(* CODESYS project BoshanMassa_13.3.project
   CustomField04_name: CustomField04
   CustomField06_name: CustomField06
   CustomField07_name: CustomField07
   CustomField09_name: CustomField09
   CustomField08_name: CustomField08
   CustomField02_name: CustomField02
   CustomField10_name: CustomField10
   CustomField01_name: CustomField01
   CustomField03_name: CustomField03
   CustomField05_name: CustomField05

Project tree, tasks and I/O mapping:
  MASSA : TM238LFDC24DT, Schneider Electric, order no. TM238LFDC24DT, version 4.0.1.28
      settings: Expansion Tasks.Expansion 1 Task Name = 'MAST'; Expansion Tasks.Expansion 2 Task Name = 'MAST'
    application Application
      task MAST (cyclic, interval 20 ms, priority 15, watchdog 100 ms x 1) calls POU_M
      program POU_M [LD]
      visualisation VisualizationM
      Symbols
    TM2DDI32DK : TM2DDI32DK, Schneider Electric, order no. TM2DDI32DK, version 4.0.1.28
        input  i_TZ_KO1 : BOOL  // ID0.I0
        input  i_TZ_KO2 : BOOL  // ID0.I1
        input  i_TZ_KO3 : BOOL  // ID0.I2
        input  i_TZ_KO4 : BOOL  // ID0.I3
        input  i_TZ_KO6 : BOOL  // ID0.I4
        input  i_TZ_KO7 : BOOL  // ID0.I5
        input  i_TZ_SMK517_37 : BOOL  // ID0.I6
        input  i_TZ_SMK517_5 : BOOL  // ID0.I7
        input  i_Nominal_SMK517_ATS : BOOL  // ID0.I8
        input  i_Avar_SMK517_ATS : BOOL  // ID0.I9
        input  i_TZ_SMK516_37 : BOOL  // ID0.I10
        input  i_TZ_SMK516_45 : BOOL  // ID0.I11
        input  i_TZ_KonvSMK516 : BOOL  // ID0.I12
        input  i_TZ_RazrSMK516 : BOOL  // ID0.I13
        input  i_TZ_EP80_1 : BOOL  // ID0.I15
        input  i_TZ_EP80_2 : BOOL  // ID0.I16
        input  i_Tros_KO1 : BOOL  // ID0.I17
        input  i_Tros_KO2 : BOOL  // ID0.I18
        input  i_Tros_KO3 : BOOL  // ID0.I19
        input  i_Tros_KO4 : BOOL  // ID0.I20
        input  i_Tros_KO6 : BOOL  // ID0.I21
        input  i_Tros_KO7 : BOOL  // ID0.I22
        input  i_Othod_SMK517 : BOOL  // ID0.I23
        input  i_Kozhuh_SMK517 : BOOL  // ID0.I24
        input  i_Othod_SMK516 : BOOL  // ID0.I25
        input  i_Kozhuh_SMK516 : BOOL  // ID0.I26
        input  i_Tros_KonvSMK516 : BOOL  // ID0.I27
        input  i_KEY_Protochka : BOOL  // ID0.I28
        input  i_Avar_PL024 : BOOL  // ID0.I31
        unmapped channels: ID0
    Serial Line 1
      Modbus_Manager : Modbus Manager, Schneider Electric, version 4.0.0.2
    Embedded Functions
      HSC : HSC, Schneider Electric, version 4.0.1.28
          settings: HSC00VarName = ''
      IO : IO, Schneider Electric, version 4.0.1.28
          input  i_Avar_PL012 : BOOL  // IW0.I0
          input  i_Rabota_PL250 : BOOL  // IW0.I1
          input  i_Avar_PL250 : BOOL  // IW0.I2
          input  i_Gotov_USM40 : BOOL  // IW0.I3
          input  i_Privoda_USM40_v_rabote : BOOL  // IW0.I4
          input  i_Liniya_USM40_v_rabote : BOOL  // IW0.I5
          input  i_TrosLentaUSM40 : BOOL  // IW0.I6
          input  i_Avar_USM40 : BOOL  // IW0.I7
          input  i_TZ_KO11 : BOOL  // IW0.I8
          input  i_Tros_KO11 : BOOL  // IW0.I9
          input  i_TZ_PL1 : BOOL  // IW0.I10
          input  i_TZ_PL2 : BOOL  // IW0.I11
          input  i_Vkl_Protoch517 : BOOL  // IW0.I12
          input  i_Otkl_Protoch517 : BOOL  // IW0.I13
          unmapped channels: IW0, QW0
      PTO_PWM : PTO_PWM, Schneider Electric, version 4.0.1.28
    CAN
      CANopen_Optimized : CANopen Optimized, Schneider Electric, order no. 1806, version 3.0.1.24
          settings: ConfigVersion = 50659584
        PL250 : Altivar 312, Schneider Electric, order no. 0, version 4.5.0.0
            settings: General Options.Optional Device = TRUE; NODEIDSAVED = 3; SDO Timeout = 1000000; EXPERTSETTINGS = True; Emergency-General Parameters.Emergency COBID = 16#83; Heartbeat-Producer Time = 200; PDO 16#1400.COBID = 16#80000203; PDO 16#1405.COBID = 16#00000303; PDO 16#1800.COBID = 16#80000183; PDO 16#1805.COBID = 16#00000283; Heartbeat-Consuming1.Heartbeat-Time = 300 ms; Drivecom command reg..Subindex = 16#00; Drivecom command reg..Subindex = 16#00; Target velocity.Index = 16#6042; Target velocity.Subindex = 16#00; Target velocity.ObjectLength = 16; Drivecom status register.Subindex = 16#00; Drivecom status register.Subindex = 16#00; Output frequency.Index = 16#2002; Output frequency.Subindex = 16#03; Output frequency.ObjectLength = 16; Motor Current.Index = 16#2002; Motor Current.Subindex = 16#05; Motor Current.ObjectLength = 16; SDO List.Set Guardtime.Index = 16#100C; SDO List.Set Guardtime.Subindex = 16#00; SDO List.Set Guardtime.Value = 16#00000000; SDO List.Set Guardtime.Size = 16; SDO List.Set Guardtime.AbortIfError = FALSE; SDO List.Set Guardtime.JumpToLine = FALSE; SDO List.Set Guardtime.Line = 0; SDO List.Set Lifetime.Index = 16#100D; SDO List.Set Lifetime.Subindex = 16#00; SDO List.Set Lifetime.Value = 16#00000000; SDO List.Set Lifetime.Size = 8; SDO List.Set Lifetime.AbortIfError = FALSE; SDO List.Set Lifetime.JumpToLine = FALSE; SDO List.Set Lifetime.Line = 0; SDO List.Set Heartbeat Consumer.Index = 16#1016; SDO List.Set Heartbeat Consumer.Subindex = 16#01;
              SDO List.Set Heartbeat Consumer.Value = 16#007F012C; SDO List.Set Heartbeat Consumer.Size = 32; SDO List.Set Heartbeat Consumer.AbortIfError = FALSE; SDO List.Set Heartbeat Consumer.JumpToLine = FALSE; SDO List.Set Heartbeat Consumer.Line = 0; SDO List.Set Heartbeat Producer.Index = 16#1017; SDO List.Set Heartbeat Producer.Subindex = 16#00; SDO List.Set Heartbeat Producer.Value = 16#000000C8; SDO List.Set Heartbeat Producer.Size = 16; SDO List.Set Heartbeat Producer.AbortIfError = FALSE; SDO List.Set Heartbeat Producer.JumpToLine = FALSE; SDO List.Set Heartbeat Producer.Line = 0; SDO List.Disable PDO.Index = 16#1400; SDO List.Disable PDO.Subindex = 16#01; SDO List.Disable PDO.Value = 16#80000203; SDO List.Disable PDO.Size = 32; SDO List.Disable PDO.AbortIfError = FALSE; SDO List.Disable PDO.JumpToLine = FALSE; SDO List.Disable PDO.Line = 0; SDO List.Disable PDO.Index = 16#1405; SDO List.Disable PDO.Subindex = 16#01; SDO List.Disable PDO.Value = 16#80000303; SDO List.Disable PDO.Size = 32; SDO List.Disable PDO.AbortIfError = FALSE; SDO List.Disable PDO.JumpToLine = FALSE; SDO List.Disable PDO.Line = 0; SDO List.Set transmission type.Index = 16#1405; SDO List.Set transmission type.Subindex = 16#02; SDO List.Set transmission type.Value = 16#FF; SDO List.Set transmission type.Size = 8; SDO List.Set transmission type.AbortIfError = FALSE; SDO List.Set transmission type.JumpToLine = FALSE; SDO List.Set transmission type.Line = 0; SDO List.Clear pdo mapping.Index = 16#1605; SDO List.Clear pdo mapping.Subindex = 16#00; SDO List.Clear pdo mapping.Value = 16#0; SDO List.Clear pdo mapping.Size = 8; SDO List.Clear pdo mapping.AbortIfError = FALSE; SDO List.Clear pdo mapping.JumpToLine = FALSE; SDO List.Clear pdo mapping.Line = 0;
              SDO List.Set Mapping.Index = 16#1605; SDO List.Set Mapping.Subindex = 16#01; SDO List.Set Mapping.Value = 16#60400010; SDO List.Set Mapping.Size = 32; SDO List.Set Mapping.AbortIfError = FALSE; SDO List.Set Mapping.JumpToLine = FALSE; SDO List.Set Mapping.Line = 0; SDO List.Set Mapping.Index = 16#1605; SDO List.Set Mapping.Subindex = 16#02; SDO List.Set Mapping.Value = 16#60420010; SDO List.Set Mapping.Size = 32; SDO List.Set Mapping.AbortIfError = FALSE; SDO List.Set Mapping.JumpToLine = FALSE; SDO List.Set Mapping.Line = 0; SDO List.Set number of pdos.Index = 16#1605; SDO List.Set number of pdos.Subindex = 16#00; SDO List.Set number of pdos.Value = 16#02; SDO List.Set number of pdos.Size = 8; SDO List.Set number of pdos.AbortIfError = FALSE; SDO List.Set number of pdos.JumpToLine = FALSE; SDO List.Set number of pdos.Line = 0; SDO List.Set and enable COB-ID.Index = 16#1405; SDO List.Set and enable COB-ID.Subindex = 16#01; SDO List.Set and enable COB-ID.Value = 16#00000303; SDO List.Set and enable COB-ID.Size = 32; SDO List.Set and enable COB-ID.AbortIfError = FALSE; SDO List.Set and enable COB-ID.JumpToLine = FALSE; SDO List.Set and enable COB-ID.Line = 0; SDO List.Disable PDO.Index = 16#1800; SDO List.Disable PDO.Subindex = 16#01; SDO List.Disable PDO.Value = 16#80000183; SDO List.Disable PDO.Size = 32; SDO List.Disable PDO.AbortIfError = FALSE; SDO List.Disable PDO.JumpToLine = FALSE; SDO List.Disable PDO.Line = 0; SDO List.Disable PDO.Index = 16#1805; SDO List.Disable PDO.Subindex = 16#01; SDO List.Disable PDO.Value = 16#80000283; SDO List.Disable PDO.Size = 32; SDO List.Disable PDO.AbortIfError = FALSE;
              SDO List.Disable PDO.JumpToLine = FALSE; SDO List.Disable PDO.Line = 0; SDO List.Set transmission type.Index = 16#1805; SDO List.Set transmission type.Subindex = 16#02; SDO List.Set transmission type.Value = 16#FF; SDO List.Set transmission type.Size = 8; SDO List.Set transmission type.AbortIfError = FALSE; SDO List.Set transmission type.JumpToLine = FALSE; SDO List.Set transmission type.Line = 0; SDO List.Set inhibit time.Index = 16#1805; SDO List.Set inhibit time.Subindex = 16#03; SDO List.Set inhibit time.Value = 16#001E; SDO List.Set inhibit time.Size = 16; SDO List.Set inhibit time.AbortIfError = FALSE; SDO List.Set inhibit time.JumpToLine = FALSE; SDO List.Set inhibit time.Line = 0; SDO List.Set event time.Index = 16#1805; SDO List.Set event time.Subindex = 16#05; SDO List.Set event time.Value = 16#0064; SDO List.Set event time.Size = 16; SDO List.Set event time.AbortIfError = FALSE; SDO List.Set event time.JumpToLine = FALSE; SDO List.Set event time.Line = 0; SDO List.Clear pdo mapping.Index = 16#1A05; SDO List.Clear pdo mapping.Subindex = 16#00; SDO List.Clear pdo mapping.Value = 16#0; SDO List.Clear pdo mapping.Size = 8; SDO List.Clear pdo mapping.AbortIfError = FALSE; SDO List.Clear pdo mapping.JumpToLine = FALSE; SDO List.Clear pdo mapping.Line = 0; SDO List.Set Mapping.Index = 16#1A05; SDO List.Set Mapping.Subindex = 16#01; SDO List.Set Mapping.Value = 16#60410010; SDO List.Set Mapping.Size = 32; SDO List.Set Mapping.AbortIfError = FALSE; SDO List.Set Mapping.JumpToLine = FALSE; SDO List.Set Mapping.Line = 0; SDO List.Set Mapping.Index = 16#1A05; SDO List.Set Mapping.Subindex = 16#02; SDO List.Set Mapping.Value = 16#20020310;
              SDO List.Set Mapping.Size = 32; SDO List.Set Mapping.AbortIfError = FALSE; SDO List.Set Mapping.JumpToLine = FALSE; SDO List.Set Mapping.Line = 0; SDO List.Set Mapping.Index = 16#1A05; SDO List.Set Mapping.Subindex = 16#03; SDO List.Set Mapping.Value = 16#20020510; SDO List.Set Mapping.Size = 32; SDO List.Set Mapping.AbortIfError = FALSE; SDO List.Set Mapping.JumpToLine = FALSE; SDO List.Set Mapping.Line = 0; SDO List.Set number of pdos.Index = 16#1A05; SDO List.Set number of pdos.Subindex = 16#00; SDO List.Set number of pdos.Value = 16#03; SDO List.Set number of pdos.Size = 8; SDO List.Set number of pdos.AbortIfError = FALSE; SDO List.Set number of pdos.JumpToLine = FALSE; SDO List.Set number of pdos.Line = 0; SDO List.Set and enable COB-ID.Index = 16#1805; SDO List.Set and enable COB-ID.Subindex = 16#01; SDO List.Set and enable COB-ID.Value = 16#00000283; SDO List.Set and enable COB-ID.Size = 32; SDO List.Set and enable COB-ID.AbortIfError = FALSE; SDO List.Set and enable COB-ID.JumpToLine = FALSE; SDO List.Set and enable COB-ID.Line = 0; ConfigVersion = 50659584
            output q_ATVPL250_Controlword : UINT  // Drivecom command reg.
            output q_ATVPL250_WriteVelocity : INT  // Target velocity
            input  i_ATVPL250_Status : UINT  // Drivecom status register
            input  i_ATVPL250_OutFrec : INT  // Output frequency
            input  i_ATVPL250_OutCur : UINT  // Motor Current
        PL024 : Altivar 312, Schneider Electric, order no. 0, version 4.5.0.0
            settings: General Options.Optional Device = TRUE; NODEIDSAVED = 5; SDO Timeout = 1000000; EXPERTSETTINGS = True; Emergency-General Parameters.Emergency COBID = 16#85; Heartbeat-Producer Time = 200; PDO 16#1400.COBID = 16#80000205; PDO 16#1405.COBID = 16#00000305; PDO 16#1800.COBID = 16#80000185; PDO 16#1805.COBID = 16#00000285; Heartbeat-Consuming1.Heartbeat-Time = 300 ms; Drivecom command reg..Subindex = 16#00; Drivecom command reg..Subindex = 16#00; Target velocity.Index = 16#6042; Target velocity.Subindex = 16#00; Target velocity.ObjectLength = 16; Drivecom status register.Subindex = 16#00; Drivecom status register.Subindex = 16#00; Output frequency.Index = 16#2002; Output frequency.Subindex = 16#03; Output frequency.ObjectLength = 16; Motor Current.Index = 16#2002; Motor Current.Subindex = 16#05; Motor Current.ObjectLength = 16; SDO List.Set Guardtime.Index = 16#100C; SDO List.Set Guardtime.Subindex = 16#00; SDO List.Set Guardtime.Value = 16#00000000; SDO List.Set Guardtime.Size = 16; SDO List.Set Guardtime.AbortIfError = FALSE; SDO List.Set Guardtime.JumpToLine = FALSE; SDO List.Set Guardtime.Line = 0; SDO List.Set Lifetime.Index = 16#100D; SDO List.Set Lifetime.Subindex = 16#00; SDO List.Set Lifetime.Value = 16#00000000; SDO List.Set Lifetime.Size = 8; SDO List.Set Lifetime.AbortIfError = FALSE; SDO List.Set Lifetime.JumpToLine = FALSE; SDO List.Set Lifetime.Line = 0; SDO List.Set Heartbeat Consumer.Index = 16#1016; SDO List.Set Heartbeat Consumer.Subindex = 16#01;
              SDO List.Set Heartbeat Consumer.Value = 16#007F012C; SDO List.Set Heartbeat Consumer.Size = 32; SDO List.Set Heartbeat Consumer.AbortIfError = FALSE; SDO List.Set Heartbeat Consumer.JumpToLine = FALSE; SDO List.Set Heartbeat Consumer.Line = 0; SDO List.Set Heartbeat Producer.Index = 16#1017; SDO List.Set Heartbeat Producer.Subindex = 16#00; SDO List.Set Heartbeat Producer.Value = 16#000000C8; SDO List.Set Heartbeat Producer.Size = 16; SDO List.Set Heartbeat Producer.AbortIfError = FALSE; SDO List.Set Heartbeat Producer.JumpToLine = FALSE; SDO List.Set Heartbeat Producer.Line = 0; SDO List.Disable PDO.Index = 16#1400; SDO List.Disable PDO.Subindex = 16#01; SDO List.Disable PDO.Value = 16#80000205; SDO List.Disable PDO.Size = 32; SDO List.Disable PDO.AbortIfError = FALSE; SDO List.Disable PDO.JumpToLine = FALSE; SDO List.Disable PDO.Line = 0; SDO List.Disable PDO.Index = 16#1405; SDO List.Disable PDO.Subindex = 16#01; SDO List.Disable PDO.Value = 16#80000305; SDO List.Disable PDO.Size = 32; SDO List.Disable PDO.AbortIfError = FALSE; SDO List.Disable PDO.JumpToLine = FALSE; SDO List.Disable PDO.Line = 0; SDO List.Set transmission type.Index = 16#1405; SDO List.Set transmission type.Subindex = 16#02; SDO List.Set transmission type.Value = 16#FF; SDO List.Set transmission type.Size = 8; SDO List.Set transmission type.AbortIfError = FALSE; SDO List.Set transmission type.JumpToLine = FALSE; SDO List.Set transmission type.Line = 0; SDO List.Clear pdo mapping.Index = 16#1605; SDO List.Clear pdo mapping.Subindex = 16#00; SDO List.Clear pdo mapping.Value = 16#0; SDO List.Clear pdo mapping.Size = 8; SDO List.Clear pdo mapping.AbortIfError = FALSE; SDO List.Clear pdo mapping.JumpToLine = FALSE; SDO List.Clear pdo mapping.Line = 0;
              SDO List.Set Mapping.Index = 16#1605; SDO List.Set Mapping.Subindex = 16#01; SDO List.Set Mapping.Value = 16#60400010; SDO List.Set Mapping.Size = 32; SDO List.Set Mapping.AbortIfError = FALSE; SDO List.Set Mapping.JumpToLine = FALSE; SDO List.Set Mapping.Line = 0; SDO List.Set Mapping.Index = 16#1605; SDO List.Set Mapping.Subindex = 16#02; SDO List.Set Mapping.Value = 16#60420010; SDO List.Set Mapping.Size = 32; SDO List.Set Mapping.AbortIfError = FALSE; SDO List.Set Mapping.JumpToLine = FALSE; SDO List.Set Mapping.Line = 0; SDO List.Set number of pdos.Index = 16#1605; SDO List.Set number of pdos.Subindex = 16#00; SDO List.Set number of pdos.Value = 16#02; SDO List.Set number of pdos.Size = 8; SDO List.Set number of pdos.AbortIfError = FALSE; SDO List.Set number of pdos.JumpToLine = FALSE; SDO List.Set number of pdos.Line = 0; SDO List.Set and enable COB-ID.Index = 16#1405; SDO List.Set and enable COB-ID.Subindex = 16#01; SDO List.Set and enable COB-ID.Value = 16#00000305; SDO List.Set and enable COB-ID.Size = 32; SDO List.Set and enable COB-ID.AbortIfError = FALSE; SDO List.Set and enable COB-ID.JumpToLine = FALSE; SDO List.Set and enable COB-ID.Line = 0; SDO List.Disable PDO.Index = 16#1800; SDO List.Disable PDO.Subindex = 16#01; SDO List.Disable PDO.Value = 16#80000185; SDO List.Disable PDO.Size = 32; SDO List.Disable PDO.AbortIfError = FALSE; SDO List.Disable PDO.JumpToLine = FALSE; SDO List.Disable PDO.Line = 0; SDO List.Disable PDO.Index = 16#1805; SDO List.Disable PDO.Subindex = 16#01; SDO List.Disable PDO.Value = 16#80000285; SDO List.Disable PDO.Size = 32; SDO List.Disable PDO.AbortIfError = FALSE;
              SDO List.Disable PDO.JumpToLine = FALSE; SDO List.Disable PDO.Line = 0; SDO List.Set transmission type.Index = 16#1805; SDO List.Set transmission type.Subindex = 16#02; SDO List.Set transmission type.Value = 16#FF; SDO List.Set transmission type.Size = 8; SDO List.Set transmission type.AbortIfError = FALSE; SDO List.Set transmission type.JumpToLine = FALSE; SDO List.Set transmission type.Line = 0; SDO List.Set inhibit time.Index = 16#1805; SDO List.Set inhibit time.Subindex = 16#03; SDO List.Set inhibit time.Value = 16#001E; SDO List.Set inhibit time.Size = 16; SDO List.Set inhibit time.AbortIfError = FALSE; SDO List.Set inhibit time.JumpToLine = FALSE; SDO List.Set inhibit time.Line = 0; SDO List.Set event time.Index = 16#1805; SDO List.Set event time.Subindex = 16#05; SDO List.Set event time.Value = 16#0064; SDO List.Set event time.Size = 16; SDO List.Set event time.AbortIfError = FALSE; SDO List.Set event time.JumpToLine = FALSE; SDO List.Set event time.Line = 0; SDO List.Clear pdo mapping.Index = 16#1A05; SDO List.Clear pdo mapping.Subindex = 16#00; SDO List.Clear pdo mapping.Value = 16#0; SDO List.Clear pdo mapping.Size = 8; SDO List.Clear pdo mapping.AbortIfError = FALSE; SDO List.Clear pdo mapping.JumpToLine = FALSE; SDO List.Clear pdo mapping.Line = 0; SDO List.Set Mapping.Index = 16#1A05; SDO List.Set Mapping.Subindex = 16#01; SDO List.Set Mapping.Value = 16#60410010; SDO List.Set Mapping.Size = 32; SDO List.Set Mapping.AbortIfError = FALSE; SDO List.Set Mapping.JumpToLine = FALSE; SDO List.Set Mapping.Line = 0; SDO List.Set Mapping.Index = 16#1A05; SDO List.Set Mapping.Subindex = 16#02; SDO List.Set Mapping.Value = 16#20020310;
              SDO List.Set Mapping.Size = 32; SDO List.Set Mapping.AbortIfError = FALSE; SDO List.Set Mapping.JumpToLine = FALSE; SDO List.Set Mapping.Line = 0; SDO List.Set Mapping.Index = 16#1A05; SDO List.Set Mapping.Subindex = 16#03; SDO List.Set Mapping.Value = 16#20020510; SDO List.Set Mapping.Size = 32; SDO List.Set Mapping.AbortIfError = FALSE; SDO List.Set Mapping.JumpToLine = FALSE; SDO List.Set Mapping.Line = 0; SDO List.Set number of pdos.Index = 16#1A05; SDO List.Set number of pdos.Subindex = 16#00; SDO List.Set number of pdos.Value = 16#03; SDO List.Set number of pdos.Size = 8; SDO List.Set number of pdos.AbortIfError = FALSE; SDO List.Set number of pdos.JumpToLine = FALSE; SDO List.Set number of pdos.Line = 0; SDO List.Set and enable COB-ID.Index = 16#1805; SDO List.Set and enable COB-ID.Subindex = 16#01; SDO List.Set and enable COB-ID.Value = 16#00000285; SDO List.Set and enable COB-ID.Size = 32; SDO List.Set and enable COB-ID.AbortIfError = FALSE; SDO List.Set and enable COB-ID.JumpToLine = FALSE; SDO List.Set and enable COB-ID.Line = 0; ConfigVersion = 50659584
            output q_ATVPL024_Controlword : UINT  // Drivecom command reg.
            output q_ATVPL024_WriteVelocity : INT  // Target velocity
            input  i_ATVPL024_Status : UINT  // Drivecom status register
            input  i_ATVPL024_OutFrec : INT  // Output frequency
            input  i_ATVPL024_OutCur : UINT  // Motor Current
        RazrSMK516 : Altivar 312, Schneider Electric, order no. 0, version 4.5.0.0
            settings: General Options.Optional Device = TRUE; NODEIDSAVED = 7; SDO Timeout = 1000000; EXPERTSETTINGS = True; Emergency-General Parameters.Emergency COBID = 16#87; Heartbeat-Producer Time = 200; PDO 16#1400.COBID = 16#80000207; PDO 16#1405.COBID = 16#00000307; PDO 16#1800.COBID = 16#80000187; PDO 16#1805.COBID = 16#00000287; Heartbeat-Consuming1.Heartbeat-Time = 300 ms; Drivecom command reg..Subindex = 16#00; Drivecom command reg..Subindex = 16#00; Target velocity.Index = 16#6042; Target velocity.Subindex = 16#00; Target velocity.ObjectLength = 16; Drivecom status register.Subindex = 16#00; Drivecom status register.Subindex = 16#00; Output frequency.Index = 16#2002; Output frequency.Subindex = 16#03; Output frequency.ObjectLength = 16; Motor Current.Index = 16#2002; Motor Current.Subindex = 16#05; Motor Current.ObjectLength = 16; SDO List.Set Guardtime.Index = 16#100C; SDO List.Set Guardtime.Subindex = 16#00; SDO List.Set Guardtime.Value = 16#00000000; SDO List.Set Guardtime.Size = 16; SDO List.Set Guardtime.AbortIfError = FALSE; SDO List.Set Guardtime.JumpToLine = FALSE; SDO List.Set Guardtime.Line = 0; SDO List.Set Lifetime.Index = 16#100D; SDO List.Set Lifetime.Subindex = 16#00; SDO List.Set Lifetime.Value = 16#00000000; SDO List.Set Lifetime.Size = 8; SDO List.Set Lifetime.AbortIfError = FALSE; SDO List.Set Lifetime.JumpToLine = FALSE; SDO List.Set Lifetime.Line = 0; SDO List.Set Heartbeat Consumer.Index = 16#1016; SDO List.Set Heartbeat Consumer.Subindex = 16#01;
              SDO List.Set Heartbeat Consumer.Value = 16#007F012C; SDO List.Set Heartbeat Consumer.Size = 32; SDO List.Set Heartbeat Consumer.AbortIfError = FALSE; SDO List.Set Heartbeat Consumer.JumpToLine = FALSE; SDO List.Set Heartbeat Consumer.Line = 0; SDO List.Set Heartbeat Producer.Index = 16#1017; SDO List.Set Heartbeat Producer.Subindex = 16#00; SDO List.Set Heartbeat Producer.Value = 16#000000C8; SDO List.Set Heartbeat Producer.Size = 16; SDO List.Set Heartbeat Producer.AbortIfError = FALSE; SDO List.Set Heartbeat Producer.JumpToLine = FALSE; SDO List.Set Heartbeat Producer.Line = 0; SDO List.Disable PDO.Index = 16#1400; SDO List.Disable PDO.Subindex = 16#01; SDO List.Disable PDO.Value = 16#80000207; SDO List.Disable PDO.Size = 32; SDO List.Disable PDO.AbortIfError = FALSE; SDO List.Disable PDO.JumpToLine = FALSE; SDO List.Disable PDO.Line = 0; SDO List.Disable PDO.Index = 16#1405; SDO List.Disable PDO.Subindex = 16#01; SDO List.Disable PDO.Value = 16#80000307; SDO List.Disable PDO.Size = 32; SDO List.Disable PDO.AbortIfError = FALSE; SDO List.Disable PDO.JumpToLine = FALSE; SDO List.Disable PDO.Line = 0; SDO List.Set transmission type.Index = 16#1405; SDO List.Set transmission type.Subindex = 16#02; SDO List.Set transmission type.Value = 16#FF; SDO List.Set transmission type.Size = 8; SDO List.Set transmission type.AbortIfError = FALSE; SDO List.Set transmission type.JumpToLine = FALSE; SDO List.Set transmission type.Line = 0; SDO List.Clear pdo mapping.Index = 16#1605; SDO List.Clear pdo mapping.Subindex = 16#00; SDO List.Clear pdo mapping.Value = 16#0; SDO List.Clear pdo mapping.Size = 8; SDO List.Clear pdo mapping.AbortIfError = FALSE; SDO List.Clear pdo mapping.JumpToLine = FALSE; SDO List.Clear pdo mapping.Line = 0;
              SDO List.Set Mapping.Index = 16#1605; SDO List.Set Mapping.Subindex = 16#01; SDO List.Set Mapping.Value = 16#60400010; SDO List.Set Mapping.Size = 32; SDO List.Set Mapping.AbortIfError = FALSE; SDO List.Set Mapping.JumpToLine = FALSE; SDO List.Set Mapping.Line = 0; SDO List.Set Mapping.Index = 16#1605; SDO List.Set Mapping.Subindex = 16#02; SDO List.Set Mapping.Value = 16#60420010; SDO List.Set Mapping.Size = 32; SDO List.Set Mapping.AbortIfError = FALSE; SDO List.Set Mapping.JumpToLine = FALSE; SDO List.Set Mapping.Line = 0; SDO List.Set number of pdos.Index = 16#1605; SDO List.Set number of pdos.Subindex = 16#00; SDO List.Set number of pdos.Value = 16#02; SDO List.Set number of pdos.Size = 8; SDO List.Set number of pdos.AbortIfError = FALSE; SDO List.Set number of pdos.JumpToLine = FALSE; SDO List.Set number of pdos.Line = 0; SDO List.Set and enable COB-ID.Index = 16#1405; SDO List.Set and enable COB-ID.Subindex = 16#01; SDO List.Set and enable COB-ID.Value = 16#00000307; SDO List.Set and enable COB-ID.Size = 32; SDO List.Set and enable COB-ID.AbortIfError = FALSE; SDO List.Set and enable COB-ID.JumpToLine = FALSE; SDO List.Set and enable COB-ID.Line = 0; SDO List.Disable PDO.Index = 16#1800; SDO List.Disable PDO.Subindex = 16#01; SDO List.Disable PDO.Value = 16#80000187; SDO List.Disable PDO.Size = 32; SDO List.Disable PDO.AbortIfError = FALSE; SDO List.Disable PDO.JumpToLine = FALSE; SDO List.Disable PDO.Line = 0; SDO List.Disable PDO.Index = 16#1805; SDO List.Disable PDO.Subindex = 16#01; SDO List.Disable PDO.Value = 16#80000287; SDO List.Disable PDO.Size = 32; SDO List.Disable PDO.AbortIfError = FALSE;
              SDO List.Disable PDO.JumpToLine = FALSE; SDO List.Disable PDO.Line = 0; SDO List.Set transmission type.Index = 16#1805; SDO List.Set transmission type.Subindex = 16#02; SDO List.Set transmission type.Value = 16#FF; SDO List.Set transmission type.Size = 8; SDO List.Set transmission type.AbortIfError = FALSE; SDO List.Set transmission type.JumpToLine = FALSE; SDO List.Set transmission type.Line = 0; SDO List.Set inhibit time.Index = 16#1805; SDO List.Set inhibit time.Subindex = 16#03; SDO List.Set inhibit time.Value = 16#001E; SDO List.Set inhibit time.Size = 16; SDO List.Set inhibit time.AbortIfError = FALSE; SDO List.Set inhibit time.JumpToLine = FALSE; SDO List.Set inhibit time.Line = 0; SDO List.Set event time.Index = 16#1805; SDO List.Set event time.Subindex = 16#05; SDO List.Set event time.Value = 16#0064; SDO List.Set event time.Size = 16; SDO List.Set event time.AbortIfError = FALSE; SDO List.Set event time.JumpToLine = FALSE; SDO List.Set event time.Line = 0; SDO List.Clear pdo mapping.Index = 16#1A05; SDO List.Clear pdo mapping.Subindex = 16#00; SDO List.Clear pdo mapping.Value = 16#0; SDO List.Clear pdo mapping.Size = 8; SDO List.Clear pdo mapping.AbortIfError = FALSE; SDO List.Clear pdo mapping.JumpToLine = FALSE; SDO List.Clear pdo mapping.Line = 0; SDO List.Set Mapping.Index = 16#1A05; SDO List.Set Mapping.Subindex = 16#01; SDO List.Set Mapping.Value = 16#60410010; SDO List.Set Mapping.Size = 32; SDO List.Set Mapping.AbortIfError = FALSE; SDO List.Set Mapping.JumpToLine = FALSE; SDO List.Set Mapping.Line = 0; SDO List.Set Mapping.Index = 16#1A05; SDO List.Set Mapping.Subindex = 16#02; SDO List.Set Mapping.Value = 16#20020310;
              SDO List.Set Mapping.Size = 32; SDO List.Set Mapping.AbortIfError = FALSE; SDO List.Set Mapping.JumpToLine = FALSE; SDO List.Set Mapping.Line = 0; SDO List.Set Mapping.Index = 16#1A05; SDO List.Set Mapping.Subindex = 16#03; SDO List.Set Mapping.Value = 16#20020510; SDO List.Set Mapping.Size = 32; SDO List.Set Mapping.AbortIfError = FALSE; SDO List.Set Mapping.JumpToLine = FALSE; SDO List.Set Mapping.Line = 0; SDO List.Set number of pdos.Index = 16#1A05; SDO List.Set number of pdos.Subindex = 16#00; SDO List.Set number of pdos.Value = 16#03; SDO List.Set number of pdos.Size = 8; SDO List.Set number of pdos.AbortIfError = FALSE; SDO List.Set number of pdos.JumpToLine = FALSE; SDO List.Set number of pdos.Line = 0; SDO List.Set and enable COB-ID.Index = 16#1805; SDO List.Set and enable COB-ID.Subindex = 16#01; SDO List.Set and enable COB-ID.Value = 16#00000287; SDO List.Set and enable COB-ID.Size = 32; SDO List.Set and enable COB-ID.AbortIfError = FALSE; SDO List.Set and enable COB-ID.JumpToLine = FALSE; SDO List.Set and enable COB-ID.Line = 0; ConfigVersion = 50659584
            output q_ATVRazrSMK516_Controlword : UINT  // Drivecom command reg.
            output q_ATVRazrSMK516_WriteVelocity : INT  // Target velocity
            input  i_ATVRazrSMK516_Status : UINT  // Drivecom status register
            input  i_ATVRazrSMK516_OutFrec : INT  // Output frequency
            input  i_ATVRazrSMK516_OutCur : UINT  // Motor Current
        PL012 : Altivar 312, Schneider Electric, order no. 0, version 4.5.0.0
            settings: General Options.Optional Device = TRUE; NODEIDSAVED = 1; SDO Timeout = 1000000; EXPERTSETTINGS = True; Heartbeat-Producer Time = 200; PDO 16#1405.COBID = 16#00000301; PDO 16#1405.available PDO-Parameter.Inhibit Time available = TRUE; Generic COBID = '$NODEID+16#0300'; PDO 16#1805.COBID = 16#00000281; Heartbeat-Consuming1.Heartbeat-Time = 300 ms; Drivecom command reg..Subindex = 16#00; Drivecom command reg..Subindex = 16#00; Target velocity.Index = 16#6042; Target velocity.Subindex = 16#00; Target velocity.ObjectLength = 16; Drivecom status register.Subindex = 16#00; Drivecom status register.Subindex = 16#00; Output frequency.Index = 16#2002; Output frequency.Subindex = 16#03; Output frequency.ObjectLength = 16; Motor Current.Index = 16#2002; Motor Current.Subindex = 16#05; Motor Current.ObjectLength = 16; SDO List.Set Guardtime.Index = 16#100C; SDO List.Set Guardtime.Subindex = 16#00; SDO List.Set Guardtime.Value = 16#00000000; SDO List.Set Guardtime.Size = 16; SDO List.Set Guardtime.AbortIfError = FALSE; SDO List.Set Guardtime.JumpToLine = FALSE; SDO List.Set Guardtime.Line = 0; SDO List.Set Lifetime.Index = 16#100D; SDO List.Set Lifetime.Subindex = 16#00; SDO List.Set Lifetime.Value = 16#00000000; SDO List.Set Lifetime.Size = 8; SDO List.Set Lifetime.AbortIfError = FALSE; SDO List.Set Lifetime.JumpToLine = FALSE; SDO List.Set Lifetime.Line = 0; SDO List.Set Heartbeat Consumer.Index = 16#1016; SDO List.Set Heartbeat Consumer.Subindex = 16#01; SDO List.Set Heartbeat Consumer.Value = 16#007F012C;
              SDO List.Set Heartbeat Consumer.Size = 32; SDO List.Set Heartbeat Consumer.AbortIfError = FALSE; SDO List.Set Heartbeat Consumer.JumpToLine = FALSE; SDO List.Set Heartbeat Consumer.Line = 0; SDO List.Set Heartbeat Producer.Index = 16#1017; SDO List.Set Heartbeat Producer.Subindex = 16#00; SDO List.Set Heartbeat Producer.Value = 16#000000C8; SDO List.Set Heartbeat Producer.Size = 16; SDO List.Set Heartbeat Producer.AbortIfError = FALSE; SDO List.Set Heartbeat Producer.JumpToLine = FALSE; SDO List.Set Heartbeat Producer.Line = 0; SDO List.Disable PDO.Index = 16#1400; SDO List.Disable PDO.Subindex = 16#01; SDO List.Disable PDO.Value = 16#80000201; SDO List.Disable PDO.Size = 32; SDO List.Disable PDO.AbortIfError = FALSE; SDO List.Disable PDO.JumpToLine = FALSE; SDO List.Disable PDO.Line = 0; SDO List.Disable PDO.Index = 16#1405; SDO List.Disable PDO.Subindex = 16#01; SDO List.Disable PDO.Value = 16#80000301; SDO List.Disable PDO.Size = 32; SDO List.Disable PDO.AbortIfError = FALSE; SDO List.Disable PDO.JumpToLine = FALSE; SDO List.Disable PDO.Line = 0; SDO List.Set transmission type.Index = 16#1405; SDO List.Set transmission type.Subindex = 16#02; SDO List.Set transmission type.Value = 16#FF; SDO List.Set transmission type.Size = 8; SDO List.Set transmission type.AbortIfError = FALSE; SDO List.Set transmission type.JumpToLine = FALSE; SDO List.Set transmission type.Line = 0; SDO List.Set inhibit time.Index = 16#1405; SDO List.Set inhibit time.Subindex = 16#03; SDO List.Set inhibit time.Value = 16#0000; SDO List.Set inhibit time.Size = 16; SDO List.Set inhibit time.AbortIfError = FALSE; SDO List.Set inhibit time.JumpToLine = FALSE; SDO List.Set inhibit time.Line = 0; SDO List.Clear pdo mapping.Index = 16#1605;
              SDO List.Clear pdo mapping.Subindex = 16#00; SDO List.Clear pdo mapping.Value = 16#0; SDO List.Clear pdo mapping.Size = 8; SDO List.Clear pdo mapping.AbortIfError = FALSE; SDO List.Clear pdo mapping.JumpToLine = FALSE; SDO List.Clear pdo mapping.Line = 0; SDO List.Set Mapping.Index = 16#1605; SDO List.Set Mapping.Subindex = 16#01; SDO List.Set Mapping.Value = 16#60400010; SDO List.Set Mapping.Size = 32; SDO List.Set Mapping.AbortIfError = FALSE; SDO List.Set Mapping.JumpToLine = FALSE; SDO List.Set Mapping.Line = 0; SDO List.Set Mapping.Index = 16#1605; SDO List.Set Mapping.Subindex = 16#02; SDO List.Set Mapping.Value = 16#60420010; SDO List.Set Mapping.Size = 32; SDO List.Set Mapping.AbortIfError = FALSE; SDO List.Set Mapping.JumpToLine = FALSE; SDO List.Set Mapping.Line = 0; SDO List.Set number of pdos.Index = 16#1605; SDO List.Set number of pdos.Subindex = 16#00; SDO List.Set number of pdos.Value = 16#02; SDO List.Set number of pdos.Size = 8; SDO List.Set number of pdos.AbortIfError = FALSE; SDO List.Set number of pdos.JumpToLine = FALSE; SDO List.Set number of pdos.Line = 0; SDO List.Set and enable COB-ID.Index = 16#1405; SDO List.Set and enable COB-ID.Subindex = 16#01; SDO List.Set and enable COB-ID.Value = 16#00000301; SDO List.Set and enable COB-ID.Size = 32; SDO List.Set and enable COB-ID.AbortIfError = FALSE; SDO List.Set and enable COB-ID.JumpToLine = FALSE; SDO List.Set and enable COB-ID.Line = 0; SDO List.Disable PDO.Index = 16#1800; SDO List.Disable PDO.Subindex = 16#01; SDO List.Disable PDO.Value = 16#80000181; SDO List.Disable PDO.Size = 32; SDO List.Disable PDO.AbortIfError = FALSE; SDO List.Disable PDO.JumpToLine = FALSE;
              SDO List.Disable PDO.Line = 0; SDO List.Disable PDO.Index = 16#1805; SDO List.Disable PDO.Subindex = 16#01; SDO List.Disable PDO.Value = 16#80000281; SDO List.Disable PDO.Size = 32; SDO List.Disable PDO.AbortIfError = FALSE; SDO List.Disable PDO.JumpToLine = FALSE; SDO List.Disable PDO.Line = 0; SDO List.Set transmission type.Index = 16#1805; SDO List.Set transmission type.Subindex = 16#02; SDO List.Set transmission type.Value = 16#FF; SDO List.Set transmission type.Size = 8; SDO List.Set transmission type.AbortIfError = FALSE; SDO List.Set transmission type.JumpToLine = FALSE; SDO List.Set transmission type.Line = 0; SDO List.Set inhibit time.Index = 16#1805; SDO List.Set inhibit time.Subindex = 16#03; SDO List.Set inhibit time.Value = 16#001E; SDO List.Set inhibit time.Size = 16; SDO List.Set inhibit time.AbortIfError = FALSE; SDO List.Set inhibit time.JumpToLine = FALSE; SDO List.Set inhibit time.Line = 0; SDO List.Set event time.Index = 16#1805; SDO List.Set event time.Subindex = 16#05; SDO List.Set event time.Value = 16#0064; SDO List.Set event time.Size = 16; SDO List.Set event time.AbortIfError = FALSE; SDO List.Set event time.JumpToLine = FALSE; SDO List.Set event time.Line = 0; SDO List.Clear pdo mapping.Index = 16#1A05; SDO List.Clear pdo mapping.Subindex = 16#00; SDO List.Clear pdo mapping.Value = 16#0; SDO List.Clear pdo mapping.Size = 8; SDO List.Clear pdo mapping.AbortIfError = FALSE; SDO List.Clear pdo mapping.JumpToLine = FALSE; SDO List.Clear pdo mapping.Line = 0; SDO List.Set Mapping.Index = 16#1A05; SDO List.Set Mapping.Subindex = 16#01; SDO List.Set Mapping.Value = 16#60410010; SDO List.Set Mapping.Size = 32;
              SDO List.Set Mapping.AbortIfError = FALSE; SDO List.Set Mapping.JumpToLine = FALSE; SDO List.Set Mapping.Line = 0; SDO List.Set Mapping.Index = 16#1A05; SDO List.Set Mapping.Subindex = 16#02; SDO List.Set Mapping.Value = 16#20020310; SDO List.Set Mapping.Size = 32; SDO List.Set Mapping.AbortIfError = FALSE; SDO List.Set Mapping.JumpToLine = FALSE; SDO List.Set Mapping.Line = 0; SDO List.Set Mapping.Index = 16#1A05; SDO List.Set Mapping.Subindex = 16#03; SDO List.Set Mapping.Value = 16#20020510; SDO List.Set Mapping.Size = 32; SDO List.Set Mapping.AbortIfError = FALSE; SDO List.Set Mapping.JumpToLine = FALSE; SDO List.Set Mapping.Line = 0; SDO List.Set number of pdos.Index = 16#1A05; SDO List.Set number of pdos.Subindex = 16#00; SDO List.Set number of pdos.Value = 16#03; SDO List.Set number of pdos.Size = 8; SDO List.Set number of pdos.AbortIfError = FALSE; SDO List.Set number of pdos.JumpToLine = FALSE; SDO List.Set number of pdos.Line = 0; SDO List.Set and enable COB-ID.Index = 16#1805; SDO List.Set and enable COB-ID.Subindex = 16#01; SDO List.Set and enable COB-ID.Value = 16#00000281; SDO List.Set and enable COB-ID.Size = 32; SDO List.Set and enable COB-ID.AbortIfError = FALSE; SDO List.Set and enable COB-ID.JumpToLine = FALSE; SDO List.Set and enable COB-ID.Line = 0; ConfigVersion = 50659584
            output q_ATVPL012_Controlword : UINT  // Drivecom command reg.
            output q_ATVPL012_WriteVelocity : INT  // Target velocity
            input  i_ATVPL012_Status : UINT  // Drivecom status register
            input  i_ATVPL012_OutFrec : INT  // Output frequency
            input  i_ATVPL012_OutCur : UINT  // Motor Current
    TM2DDO32TK : TM2DDO32TK, Schneider Electric, order no. TM2DDO32TK, version 4.0.1.28
        output q_Pusk_KO1 : BOOL  // QD0.Q0
        output q_Pusk_KO2 : BOOL  // QD0.Q1
        output q_Pusk_KO3 : BOOL  // QD0.Q2
        output q_Pusk_KO4 : BOOL  // QD0.Q3
        output q_Pusk_KO6 : BOOL  // QD0.Q4
        output q_Pusk_KO7 : BOOL  // QD0.Q5
        output q_Pusk_SMK517_37 : BOOL  // QD0.Q6
        output q_Pusk_SMK517_ATS : BOOL  // QD0.Q7
        output q_Pusk_SMK516_37 : BOOL  // QD0.Q8
        output q_Pusk_SMK516_45 : BOOL  // QD0.Q9
        output q_Pusk_KonvSMK516 : BOOL  // QD0.Q10
        output q_Pusk_RazrSMK516 : BOOL  // QD0.Q11
        output q_Pusk_EP80_1 : BOOL  // QD0.Q12
        output q_Pusk_EP80_2 : BOOL  // QD0.Q13
        output q_Pusk_PL024 : BOOL  // QD0.Q14
        output q_Pusk_PL012 : BOOL  // QD0.Q15
        output q_Pusk_PL250 : BOOL  // QD0.Q16
        output q_Podgot_USM40 : BOOL  // QD0.Q17
        output q_Pusk_PrivodaUSM40 : BOOL  // QD0.Q18
        output q_Pusk_LiniyaUSM40 : BOOL  // QD0.Q19
        output q_Pusk_KO11 : BOOL  // QD0.Q20
        output q_Pusk_PL1 : BOOL  // QD0.Q21
        output q_Pusk_PL2 : BOOL  // QD0.Q22
        output q_Zvonok : BOOL  // QD0.Q23
        output q_SMK517_Prjamo : BOOL  // QD0.Q24
        output q_SMK517_Revers : BOOL  // QD0.Q25
        output q_Vkl_Voda_PL250 : BOOL  // QD0.Q26
        unmapped channels: QD0
    Serial Line 2
      SoMachine_Network_Manager : SoMachine-Network Manager, Schneider Electric, version 4.0.0.2
  XBTGT7340_M : XBTGT7340, Schneider Electric, order no. XBTGT7340, version 3.5.3.54
    HMI Application
    Ethernet
    COM1
      SoMachine_Network_Manager_1 : SoMachine-Network Manager, Schneider Electric, version 4.0.0.2
    USB
      SoMachine_Network_Manager4 : SoMachine-Network Manager, Schneider Electric, version 4.0.0.2
    COM2
      SoMachine_Network_Manager_3 : SoMachine-Network Manager, Schneider Electric, version 4.0.0.2
  MachineLayoutPicture
  Vijeo Designer Project Container Data
  text list GlobalTextList
  Vijeo Designer Project Container
*)

// MASSA/Application/POU_M
PROGRAM POU_M
VAR
	// Пуск КО-4 из панели в ручном режиме.
	Pusk_HMI_KO1: BOOL;
	// Промежуточная катушка тросового выключателя КО-1 для фиксации защиты.
	m_Tros_KO1: BOOL;
	// Квитирование из панели.
	Kvitir_HMI: BOOL;
	// Пуск КО-2 из панели в ручном режиме.
	Pusk_HMI_KO2: BOOL;
	// Пуск КО-3 из панели в ручном режиме.
	Pusk_HMI_KO3: BOOL;
	// Пуск КО-4 из панели в ручном режиме.
	Pusk_HMI_KO4: BOOL;
	// Пуск КО-6 из панели в ручном режиме.
	Pusk_HMI_KO6: BOOL;
	// Пуск КО-7 из панели в ручном режиме.
	Pusk_HMI_KO7: BOOL;
	// Пуск КО-11 из панели в ручном режиме.
	Pusk_HMI_KO11: BOOL;
	//Пуск PL024 из панели в ручном режиме.
	Pusk_HMI_PL024: BOOL;
	//Пуск PL012 из панели в ручном режиме.
	Pusk_HMI_PL012: BOOL;
	//Пуск ЭП80 на КО-2 из панели в ручном режиме.
	Pusk_HMI_EP80_1: BOOL;
	//Пуск 37 кВт на СМК517 из панели в ручном режиме.
	Pusk_HMI_SMK517_37: BOOL;
	//Пуск 5,5 кВт на СМК517 из панели в ручном режиме.
	Pusk_HMI_SMK517_5: BOOL;
	//Пуск 45 кВт на СМК516 из панели в ручном режиме.
	Pusk_HMI_SMK516_45: BOOL;
	//Пуск 37 кВт на СМК516 из панели в ручном режиме.
	Pusk_HMI_SMK516_37: BOOL;
	//Пуск разравниватель СМК516 из панели в ручном режиме.
	Pusk_HMI_RazrSMK516: BOOL;
	//Пуск конвейер СМК516 из панели в ручном режиме.
	Pusk_HMI_KonvSMK516: BOOL;
	//Пуск PL250 из панели в ручном режиме.
	Pusk_HMI_PL250: BOOL;
	//Включение воды в смеситель PL250 из панели в ручном режиме.
	Pusk_HMI_VodaPL250: BOOL;
	//Пуск ЭП80 на КО-6 из панели в ручном режиме.
	Pusk_HMI_EP80_2: BOOL;
	//Пуск привода для УСМ40 из панели в ручном режиме.
	Pusk_HMI_PrivodaUSM40: BOOL;
	//Пуск линия для УСМ40 из панели в ручном режиме.
	Pusk_HMI_LiniyaUSM40: BOOL;
	//Пуск ПЛ1-10 №1 из панели в ручном режиме.
	Pusk_HMI_PL1: BOOL;
	//Пуск ПЛ1-10 №2 из панели в ручном режиме.
	Pusk_HMI_PL2: BOOL;
	//Пуск 5,5 кВт на СМК 517 в реверс из панели в ручном режиме.
	Pusk_HMI_SMK517_5_Rev: BOOL;
	//Включение звонка из панели в ручном режиме.	
	Pusk_HMI_Zvonok: BOOL;
	TP_mZV1: TP;
	// Маркер первого звонка перед пуском.
	mZV1: BOOL;
	TP_mZV2: TP;
	TP_mPauza: TP;
	// Маркер паузы после первого звонка перед пуском.
	mPauza: BOOL;
	// Маркер второго звонка перед пуском.
	mZV2: BOOL;
	// Промежуточная катушка тросового выключателя КО-2 для фиксации защиты.
	m_Tros_KO2: BOOL;
	// Промежуточная катушка тросового выключателя КО-3 для фиксации защиты.
	m_Tros_KO3: BOOL;
	// Промежуточная катушка тросового выключателя КО-4 для фиксации защиты.
	m_Tros_KO4: BOOL;
	// Промежуточная катушка тросового выключателя КО-6 для фиксации защиты.
	m_Tros_KO6: BOOL;
	// Промежуточная катушка тросового выключателя КО-7 для фиксации защиты.
	m_Tros_KO7: BOOL;
	// Промежуточная катушка тросового выключателя конвейера на СМК516 для фиксации защиты.
	m_Tros_KonvSMK516: BOOL;
	// Промежуточная катушка тросового выключателя ленты на УСМ40 для фиксации защиты.
	m_TrosLentaUSM40: BOOL;
	// Промежуточная катушка тросового выключателя КО-11 для фиксации защиты.
	m_Tros_KO11: BOOL;
	// Промежуточная катушка тепловой защиты КО-1 для фиксации и квитирования.
	m_TZ_KO1: BOOL;
	// Промежуточная катушка тепловой защиты КО-2 для фиксации и квитирования.
	m_TZ_KO2: BOOL;
	// Промежуточная катушка тепловой защиты КО-3 для фиксации и квитирования.
	m_TZ_KO3: BOOL;
	// Промежуточная катушка тепловой защиты КО-4 для фиксации и квитирования.
	m_TZ_KO4: BOOL;
	// Промежуточная катушка тепловой защиты КО-6 для фиксации и квитирования.
	m_TZ_KO6: BOOL;
	// Промежуточная катушка тепловой защиты КО-7 для фиксации и квитирования.
	m_TZ_KO7: BOOL;
	// Промежуточная катушка тепловой защиты конвейера на СМК516 для фиксации и квитирования.
	m_TZ_KonvSMK516: BOOL;
	// Промежуточная катушка тепловой защиты КО-11 для фиксации и квитирования.
	m_TZ_KO11: BOOL;
	// Сброс звонка.
	SbrosZvonka_HMI: BOOL;
	// Маркер звонка при защитах.
	mZV3: BOOL;
	// Триггер звонков при срабатывании защит.
	RS_Zv_Avar: RS;
	// Все маркеры тросовых защит для останова линии по любому из тросовых выключателей.
	m_Tros_All: BOOL;
	// Пуск "Привода"
	Pusk_HMI_Privoda: BOOL;
	// Маркер для "Пуск привода". Взводит таймеры для поочередного включения приводов.
	m_Pusk_Privoda: BOOL;
	// Маркер общих защит приводов.
	m_Avar_Priv: BOOL;
	// Задержка перед включением PL250.
	TON_PL250: TON;
	// Задержка перед пуском 45 кВт на СМК516.
	TON_SMK516_45: TON;
	// Задержка перед пуском 37 кВт на СМК516.
	TON_SMK516_37: TON;
	// Задержка перед пуском 37 кВт на СМК517.
	TON_SMK517_37: TON;
	// Задержка перед запуском 5 кВт на СМК517.
	TON_SMK_517_5: TON;
	// Пуск "Линия"
	Pusk_HMI_Liniya: BOOL;
	// Маркер для "Пуск Линия". Взводит таймеры для поочередного включения конвейеров.
	m_Pusk_Liniya: BOOL;
	// Задержка перед включение КО-7.
	TON_KO7: TON;
	// Задержка перед включение УСМ40 по "Пуск линия".
	TON_USM40_Lin: TON;
	// Задержка перед включением КО-6.
	TON_KO6: TON;
	// Задержка перед включением КО-4.
	TON_KO4: TON;
	// Задержка перед включением разравнивателя на СМК516 по "Пуск линия".
	TON_RazrSMK516: TON;
	// Задержка перед включением конвейера на СМК516 по "Пуск линия".
	TON_KonvSMK516: TON;
	// Задержка перед включением КО-3.
	TON_KO3: TON;
	// Задержка перед включением КО-2.
	TON_KO2: TON;
	// Задержка перед включением КО-1.
	TON_KO1: TON;
	// Задержка перед включением PL024.
	TON_PL024: TON;
	// Задержка перед включением PL012.
	TON_PL012: TON;	
	// Маркер пуск КО-1 в ручном режиме.
	mh_Pusk_KO1: BOOL;
	// Маркер пуск КО-2 в ручном режиме.
	mh_Pusk_KO2: BOOL;
	// Маркер пуск КО-3 в ручном режиме.
	mh_Pusk_KO3: BOOL;
	// Маркер пуск КО-4 в ручном режиме.
	mh_Pusk_KO4: BOOL;
	// Маркер пуск КО-6 в ручном режиме.
	mh_Pusk_KO6: BOOL;
	// Маркер пуск КО-7 в ручном режиме.
	mh_Pusk_KO7: BOOL;
	//Маркер пуск КО-11 в ручном режиме.
	mh_Pusk_KO11: BOOL;
	// Маркер пуск питателя PL024 в ручном режиме.
	mh_Pusk_PL024: BOOL;
	// Маркер пуск питателя PL012 в ручном режиме.
	mh_Pusk_PL012: BOOL;
	// Маркер пуск электромагнита ЭП80 на КО-2 в ручном режиме.
	mh_Pusk_EP80_1: BOOL;
	// Маркер пуск 37 кВт на СМК 517 в ручном режиме.
	mh_Pusk_SMK517_37: BOOL;
	// Маркер пуск 5,5 кВт на СМК 517 в ручном режиме.
	mh_Pusk_SMK517_5: BOOL;
	// Маркер пуск 45 кВт на СМК 516 в ручном режиме.
	mh_Pusk_SMK516_45: BOOL;
	// Маркер пуск 37 кВт на СМК516 в ручном режиме.
	mh_Pusk_SMK516_37: BOOL;
	// Маркер пуск разравниватель на СМК516 в ручном режиме.
	mh_Pusk_RazrSMK516: BOOL;
	// Маркер пуск конвейер на СМК516 в ручном режиме.
	mh_Pusk_KonvSMK516: BOOL;
	// Маркер пуск смеситель PL250 в ручном режиме.
	mh_Pusk_PL250: BOOL;
	// Маркер пуск вода на PL250 в ручном режиме.
	mh_Pusk_VodaPL250: BOOL;
	// Маркер пуск электромагнита ЭП80 на КО-6 в ручном режиме.
	mh_Pusk_EP80_2: BOOL;
	// Маркер пуск привода для УСМ40 в ручном режиме.
	mh_PuskPrivUSM40: BOOL;
	// Маркер пуск линия для УСМ40 в ручном режиме.
	mh_PuskLinUSM40: BOOL;
	// Маркер пуск питателя ПЛ1-10 №1 в ручном режиме.
	mh_Pusk_Pl1: BOOL;
	// Маркер пуск питателя ПЛ1-10 №2 в ручном режиме.
	mh_Pusk_PL2: BOOL;
	// Маркер пуск 5,5 кВт для СМК517 в реверс в ручном режиме.
	mh_Pusk_SMK517_5_rev: BOOL;
	// Маркер пуск КО-1 в автоматическом режиме.
	ma_Pusk_KO1: BOOL;
	// Маркер пуск привода для УСМ40 в автоматическом режиме.
	ma_Pusk_PrivodaUSM40: BOOL;
	// Маркер пуск PL250 в автоматическом режиме.
	ma_Pusk_PL250: BOOL;
	// Маркер пуск 45 кВт для СМК516 в автоматическом режиме.
	ma_Pusk_SMK516_45: BOOL;
	// Маркер включение воды в питатель PL250 в автоматическом режиме.
	ma_Pusk_VodaPL250: BOOL;
	// Маркер пуск 37 кВт для СМК516 в автоматическом режиме.
	ma_Pusk_SMK516_37: BOOL;
	// Маркер пуск 37 кВт для СМК517 в автоматическом режиме.
	ma_Pusk_SMK517_37: BOOL;
	// Маркер пуск 5,5 кВт для СМК517 в автоматическом режиме.
	ma_Pusk_SMK517_5: BOOL;
	// Маркер пуск ЭП80 на КО-2 в автоматическом режиме.
	ma_Pusk_EP80_1: BOOL;
	// Маркер пуск ЭП80 на КО-6 в автоматическом режиме.
	ma_Pusk_EP80_2: BOOL;
	// Маркер пуск КО-7 в автоматическом режиме.
	ma_Pusk_KO7: BOOL;
	// Маркер пуск линия для УСМ40 в автоматическом режиме.
	ma_Pusk_LiniyaUSM40: BOOL;
	// Маркер пуск КО-6 в автоматическом режиме.
	ma_Pusk_KO6: BOOL;
	// Маркер пуск КО-4 в автоматическом режиме.
	ma_Pusk_KO4: BOOL;
	// Маркер пуск разравниватель на СМК516 в автоматическом режиме.
	ma_Pusk_RazrSMK516: BOOL;
	// Маркер пуск конвейер на СМК516 в автоматическом режиме.
	ma_Pusk_KonvSMK516: BOOL;
	// Маркер пуск КО-3 в автоматическом режиме.
	ma_Pusk_KO3: BOOL;
	// Маркер пуск КО-2 в автоматическом режиме.
	ma_Pusk_KO2: BOOL;
	// Маркер пуск PL012 в автоматическом режиме.
	ma_Pusk_PL012: BOOL;
	// Маркер пуск PL024 в автоматическом режиме.
	ma_Pusk_PL024: BOOL;
	// Задержка перед включением ПЛ1-10 №1.
	TON_PL1: TON;
	// Маркер пуск ПЛ1-10 №1 в автоматическом режиме.
	ma_Pusk_Pl1: BOOL;
	// Задержка перед включением ПЛ1-10 №2.
	TON_PL2: TON;
	// Маркер пуск ПЛ1-10 №2 в автоматическом режиме.
	ma_Pusk_PL2: BOOL;
	// Маркер пуск КО-11 в автоматическом режиме.
	ma_Pusk_KO11: BOOL;
	// Промежуточный маркер защиты PL024 для квитирования.
	m_Avar_PL024: BOOL;
	// Промежуточный маркер защиты PL012 для квитирования.
	m_Avar_PL012: BOOL;
	// Промежуточный маркер тепловой защиты ЭП80 на КО-2 для квитирования.
	m_TZ_EP80_1: BOOL;
	// Промежуточный маркер тепловой защиты 37 кВт на СМК517 для квитирования.
	m_TZ_SMK517_37: BOOL;
	// Промежуточный маркер тепловой защиты 5,5 кВт на СМК517 для квитирования.
	m_TZ_SMK517_5: BOOL;
	// Промежуточный маркер защиты ATS на СМК517 для квитирования.
	m_Avar_SMK517_ATS: BOOL;
	// Промежуточный маркер тепловой защиты 45 кВт на СМК516 для квитирования.
	m_TZ_SMK516_45: BOOL;
	// Промежуточный маркер тепловой защиты 37 кВт на СМК516 для квитирования.
	m_TZ_SMK516_37: BOOL;
	// Промежуточный маркер тепловой защиты разравнивателя на СМК516 для квитирования.
	m_TZ_RazrSMK516: BOOL;
	// Промежуточный маркер защиты PL250 для квитирования.
	m_Avar_PL250: BOOL;
	// Промежуточный маркер тепловой защиты ЭП80 на КО-6 для квитирования.
	m_TZ_EP80_2: BOOL;
	// Промежуточный маркер защиты УСМ40 для квитирования.
	m_Avar_USM40: BOOL;
	// Промежуточный маркер тепловой защиты питателя ПЛ1-10 №1 для квитирования.
	m_TZ_PL1: BOOL;
	// Промежуточный маркер тепловой защиты питателя ПЛ1-10 №2 для квитирования.
	m_TZ_PL2: BOOL;
	// Маркер общей защиты линии.
	m_Avar_Lin: BOOL;
	// Маркер пуск контактора СМК517 5,5 кВт прямо в ручном режиме.
	mh_SMK517_Prjamo: BOOL;
	// Маркер пуск контактора СМК517 5,5 кВт в реверс в ручном режиме.
	mh_SMK517_Revers: BOOL;
	// Маркер пуск контактора СМК517 5,5 кВт прямо в автоматическом режиме.
	ma_SMK517_Prjamo: BOOL;
	// Маркер датчика кожуха на СМК516 для квитирования.
	m_Kozhuh_SMK516: BOOL;
	// Маркер отхода валков на СМК516 для квитирования.
	m_Othod_SMK516: BOOL;
	// Маркер датчика кожуха СМК517 для квитирования.
	m_Kozhuh_SMK517: BOOL;
	// Маркер отхода валков на СМК517 для квитирования.
	m_Othod_SMK517: BOOL;
	// Маркер пуск ATS на СМК517 в реверс для проточки.
	mp_Pusk_SMK517_5_rev: BOOL;
	// Маркер пуск контактора 5,5 кВт на  СМК517 в реверс для проточки.
	mp_SMK517_Revers: BOOL;
	// Маркер пуска 5,5 кВт на СМК517 для проточки.
	m_Vkl_Protoch517: BOOL;
	// Команда из HMI на подготовку УСМ40.
	Pusk_HMI_PodgotUSM40: BOOL;
	// Блок частотника PL012.
	fbATVPL012: ALTIVAR31_CONTROL;
	// Перевод в RUN частотника на PL012 при ручном рецепте.
	m_RunATVPL012: BOOL;
	// Перевод в RUN частотника на PL012 при рецепте 1.
	m_RunATVPL012_R1: BOOL;
	// Перевод в RUN частотника на PL012 при рецепте 2.
	m_RunATVPL012_R2: BOOL;
	// Перевод в RUN частотника на PL012 при рецепте 3.
	m_RunATVPL012_R3: BOOL;
	// Перевод в RUN частотника на PL012 при рецепте 4.
	m_RunATVPL012_R4: BOOL;
	// Ошибка от ПЧ PL012.
	m_AvarATVPL012: BOOL;
	// Текущая частота ПЧ на PL012.
	m_ATVPL012_OutFrec: INT;
	// Текущий выходной ток ПЧ на PL012.
	m_ATVPL012_OutCur: INT;
	// Задание частоты ПЧ на PL012 при ручном рецепте.
	m_HMI_WriteFrecPL012: INT := 500;
	// Задание частоты ПЧ на PL012 при рецепте 1.
	m_HMI_WriteFrecPL012_R1: INT;
	// Задание частоты ПЧ на PL012 при рецепте 2.
	m_HMI_WriteFrecPL012_R2: INT;	
	// Задание частоты ПЧ на PL012 при рецепте 3.
	m_HMI_WriteFrecPL012_R3: INT;	
	// Задание частоты ПЧ на PL012 при рецепте 4.
	m_HMI_WriteFrecPL012_R4: INT;	
	// Блок чатотника PL024.
	fbATVPL024: ALTIVAR31_CONTROL;
	// Перевод в RUN частотника на PL024 при ручном рецепте.
	m_RunATVPL024: BOOL;
	// Перевод в RUN частотника на PL024 при рецепте 1.
	m_RunATVPL024_R1: BOOL;
	// Перевод в RUN частотника на PL024 при рецепте 2.
	m_RunATVPL024_R2: BOOL;
	// Перевод в RUN частотника на PL024 при рецепте 3.
	m_RunATVPL024_R3: BOOL;
	// Перевод в RUN частотника на PL024 при рецепте 4.
	m_RunATVPL024_R4: BOOL;
	// Ошибка от ПЧ PL024.
	m_AvarATVPL024: BOOL;
	// Текущая частота ПЧ на PL024.
	m_ATVPL024_OutFrec: INT;
	// Текущий выходной ток ПЧ на PL024.
	m_ATVPL024_OutCur: INT;
	// Задание частоты ПЧ на PL024 при ручном рецепте.
	m_HMI_WriteFrecPL024: INT := 500;
	// Задание частоты ПЧ на PL024 при рецепте 1.
	m_HMI_WriteFrecPL024_R1: INT;
	// Задание частоты ПЧ на PL024 при рецепте 2.
	m_HMI_WriteFrecPL024_R2: INT;
	// Задание частоты ПЧ на PL024 при рецепте 3.
	m_HMI_WriteFrecPL024_R3: INT;
	// Задание частоты ПЧ на PL024 при рецепте 4.
	m_HMI_WriteFrecPL024_R4: INT;
	// Блок частотника на ПЛ1-10_!.
	fbATVPL1: ALTIVAR31_CONTROL;
	// Перевод в RUN частотника на ПЛ1-10_1 при ручном рецепте.
	m_RunATVPL1: BOOL;
	// Перевод в RUN частотника на ПЛ1-10_1 при рецепте 1.
	m_RunATVPL1_R1: BOOL;
	// Перевод в RUN частотника на ПЛ1-10_1 при рецепте 2.
	m_RunATVPL1_R2: BOOL;
	// Перевод в RUN частотника на ПЛ1-10_1 при рецепте 3.
	m_RunATVPL1_R3: BOOL;
	// Перевод в RUN частотника на ПЛ1-10_1 при рецепте 4.
	m_RunATVPL1_R4: BOOL;
	// Ошибка от ПЧ ПЛ1-10_1.
	m_AvarATVPL1: BOOL;
	// Текущая частота ПЧ на ПЛ1-10_1.
	m_ATVPL1OutFrec: INT;
	// Текущий выходной ток ПЧ на ПЛ1-10_1.
	m_ATVPL1_OutCur: INT;
	// Задание частоты ПЧ на ПЛ1-10_1 при ручном рецепте.
	m_HMI_WriteFrecPL1: INT := 500;
	// Задание частоты ПЧ на ПЛ1-10_1 при рецепте 1.
	m_HMI_WriteFrecPL1_R1: INT;
	// Задание частоты ПЧ на ПЛ1-10_1 при рецепте 2.
	m_HMI_WriteFrecPL1_R2: INT;
	// Задание частоты ПЧ на ПЛ1-10_1 при рецепте 3.
	m_HMI_WriteFrecPL1_R3: INT;
	// Задание частоты ПЧ на ПЛ1-10_1 при рецепте 4.
	m_HMI_WriteFrecPL1_R4: INT;
	// Блок частотника на ПЛ1-10_2.
	fbATVPL2: ALTIVAR31_CONTROL;
	// Перевод в RUN частотника на ПЛ1-10_2 при ручном рецепте.
	m_RunATVPL2: BOOL;
	// Перевод в RUN частотника на ПЛ1-10_2 при рецепте 1.
	m_RunATVPL2_R1: BOOL;
	// Перевод в RUN частотника на ПЛ1-10_2 при рецепте 2.
	m_RunATVPL2_R2: BOOL;
	// Перевод в RUN частотника на ПЛ1-10_2 при рецепте 3.
	m_RunATVPL2_R3: BOOL;
	// Перевод в RUN частотника на ПЛ1-10_2 при рецепте 4.
	m_RunATVPL2_R4: BOOL;
	// Ошибка от ПЧ ПЛ1-10_2.
	m_AvarATVPL2: BOOL;
	// Текущая частота ПЧ на ПЛ1-10_2.
	m_ATVPL2OutFrec: INT;
	// Текущий выходной ток ПЧ на ПЛ1-10_2.
	m_ATVPL2_OutCur: INT;
	// Задание частоты ПЧ на ПЛ1-10_2 при ручном рецепте.
	m_HMI_WriteFrecPL2: INT := 500;
	// Задание частоты ПЧ на ПЛ1-10_2 при рецепте 1.
	m_HMI_WriteFrecPL2_R1: INT;
	// Задание частоты ПЧ на ПЛ1-10_2 при рецепте 2.
	m_HMI_WriteFrecPL2_R2: INT;
	// Задание частоты ПЧ на ПЛ1-10_2 при рецепте 3.
	m_HMI_WriteFrecPL2_R3: INT;
	// Задание частоты ПЧ на ПЛ1-10_2 при рецепте 4.
	m_HMI_WriteFrecPL2_R4: INT;
	// Блок частотника на PL250.
	fbATVPL250: ALTIVAR31_CONTROL;
	// Ошибка от ПЧ PL250.
	m_AvarATVPL250: BOOL;
	// Текущая частота ПЧ на PL250.
	m_ATVPL250OutFrec: INT;
	// Текущий выходной ток ПЧ на PL250.
	m_ATVPL250_OutCur: INT;
	// Задание частоты ПЧ на PL250.
	m_HMI_WriteFrecPL250: INT := 500;
	// Блок частотника на УСМ40.
	fbATVUSM40: ALTIVAR31_CONTROL;
	// Ошибка от ПЧ УСМ40.
	m_AvarATVUSM40: BOOL;
	// Текущая частота на ПЧ УСМ40.
	m_ATVUSM40OutFrec: INT;
	// Текущий выходной ток ПЧ на УСМ40.
	m_ATVUSM40_OutCur: INT;
	// Задание частоты ПЧ на УСМ40.
	m_HMI_WriteFrecUSM40: INT := 500;
	// Блок частотника на разравнивателе СМК516.
	fbATVRazrSMK516: ALTIVAR31_CONTROL;
	// Ошибка от ПЧ разравнивателя на СМК516.
	m_AvarATVRazrSMK516: BOOL;
	// Текущая частота ПЧ на разравнивателе СМК516.
	m_ATVRazrSMK516OutFrec: INT;
	// Текущий выходной ток ПЧ на разравнивателе СМК516.
	m_ATVRazrSMK516_OutCur: INT;
	// Задание частоты ПЧ на разравнивателе СМК516.
	m_HMI_WriteFrecRazrSMK516: INT := 500;
	// Перевод в RUN всех ПЧ в ручном режиме.
	m_RunATVAll: BOOL;
	// Задержка перед выключением конвейера УСМ40.
	TOF_USM40_Lin: TOF;
	// Задержка перед выключением конвейера на СМК516.
	TOF_SMK516_Konv: TOF;
	// Задержка перед выключением разравнивателя на СМК516.
	TOF_SMK516_Razr: TOF;
	// Текущий уровень в PL024У переведенный в %.
	Uroven0100_PL024U AT %MW21: INT;
	// Задание максимально допустимого уровня в PL024У.
	TargMaxUrovenPL024U: INT := 90;
	// Маркер достижения максимального уровня в PL024У.
	m_MaxUrovenPL024U: BOOL;
	// Задание минимально допустимого уровня в PL024У.
	TargMinUrovenPL024U: INT := 10;
	// Маркер уровня меньше максимального в PL024У.
	m_MinUrovenPL024U: BOOL;
	// Маркер уровня в питателе. Дает разрешение на включение линии.
	m_UrovenPL024U: BOOL;	
	// RS-триггер уровня.
	RS_Uroven: RS;
	// Задержка перед выключением КО-1 при "Стоп линия автомат".
	TOF_KO1: TOF;
	// Задержка перед выключением КО-11 при "Стоп линия автомат".
	TOF_KO11: TOF;
	// Задержка перед выключением КО-2 при "Стоп линия автомат".
	TOF_KO2: TOF;
	// Стоп линия автомат из панели.
	StopHMILinAvt: BOOL;
	// Задержка перед выключением КО-3 при "Стоп линия автомат".
	TOF_KO3: TOF;
	// Задержка перед выключением  конвейера на СМК516 при "Стоп линия автомат".
	TOF_KonvSMK516: TOF;
	// Задержка перед выключением КО-4 при "Стоп линия автомат".
	TOF_KO4: TOF;
	// Задержка перед выключением КО-7 при "Стоп линия автомат".
	TOF_KO7: TOF;
	// Задержка перед выключением конвейера на УСМ40 при "Стоп линия автомат".
	TOF_LiniyaUSM40: TOF;
	// Задержка перед выключением КО-6 при "Стоп линия автомат".
	TOF_KO6: TOF;
	// Время задержки перед включением СМК516 45 кВт.
	t_ON_SMK516_45: TIME := TIME#15MS;
	// Время задержки перед включением СМК516 37 кВт.
	t_ON_SMK516_37: TIME := TIME#25MS;
	// Время задержки перед включением СМК517 37 кВт.
	t_ON_SMK517_37: TIME := TIME#35MS;
	// Время задержки перед включением СМК516 5,5 кВт.
	t_ON_SMK517_5: TIME := TIME#45MS;
	// Время задержки перед включением КО-6.
	t_ON_KO6: TIME := TIME#2ms;
	// Время задержки перед включением линии на УСМ40.
	t_ON_USM40Lin: TIME := TIME#0MS;
	// Время задержки перед включением КО-7.
	t_ON_KO7: TIME := TIME#17MS;
	// Время задержки перед включением PL250.
	t_ON_PL250: TIME := TIME#18MS;
	// Время задержки перед включением КО-4.
	t_ON_KO4: TIME := TIME#28MS;
	// Время задержки перед включением разравнивателя на СМК516.
	t_ON_RazrSMK516: TIME := TIME#29MS;
	// Время задержки перед включением конвейера на СМК516.
	t_ON_KonvSMK516: TIME := TIME#30MS;
	// Время задержки перед включением КО-3.
	t_ON_KO3: TIME := TIME#31MS;
	// Время задержки перед включением КО-2.
	t_ON_KO2: TIME := TIME#32MS;
	// Время задержки перед включением КО-1 и КО-11.
	t_ON_KO1: TIME := TIME#33MS;
	// Время задержки перед включением питателей в приемном (PL012, PL024) отделении и на добавках (ПЛ1-10).
	t_ON_PL012: TIME := TIME#33ms;
	// Время задержки перед выключением КО-1 при Стоп Линия Автомат.
	t_OF_KO1: TIME := TIME#17ms;
	// Время задержки перед выключением КО-11 при Стоп Линия Автомат.
	t_OF_KO11: TIME := TIME#14ms;
	// Время задержки перед выключением КО-2 при Стоп Линия Автомат.
	t_OF_KO2: TIME := TIME#46MS;
	// Время задержки перед выключением КО-3 при Стоп Линия Автомат.
	t_OF_KO3: TIME := TIME#63ms;
	// Время задержки перед выключением конвейера на СМК516 при Стоп Линия Автомат.
	t_OF_KonvSMK516: TIME := TIME#66ms;
	// Время задержки перед выключением КО-4 при Стоп Линия Автомат.
	t_OF_KO4: TIME := TIME#78ms;
	// Время задержки перед выключением КО-7 при Стоп Линия Автомат.
	t_OF_KO7: TIME := TIME#99ms;
	// Время задержки перед выключением линии на УСМ40 при Стоп Линия Автомат.
	t_OF_LiniyaUSM40: TIME := TIME#102ms;
	// Время задержки перед выключением КО-6 при Стоп Линия Автомат.
	t_OF_KO6: TIME := TIME#124ms;	
	T1: TON;
	t2: TON;
	t3: TON;
	t_pl250: TON;
	t_usm40: TON;
	tl_usm40: TON;
END_VAR
VAR // added by the converter: edge detectors and wires of the graphical bodies
    _rt1, _rt2, _rt3, _rt4, _rt5, _rt6, _rt7, _rt8, _rt9, _rt10, _rt11, _rt12, _rt13, _rt14, _rt15, _rt16, _rt17, _rt18, _rt19, _rt20, _rt21, _rt22, _rt23, _rt24, _rt25, _rt26, _rt27, _rt28, _rt29, _rt30, _rt31, _rt32, _rt33, _rt34, _rt35, _rt36, _rt37, _rt38, _rt39, _rt40, _rt41, _rt42, _rt43, _rt44, _rt45, _rt46, _rt47, _rt48, _rt49, _rt50, _rt51, _rt52, _rt53, _rt54, _rt55, _rt56, _rt57, _rt58, _rt59, _rt60, _rt61, _rt62, _rt63, _rt64, _rt65, _rt66, _rt67, _rt68 : R_TRIG;
    _ft1, _ft2, _ft3 : F_TRIG;
    _w1, _w2, _w3, _w4, _w5, _w6, _w7, _w8 : BOOL;
END_VAR

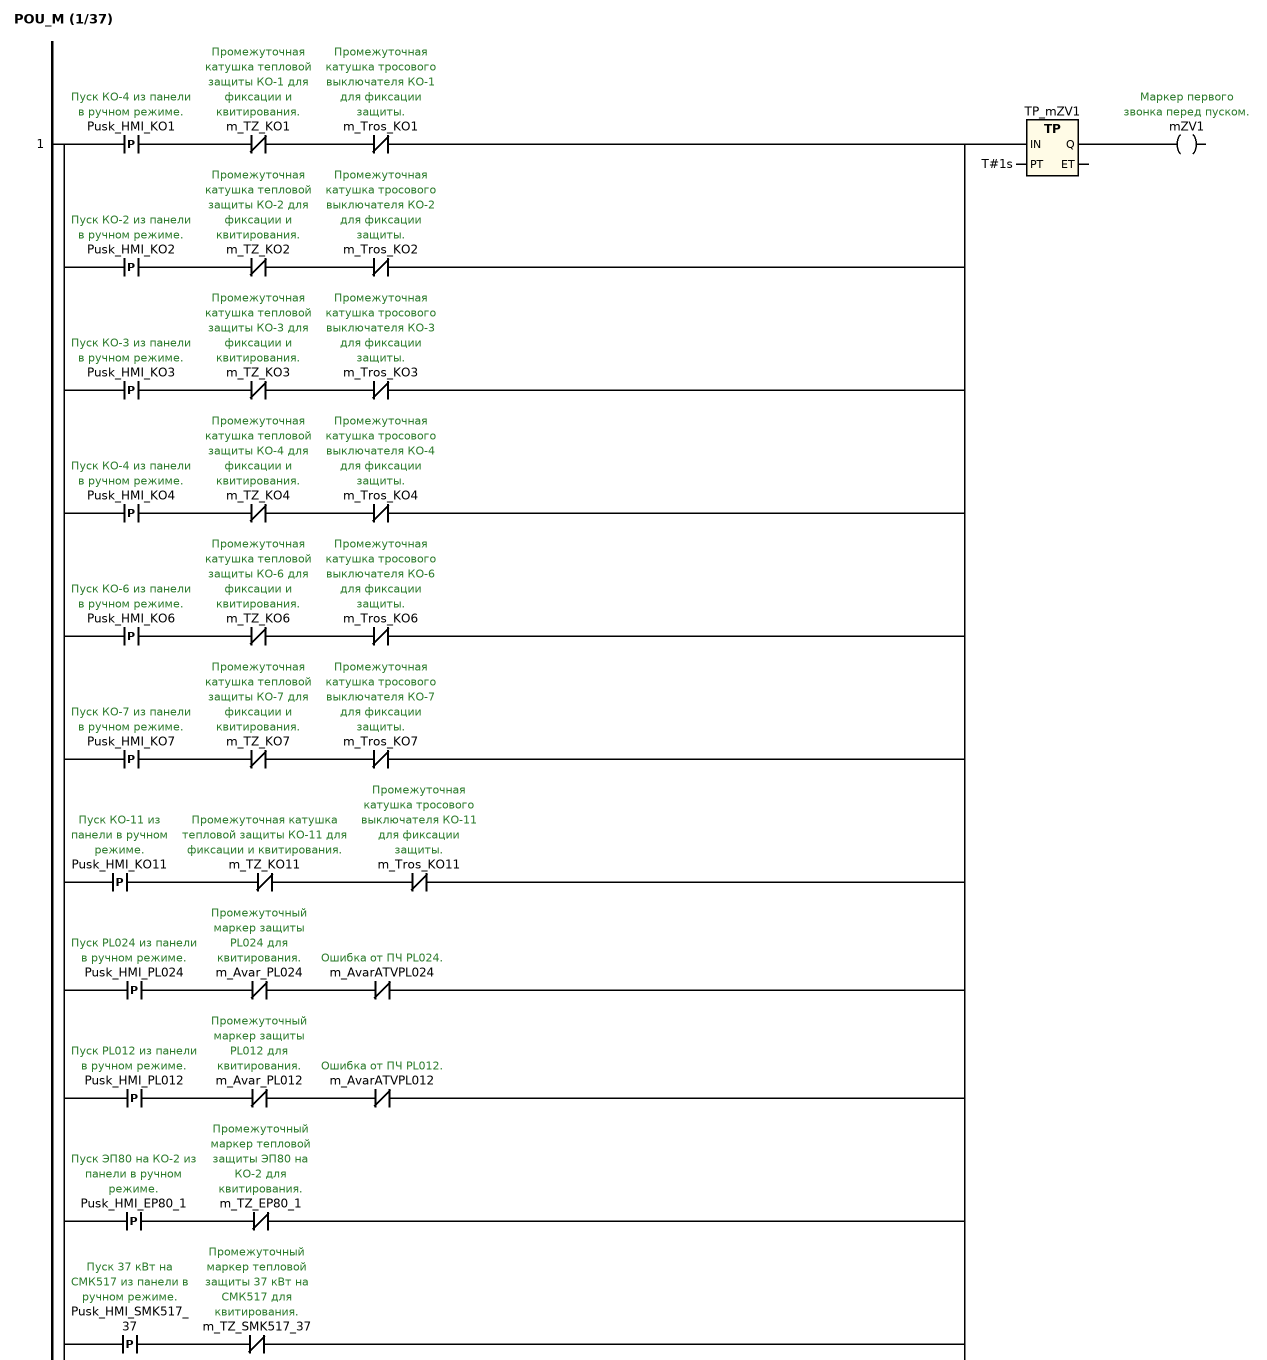
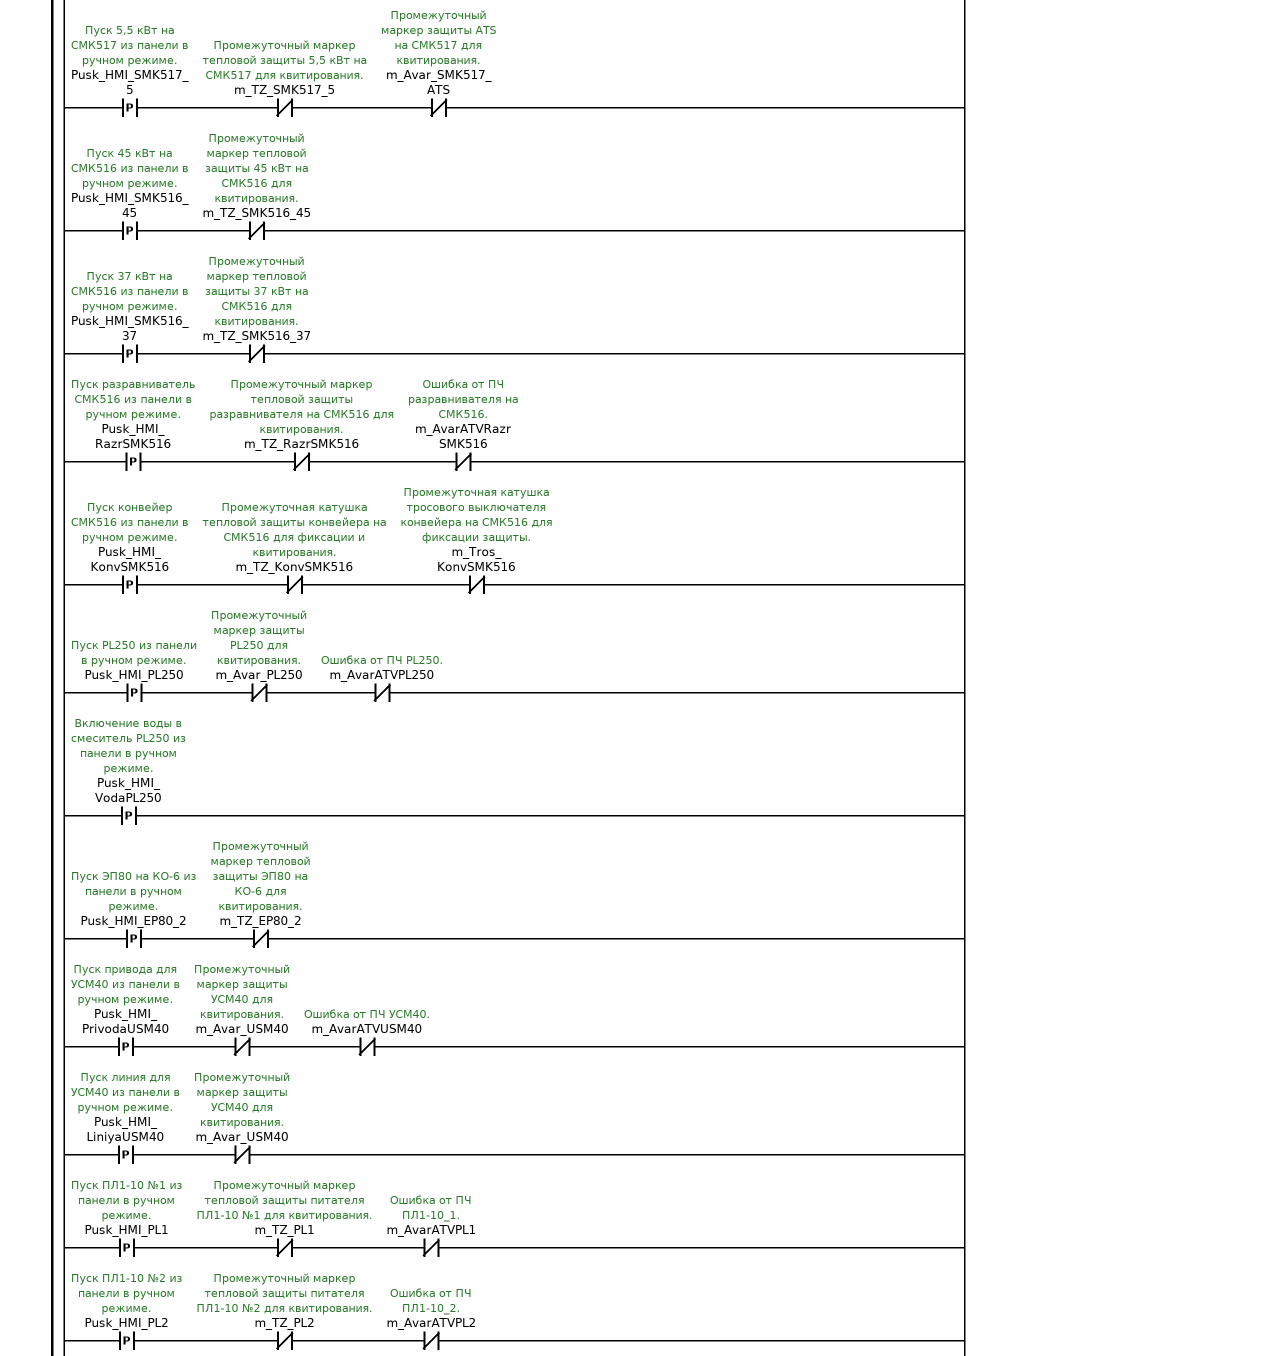
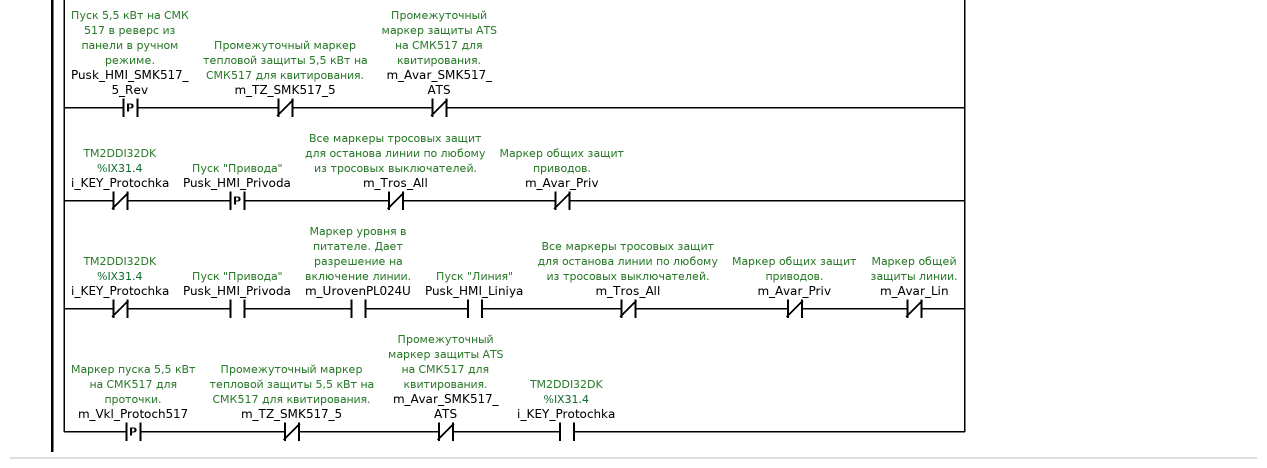
// NETWORK 1
//   Pusk_HMI_KO1: Пуск КО-4 из панели в ручном режиме.
//   m_TZ_KO1: Промежуточная катушка тепловой защиты КО-1 для фиксации и квитирования.
//   m_Tros_KO1: Промежуточная катушка тросового выключателя КО-1 для фиксации защиты.
//   Pusk_HMI_KO2: Пуск КО-2 из панели в ручном режиме.
//   m_TZ_KO2: Промежуточная катушка тепловой защиты КО-2 для фиксации и квитирования.
//   m_Tros_KO2: Промежуточная катушка тросового выключателя КО-2 для фиксации защиты.
//   Pusk_HMI_KO3: Пуск КО-3 из панели в ручном режиме.
//   m_TZ_KO3: Промежуточная катушка тепловой защиты КО-3 для фиксации и квитирования.
//   m_Tros_KO3: Промежуточная катушка тросового выключателя КО-3 для фиксации защиты.
//   Pusk_HMI_KO4: Пуск КО-4 из панели в ручном режиме.
//   m_TZ_KO4: Промежуточная катушка тепловой защиты КО-4 для фиксации и квитирования.
//   m_Tros_KO4: Промежуточная катушка тросового выключателя КО-4 для фиксации защиты.
//   Pusk_HMI_KO6: Пуск КО-6 из панели в ручном режиме.
//   m_TZ_KO6: Промежуточная катушка тепловой защиты КО-6 для фиксации и квитирования.
//   m_Tros_KO6: Промежуточная катушка тросового выключателя КО-6 для фиксации защиты.
//   Pusk_HMI_KO7: Пуск КО-7 из панели в ручном режиме.
//   m_TZ_KO7: Промежуточная катушка тепловой защиты КО-7 для фиксации и квитирования.
//   m_Tros_KO7: Промежуточная катушка тросового выключателя КО-7 для фиксации защиты.
//   Pusk_HMI_KO11: Пуск КО-11 из панели в ручном режиме.
//   m_TZ_KO11: Промежуточная катушка тепловой защиты КО-11 для фиксации и квитирования.
//   m_Tros_KO11: Промежуточная катушка тросового выключателя КО-11 для фиксации защиты.
//   Pusk_HMI_PL024: Пуск PL024 из панели в ручном режиме.
//   m_Avar_PL024: Промежуточный маркер защиты PL024 для квитирования.
//   m_AvarATVPL024: Ошибка от ПЧ PL024.
//   Pusk_HMI_PL012: Пуск PL012 из панели в ручном режиме.
//   m_Avar_PL012: Промежуточный маркер защиты PL012 для квитирования.
//   m_AvarATVPL012: Ошибка от ПЧ PL012.
//   Pusk_HMI_EP80_1: Пуск ЭП80 на КО-2 из панели в ручном режиме.
//   m_TZ_EP80_1: Промежуточный маркер тепловой защиты ЭП80 на КО-2 для квитирования.
//   Pusk_HMI_SMK517_37: Пуск 37 кВт на СМК517 из панели в ручном режиме.
//   m_TZ_SMK517_37: Промежуточный маркер тепловой защиты 37 кВт на СМК517 для квитирования.
//   Pusk_HMI_SMK517_5: Пуск 5,5 кВт на СМК517 из панели в ручном режиме.
//   m_TZ_SMK517_5: Промежуточный маркер тепловой защиты 5,5 кВт на СМК517 для квитирования.
//   m_Avar_SMK517_ATS: Промежуточный маркер защиты ATS на СМК517 для квитирования.
//   Pusk_HMI_SMK516_45: Пуск 45 кВт на СМК516 из панели в ручном режиме.
//   m_TZ_SMK516_45: Промежуточный маркер тепловой защиты 45 кВт на СМК516 для квитирования.
//   Pusk_HMI_SMK516_37: Пуск 37 кВт на СМК516 из панели в ручном режиме.
//   m_TZ_SMK516_37: Промежуточный маркер тепловой защиты 37 кВт на СМК516 для квитирования.
//   Pusk_HMI_RazrSMK516: Пуск разравниватель СМК516 из панели в ручном режиме.
//   m_TZ_RazrSMK516: Промежуточный маркер тепловой защиты разравнивателя на СМК516 для квитирования.
//   m_AvarATVRazrSMK516: Ошибка от ПЧ разравнивателя на СМК516.
//   Pusk_HMI_KonvSMK516: Пуск конвейер СМК516 из панели в ручном режиме.
//   m_TZ_KonvSMK516: Промежуточная катушка тепловой защиты конвейера на СМК516 для фиксации и квитирования.
//   m_Tros_KonvSMK516: Промежуточная катушка тросового выключателя конвейера на СМК516 для фиксации защиты.
//   Pusk_HMI_PL250: Пуск PL250 из панели в ручном режиме.
//   m_Avar_PL250: Промежуточный маркер защиты PL250 для квитирования.
//   m_AvarATVPL250: Ошибка от ПЧ PL250.
//   Pusk_HMI_VodaPL250: Включение воды в смеситель PL250 из панели в ручном режиме.
//   Pusk_HMI_EP80_2: Пуск ЭП80 на КО-6 из панели в ручном режиме.
//   m_TZ_EP80_2: Промежуточный маркер тепловой защиты ЭП80 на КО-6 для квитирования.
//   Pusk_HMI_PrivodaUSM40: Пуск привода для УСМ40 из панели в ручном режиме.
//   m_Avar_USM40: Промежуточный маркер защиты УСМ40 для квитирования.
//   m_AvarATVUSM40: Ошибка от ПЧ УСМ40.
//   Pusk_HMI_LiniyaUSM40: Пуск линия для УСМ40 из панели в ручном режиме.
//   Pusk_HMI_PL1: Пуск ПЛ1-10 №1 из панели в ручном режиме.
//   m_TZ_PL1: Промежуточный маркер тепловой защиты питателя ПЛ1-10 №1 для квитирования.
//   m_AvarATVPL1: Ошибка от ПЧ ПЛ1-10_1.
//   Pusk_HMI_PL2: Пуск ПЛ1-10 №2 из панели в ручном режиме.
//   m_TZ_PL2: Промежуточный маркер тепловой защиты питателя ПЛ1-10 №2 для квитирования.
//   m_AvarATVPL2: Ошибка от ПЧ ПЛ1-10_2.
//   Pusk_HMI_SMK517_5_Rev: Пуск 5,5 кВт на СМК 517 в реверс из панели в ручном режиме.
//   i_KEY_Protochka: TM2DDI32DK | AT %IX31.4
//   Pusk_HMI_Privoda: Пуск "Привода"
//   m_Tros_All: Все маркеры тросовых защит для останова линии по любому из тросовых выключателей.
//   m_Avar_Priv: Маркер общих защит приводов.
//   m_UrovenPL024U: Маркер уровня в питателе. Дает разрешение на включение линии.
//   Pusk_HMI_Liniya: Пуск "Линия"
//   m_Avar_Lin: Маркер общей защиты линии.
//   m_Vkl_Protoch517: Маркер пуска 5,5 кВт на СМК517 для проточки.
//   mZV1: Маркер первого звонка перед пуском.
_rt1(CLK := Pusk_HMI_KO1);
_rt2(CLK := Pusk_HMI_KO2);
_rt3(CLK := Pusk_HMI_KO3);
_rt4(CLK := Pusk_HMI_KO4);
_rt5(CLK := Pusk_HMI_KO6);
_rt6(CLK := Pusk_HMI_KO7);
_rt7(CLK := Pusk_HMI_KO11);
_rt8(CLK := Pusk_HMI_PL024);
_rt9(CLK := Pusk_HMI_PL012);
_rt10(CLK := Pusk_HMI_EP80_1);
_rt11(CLK := Pusk_HMI_SMK517_37);
_rt12(CLK := Pusk_HMI_SMK517_5);
_rt13(CLK := Pusk_HMI_SMK516_45);
_rt14(CLK := Pusk_HMI_SMK516_37);
_rt15(CLK := Pusk_HMI_RazrSMK516);
_rt16(CLK := Pusk_HMI_KonvSMK516);
_rt17(CLK := Pusk_HMI_PL250);
_rt18(CLK := Pusk_HMI_VodaPL250);
_rt19(CLK := Pusk_HMI_EP80_2);
_rt20(CLK := Pusk_HMI_PrivodaUSM40);
_rt21(CLK := Pusk_HMI_LiniyaUSM40);
_rt22(CLK := Pusk_HMI_PL1);
_rt23(CLK := Pusk_HMI_PL2);
_rt24(CLK := Pusk_HMI_SMK517_5_Rev);
_rt25(CLK := Pusk_HMI_Privoda);
_rt26(CLK := m_Vkl_Protoch517);
TP_mZV1(IN := _rt1.Q AND NOT m_TZ_KO1 AND NOT m_Tros_KO1 OR _rt2.Q AND NOT m_TZ_KO2 AND NOT m_Tros_KO2 OR _rt3.Q AND NOT m_TZ_KO3 AND NOT m_Tros_KO3 OR _rt4.Q AND NOT m_TZ_KO4 AND NOT m_Tros_KO4 OR _rt5.Q AND NOT m_TZ_KO6 AND NOT m_Tros_KO6 OR _rt6.Q AND NOT m_TZ_KO7 AND NOT m_Tros_KO7 OR _rt7.Q AND NOT m_TZ_KO11 AND NOT m_Tros_KO11 OR _rt8.Q AND NOT m_Avar_PL024 AND NOT m_AvarATVPL024 OR _rt9.Q AND NOT m_Avar_PL012 AND NOT m_AvarATVPL012 OR _rt10.Q AND NOT m_TZ_EP80_1 OR _rt11.Q AND NOT m_TZ_SMK517_37 OR _rt12.Q AND NOT m_TZ_SMK517_5 AND NOT m_Avar_SMK517_ATS OR _rt13.Q AND NOT m_TZ_SMK516_45 OR _rt14.Q AND NOT m_TZ_SMK516_37 OR _rt15.Q AND NOT m_TZ_RazrSMK516 AND NOT m_AvarATVRazrSMK516 OR _rt16.Q AND NOT m_TZ_KonvSMK516 AND NOT m_Tros_KonvSMK516 OR _rt17.Q AND NOT m_Avar_PL250 AND NOT m_AvarATVPL250 OR _rt18.Q OR _rt19.Q AND NOT m_TZ_EP80_2 OR _rt20.Q AND NOT m_Avar_USM40 AND NOT m_AvarATVUSM40 OR _rt21.Q AND NOT m_Avar_USM40 OR _rt22.Q AND NOT m_TZ_PL1 AND NOT m_AvarATVPL1 OR _rt23.Q AND NOT m_TZ_PL2 AND NOT m_AvarATVPL2 OR _rt24.Q AND NOT m_TZ_SMK517_5 AND NOT m_Avar_SMK517_ATS OR NOT i_KEY_Protochka AND _rt25.Q AND NOT m_Tros_All AND NOT m_Avar_Priv OR NOT i_KEY_Protochka AND Pusk_HMI_Privoda AND m_UrovenPL024U AND Pusk_HMI_Liniya AND NOT m_Tros_All AND NOT m_Avar_Priv AND NOT m_Avar_Lin OR _rt26.Q AND NOT m_TZ_SMK517_5 AND NOT m_Avar_SMK517_ATS AND i_KEY_Protochka, PT := T#1s); // TP
mZV1 := TP_mZV1.Q;

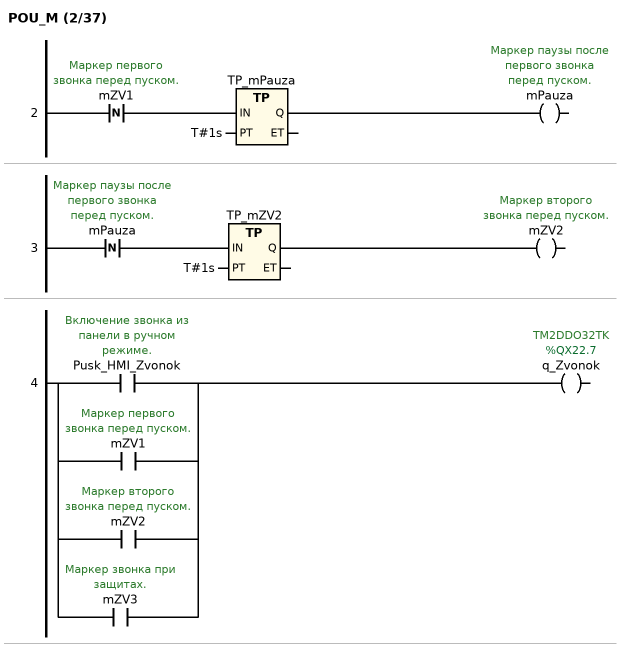
// NETWORK 2
//   mZV1: Маркер первого звонка перед пуском.
//   mPauza: Маркер паузы после первого звонка перед пуском.
_ft1(CLK := mZV1);
TP_mPauza(IN := _ft1.Q, PT := T#1s); // TP
mPauza := TP_mPauza.Q;

// NETWORK 3
//   mPauza: Маркер паузы после первого звонка перед пуском.
//   mZV2: Маркер второго звонка перед пуском.
_ft2(CLK := mPauza);
TP_mZV2(IN := _ft2.Q, PT := T#1s); // TP
mZV2 := TP_mZV2.Q;

// NETWORK 4
//   Pusk_HMI_Zvonok: Включение звонка из панели в ручном режиме.
//   mZV1: Маркер первого звонка перед пуском.
//   mZV2: Маркер второго звонка перед пуском.
//   mZV3: Маркер звонка при защитах.
//   q_Zvonok: TM2DDO32TK | AT %QX22.7
q_Zvonok := Pusk_HMI_Zvonok OR mZV1 OR mZV2 OR mZV3;

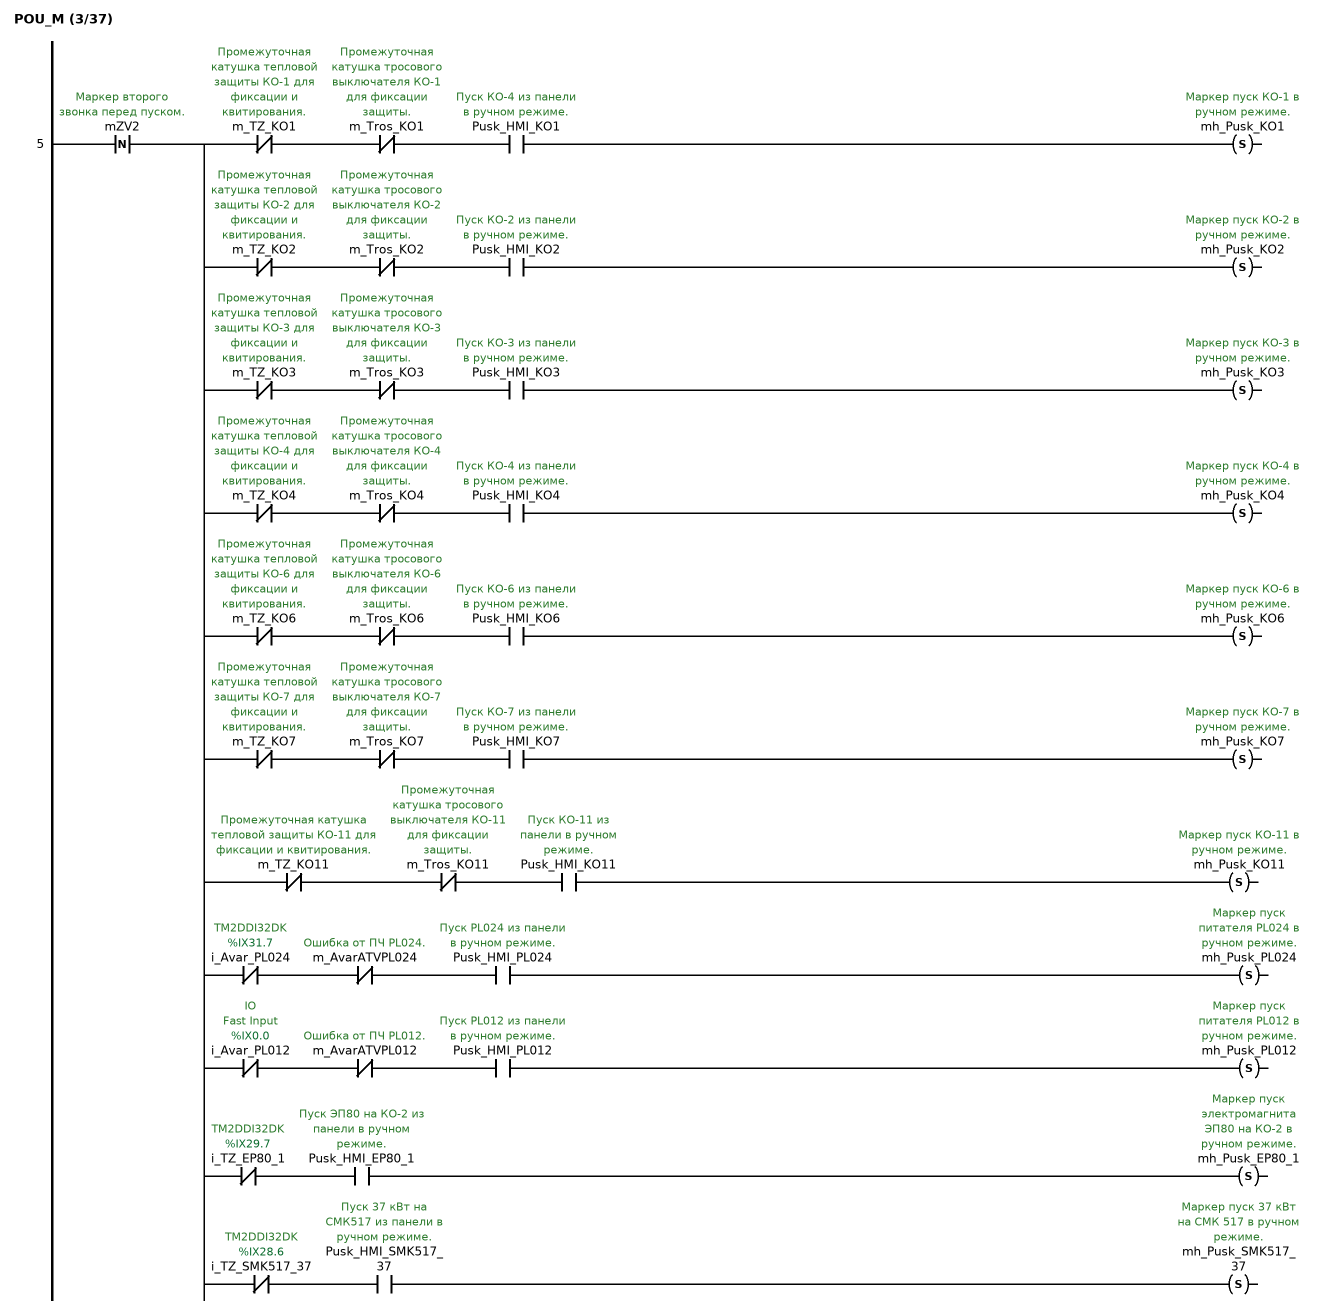
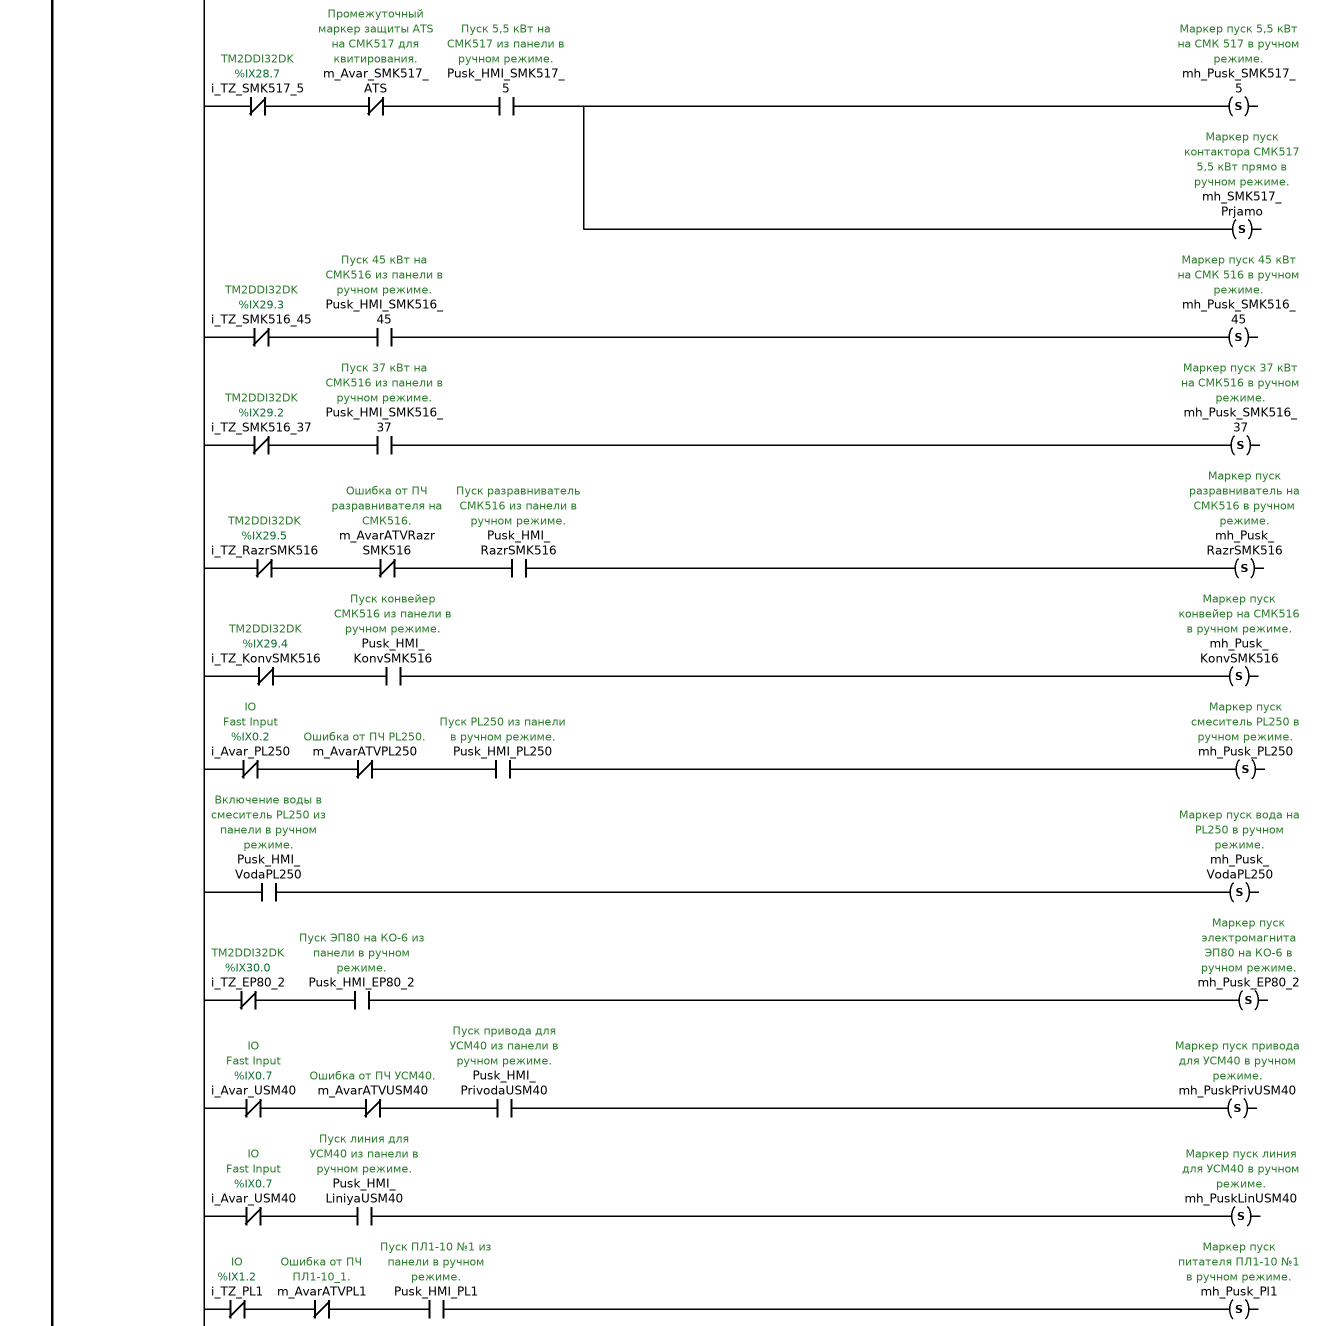
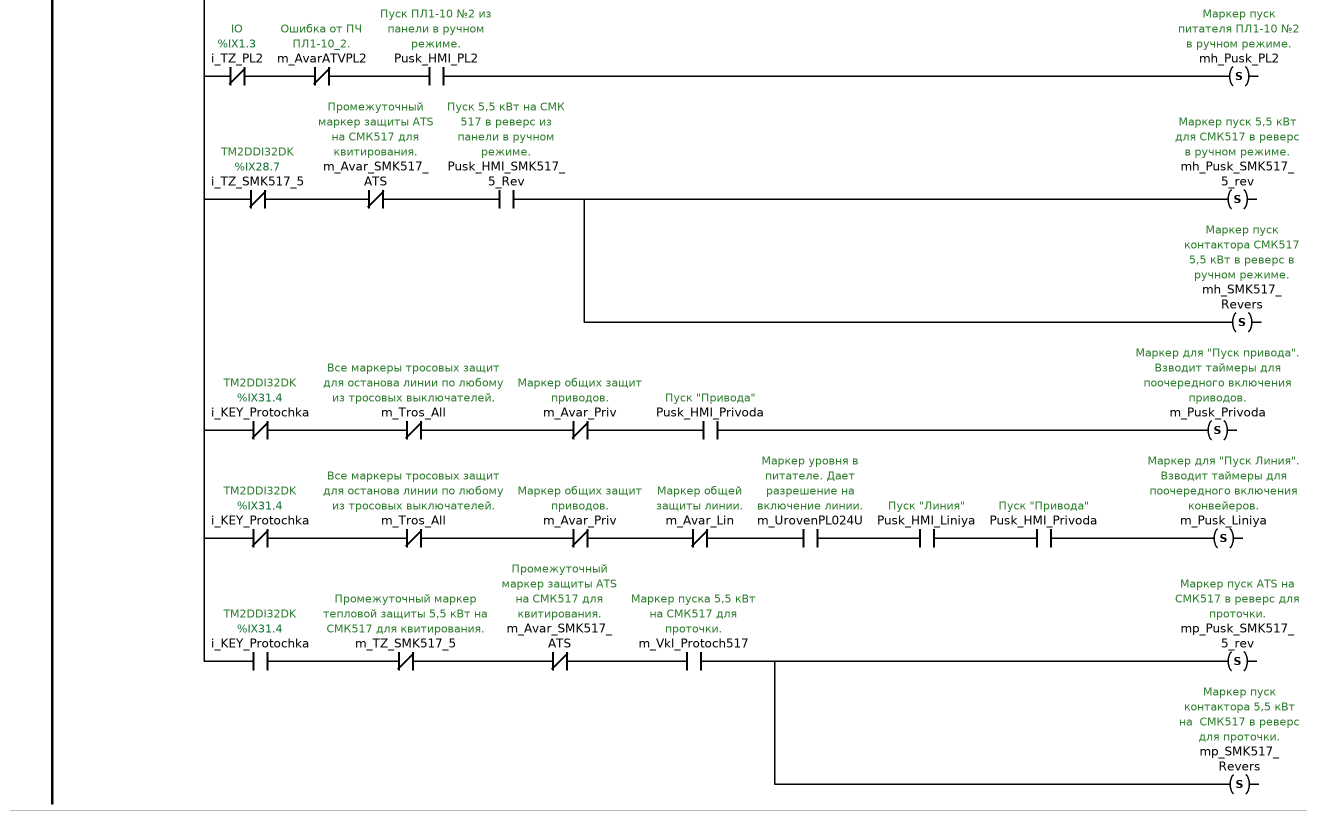
// NETWORK 5
//   mZV2: Маркер второго звонка перед пуском.
//   m_TZ_KO1: Промежуточная катушка тепловой защиты КО-1 для фиксации и квитирования.
//   m_Tros_KO1: Промежуточная катушка тросового выключателя КО-1 для фиксации защиты.
//   Pusk_HMI_KO1: Пуск КО-4 из панели в ручном режиме.
//   mh_Pusk_KO1: Маркер пуск КО-1 в ручном режиме.
//   m_TZ_KO2: Промежуточная катушка тепловой защиты КО-2 для фиксации и квитирования.
//   m_Tros_KO2: Промежуточная катушка тросового выключателя КО-2 для фиксации защиты.
//   Pusk_HMI_KO2: Пуск КО-2 из панели в ручном режиме.
//   mh_Pusk_KO2: Маркер пуск КО-2 в ручном режиме.
//   m_TZ_KO3: Промежуточная катушка тепловой защиты КО-3 для фиксации и квитирования.
//   m_Tros_KO3: Промежуточная катушка тросового выключателя КО-3 для фиксации защиты.
//   Pusk_HMI_KO3: Пуск КО-3 из панели в ручном режиме.
//   mh_Pusk_KO3: Маркер пуск КО-3 в ручном режиме.
//   m_TZ_KO4: Промежуточная катушка тепловой защиты КО-4 для фиксации и квитирования.
//   m_Tros_KO4: Промежуточная катушка тросового выключателя КО-4 для фиксации защиты.
//   Pusk_HMI_KO4: Пуск КО-4 из панели в ручном режиме.
//   mh_Pusk_KO4: Маркер пуск КО-4 в ручном режиме.
//   m_TZ_KO6: Промежуточная катушка тепловой защиты КО-6 для фиксации и квитирования.
//   m_Tros_KO6: Промежуточная катушка тросового выключателя КО-6 для фиксации защиты.
//   Pusk_HMI_KO6: Пуск КО-6 из панели в ручном режиме.
//   mh_Pusk_KO6: Маркер пуск КО-6 в ручном режиме.
//   m_TZ_KO7: Промежуточная катушка тепловой защиты КО-7 для фиксации и квитирования.
//   m_Tros_KO7: Промежуточная катушка тросового выключателя КО-7 для фиксации защиты.
//   Pusk_HMI_KO7: Пуск КО-7 из панели в ручном режиме.
//   mh_Pusk_KO7: Маркер пуск КО-7 в ручном режиме.
//   m_TZ_KO11: Промежуточная катушка тепловой защиты КО-11 для фиксации и квитирования.
//   m_Tros_KO11: Промежуточная катушка тросового выключателя КО-11 для фиксации защиты.
//   Pusk_HMI_KO11: Пуск КО-11 из панели в ручном режиме.
//   mh_Pusk_KO11: Маркер пуск КО-11 в ручном режиме.
//   i_Avar_PL024: TM2DDI32DK | AT %IX31.7
//   m_AvarATVPL024: Ошибка от ПЧ PL024.
//   Pusk_HMI_PL024: Пуск PL024 из панели в ручном режиме.
//   mh_Pusk_PL024: Маркер пуск питателя PL024 в ручном режиме.
//   i_Avar_PL012: IO Fast Input | AT %IX0.0
//   m_AvarATVPL012: Ошибка от ПЧ PL012.
//   Pusk_HMI_PL012: Пуск PL012 из панели в ручном режиме.
//   mh_Pusk_PL012: Маркер пуск питателя PL012 в ручном режиме.
//   i_TZ_EP80_1: TM2DDI32DK | AT %IX29.7
//   Pusk_HMI_EP80_1: Пуск ЭП80 на КО-2 из панели в ручном режиме.
//   mh_Pusk_EP80_1: Маркер пуск электромагнита ЭП80 на КО-2 в ручном режиме.
//   i_TZ_SMK517_37: TM2DDI32DK | AT %IX28.6
//   Pusk_HMI_SMK517_37: Пуск 37 кВт на СМК517 из панели в ручном режиме.
//   mh_Pusk_SMK517_37: Маркер пуск 37 кВт на СМК 517 в ручном режиме.
//   i_TZ_SMK517_5: TM2DDI32DK | AT %IX28.7
//   m_Avar_SMK517_ATS: Промежуточный маркер защиты ATS на СМК517 для квитирования.
//   Pusk_HMI_SMK517_5: Пуск 5,5 кВт на СМК517 из панели в ручном режиме.
//   mh_Pusk_SMK517_5: Маркер пуск 5,5 кВт на СМК 517 в ручном режиме.
//   mh_SMK517_Prjamo: Маркер пуск контактора СМК517 5,5 кВт прямо в ручном режиме.
//   i_TZ_SMK516_45: TM2DDI32DK | AT %IX29.3
//   Pusk_HMI_SMK516_45: Пуск 45 кВт на СМК516 из панели в ручном режиме.
//   mh_Pusk_SMK516_45: Маркер пуск 45 кВт на СМК 516 в ручном режиме.
//   i_TZ_SMK516_37: TM2DDI32DK | AT %IX29.2
//   Pusk_HMI_SMK516_37: Пуск 37 кВт на СМК516 из панели в ручном режиме.
//   mh_Pusk_SMK516_37: Маркер пуск 37 кВт на СМК516 в ручном режиме.
//   i_TZ_RazrSMK516: TM2DDI32DK | AT %IX29.5
//   m_AvarATVRazrSMK516: Ошибка от ПЧ разравнивателя на СМК516.
//   Pusk_HMI_RazrSMK516: Пуск разравниватель СМК516 из панели в ручном режиме.
//   mh_Pusk_RazrSMK516: Маркер пуск разравниватель на СМК516 в ручном режиме.
//   i_TZ_KonvSMK516: TM2DDI32DK | AT %IX29.4
//   Pusk_HMI_KonvSMK516: Пуск конвейер СМК516 из панели в ручном режиме.
//   mh_Pusk_KonvSMK516: Маркер пуск конвейер на СМК516 в ручном режиме.
//   i_Avar_PL250: IO Fast Input | AT %IX0.2
//   m_AvarATVPL250: Ошибка от ПЧ PL250.
//   Pusk_HMI_PL250: Пуск PL250 из панели в ручном режиме.
//   mh_Pusk_PL250: Маркер пуск смеситель PL250 в ручном режиме.
//   Pusk_HMI_VodaPL250: Включение воды в смеситель PL250 из панели в ручном режиме.
//   mh_Pusk_VodaPL250: Маркер пуск вода на PL250 в ручном режиме.
//   i_TZ_EP80_2: TM2DDI32DK | AT %IX30.0
//   Pusk_HMI_EP80_2: Пуск ЭП80 на КО-6 из панели в ручном режиме.
//   mh_Pusk_EP80_2: Маркер пуск электромагнита ЭП80 на КО-6 в ручном режиме.
//   i_Avar_USM40: IO Fast Input | AT %IX0.7
//   m_AvarATVUSM40: Ошибка от ПЧ УСМ40.
//   Pusk_HMI_PrivodaUSM40: Пуск привода для УСМ40 из панели в ручном режиме.
//   mh_PuskPrivUSM40: Маркер пуск привода для УСМ40 в ручном режиме.
//   Pusk_HMI_LiniyaUSM40: Пуск линия для УСМ40 из панели в ручном режиме.
//   mh_PuskLinUSM40: Маркер пуск линия для УСМ40 в ручном режиме.
//   i_TZ_PL1: IO | AT %IX1.2
//   m_AvarATVPL1: Ошибка от ПЧ ПЛ1-10_1.
//   Pusk_HMI_PL1: Пуск ПЛ1-10 №1 из панели в ручном режиме.
//   mh_Pusk_Pl1: Маркер пуск питателя ПЛ1-10 №1 в ручном режиме.
//   i_TZ_PL2: IO | AT %IX1.3
//   m_AvarATVPL2: Ошибка от ПЧ ПЛ1-10_2.
//   Pusk_HMI_PL2: Пуск ПЛ1-10 №2 из панели в ручном режиме.
//   mh_Pusk_PL2: Маркер пуск питателя ПЛ1-10 №2 в ручном режиме.
//   Pusk_HMI_SMK517_5_Rev: Пуск 5,5 кВт на СМК 517 в реверс из панели в ручном режиме.
//   mh_Pusk_SMK517_5_rev: Маркер пуск 5,5 кВт для СМК517 в реверс в ручном режиме.
//   mh_SMK517_Revers: Маркер пуск контактора СМК517 5,5 кВт в реверс в ручном режиме.
//   i_KEY_Protochka: TM2DDI32DK | AT %IX31.4
//   m_Tros_All: Все маркеры тросовых защит для останова линии по любому из тросовых выключателей.
//   m_Avar_Priv: Маркер общих защит приводов.
//   Pusk_HMI_Privoda: Пуск "Привода"
//   m_Pusk_Privoda: Маркер для "Пуск привода". Взводит таймеры для поочередного включения приводов.
//   m_Avar_Lin: Маркер общей защиты линии.
//   m_UrovenPL024U: Маркер уровня в питателе. Дает разрешение на включение линии.
//   Pusk_HMI_Liniya: Пуск "Линия"
//   m_Pusk_Liniya: Маркер для "Пуск Линия". Взводит таймеры для поочередного включения конвейеров.
//   m_TZ_SMK517_5: Промежуточный маркер тепловой защиты 5,5 кВт на СМК517 для квитирования.
//   m_Vkl_Protoch517: Маркер пуска 5,5 кВт на СМК517 для проточки.
//   mp_Pusk_SMK517_5_rev: Маркер пуск ATS на СМК517 в реверс для проточки.
//   mp_SMK517_Revers: Маркер пуск контактора 5,5 кВт на СМК517 в реверс для проточки.
_ft3(CLK := mZV2);
mh_Pusk_KO1 S= _ft3.Q AND NOT m_TZ_KO1 AND NOT m_Tros_KO1 AND Pusk_HMI_KO1;
mh_Pusk_KO2 S= _ft3.Q AND NOT m_TZ_KO2 AND NOT m_Tros_KO2 AND Pusk_HMI_KO2;
mh_Pusk_KO3 S= _ft3.Q AND NOT m_TZ_KO3 AND NOT m_Tros_KO3 AND Pusk_HMI_KO3;
mh_Pusk_KO4 S= _ft3.Q AND NOT m_TZ_KO4 AND NOT m_Tros_KO4 AND Pusk_HMI_KO4;
mh_Pusk_KO6 S= _ft3.Q AND NOT m_TZ_KO6 AND NOT m_Tros_KO6 AND Pusk_HMI_KO6;
mh_Pusk_KO7 S= _ft3.Q AND NOT m_TZ_KO7 AND NOT m_Tros_KO7 AND Pusk_HMI_KO7;
mh_Pusk_KO11 S= _ft3.Q AND NOT m_TZ_KO11 AND NOT m_Tros_KO11 AND Pusk_HMI_KO11;
mh_Pusk_PL024 S= _ft3.Q AND NOT i_Avar_PL024 AND NOT m_AvarATVPL024 AND Pusk_HMI_PL024;
mh_Pusk_PL012 S= _ft3.Q AND NOT i_Avar_PL012 AND NOT m_AvarATVPL012 AND Pusk_HMI_PL012;
mh_Pusk_EP80_1 S= _ft3.Q AND NOT i_TZ_EP80_1 AND Pusk_HMI_EP80_1;
mh_Pusk_SMK517_37 S= _ft3.Q AND NOT i_TZ_SMK517_37 AND Pusk_HMI_SMK517_37;
_w1 := _ft3.Q AND NOT i_TZ_SMK517_5 AND NOT m_Avar_SMK517_ATS AND Pusk_HMI_SMK517_5;
mh_Pusk_SMK517_5 S= _w1;
mh_SMK517_Prjamo S= _w1;
mh_Pusk_SMK516_45 S= _ft3.Q AND NOT i_TZ_SMK516_45 AND Pusk_HMI_SMK516_45;
mh_Pusk_SMK516_37 S= _ft3.Q AND NOT i_TZ_SMK516_37 AND Pusk_HMI_SMK516_37;
mh_Pusk_RazrSMK516 S= _ft3.Q AND NOT i_TZ_RazrSMK516 AND NOT m_AvarATVRazrSMK516 AND Pusk_HMI_RazrSMK516;
mh_Pusk_KonvSMK516 S= _ft3.Q AND NOT i_TZ_KonvSMK516 AND Pusk_HMI_KonvSMK516;
mh_Pusk_PL250 S= _ft3.Q AND NOT i_Avar_PL250 AND NOT m_AvarATVPL250 AND Pusk_HMI_PL250;
mh_Pusk_VodaPL250 S= _ft3.Q AND Pusk_HMI_VodaPL250;
mh_Pusk_EP80_2 S= _ft3.Q AND NOT i_TZ_EP80_2 AND Pusk_HMI_EP80_2;
mh_PuskPrivUSM40 S= _ft3.Q AND NOT i_Avar_USM40 AND NOT m_AvarATVUSM40 AND Pusk_HMI_PrivodaUSM40;
mh_PuskLinUSM40 S= _ft3.Q AND NOT i_Avar_USM40 AND Pusk_HMI_LiniyaUSM40;
mh_Pusk_Pl1 S= _ft3.Q AND NOT i_TZ_PL1 AND NOT m_AvarATVPL1 AND Pusk_HMI_PL1;
mh_Pusk_PL2 S= _ft3.Q AND NOT i_TZ_PL2 AND NOT m_AvarATVPL2 AND Pusk_HMI_PL2;
_w2 := _ft3.Q AND NOT i_TZ_SMK517_5 AND NOT m_Avar_SMK517_ATS AND Pusk_HMI_SMK517_5_Rev;
mh_Pusk_SMK517_5_rev S= _w2;
mh_SMK517_Revers S= _w2;
m_Pusk_Privoda S= _ft3.Q AND NOT i_KEY_Protochka AND NOT m_Tros_All AND NOT m_Avar_Priv AND Pusk_HMI_Privoda;
m_Pusk_Liniya S= _ft3.Q AND NOT i_KEY_Protochka AND NOT m_Tros_All AND NOT m_Avar_Priv AND NOT m_Avar_Lin AND m_UrovenPL024U AND Pusk_HMI_Liniya AND Pusk_HMI_Privoda;
_w3 := _ft3.Q AND i_KEY_Protochka AND NOT m_TZ_SMK517_5 AND NOT m_Avar_SMK517_ATS AND m_Vkl_Protoch517;
mp_Pusk_SMK517_5_rev S= _w3;
mp_SMK517_Revers S= _w3;

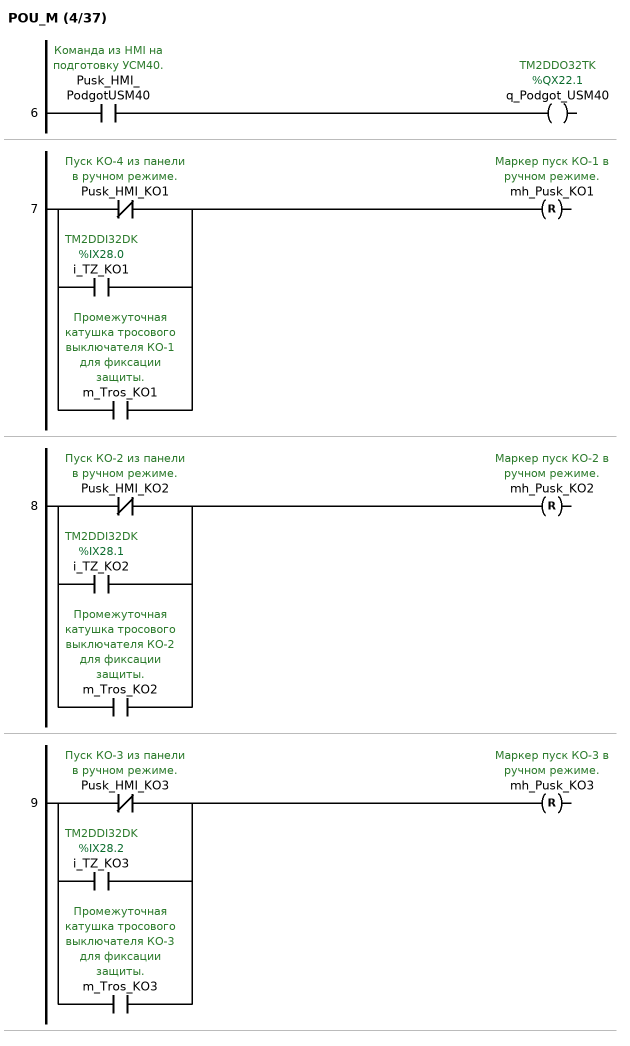
// NETWORK 6
//   Pusk_HMI_PodgotUSM40: Команда из HMI на подготовку УСМ40.
//   q_Podgot_USM40: TM2DDO32TK | AT %QX22.1
q_Podgot_USM40 := Pusk_HMI_PodgotUSM40;

// NETWORK 7
//   Pusk_HMI_KO1: Пуск КО-4 из панели в ручном режиме.
//   i_TZ_KO1: TM2DDI32DK | AT %IX28.0
//   m_Tros_KO1: Промежуточная катушка тросового выключателя КО-1 для фиксации защиты.
//   mh_Pusk_KO1: Маркер пуск КО-1 в ручном режиме.
mh_Pusk_KO1 R= NOT Pusk_HMI_KO1 OR i_TZ_KO1 OR m_Tros_KO1;

// NETWORK 8
//   Pusk_HMI_KO2: Пуск КО-2 из панели в ручном режиме.
//   i_TZ_KO2: TM2DDI32DK | AT %IX28.1
//   m_Tros_KO2: Промежуточная катушка тросового выключателя КО-2 для фиксации защиты.
//   mh_Pusk_KO2: Маркер пуск КО-2 в ручном режиме.
mh_Pusk_KO2 R= NOT Pusk_HMI_KO2 OR i_TZ_KO2 OR m_Tros_KO2;

// NETWORK 9
//   Pusk_HMI_KO3: Пуск КО-3 из панели в ручном режиме.
//   i_TZ_KO3: TM2DDI32DK | AT %IX28.2
//   m_Tros_KO3: Промежуточная катушка тросового выключателя КО-3 для фиксации защиты.
//   mh_Pusk_KO3: Маркер пуск КО-3 в ручном режиме.
mh_Pusk_KO3 R= NOT Pusk_HMI_KO3 OR i_TZ_KO3 OR m_Tros_KO3;

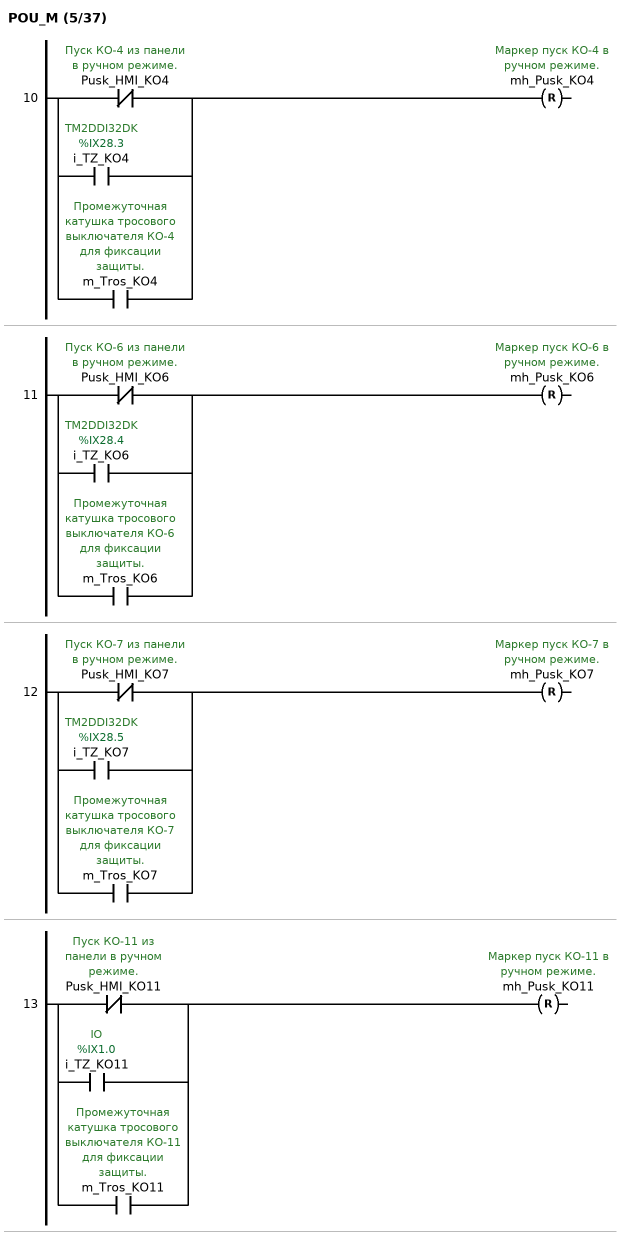
// NETWORK 10
//   Pusk_HMI_KO4: Пуск КО-4 из панели в ручном режиме.
//   i_TZ_KO4: TM2DDI32DK | AT %IX28.3
//   m_Tros_KO4: Промежуточная катушка тросового выключателя КО-4 для фиксации защиты.
//   mh_Pusk_KO4: Маркер пуск КО-4 в ручном режиме.
mh_Pusk_KO4 R= NOT Pusk_HMI_KO4 OR i_TZ_KO4 OR m_Tros_KO4;

// NETWORK 11
//   Pusk_HMI_KO6: Пуск КО-6 из панели в ручном режиме.
//   i_TZ_KO6: TM2DDI32DK | AT %IX28.4
//   m_Tros_KO6: Промежуточная катушка тросового выключателя КО-6 для фиксации защиты.
//   mh_Pusk_KO6: Маркер пуск КО-6 в ручном режиме.
mh_Pusk_KO6 R= NOT Pusk_HMI_KO6 OR i_TZ_KO6 OR m_Tros_KO6;

// NETWORK 12
//   Pusk_HMI_KO7: Пуск КО-7 из панели в ручном режиме.
//   i_TZ_KO7: TM2DDI32DK | AT %IX28.5
//   m_Tros_KO7: Промежуточная катушка тросового выключателя КО-7 для фиксации защиты.
//   mh_Pusk_KO7: Маркер пуск КО-7 в ручном режиме.
mh_Pusk_KO7 R= NOT Pusk_HMI_KO7 OR i_TZ_KO7 OR m_Tros_KO7;

// NETWORK 13
//   Pusk_HMI_KO11: Пуск КО-11 из панели в ручном режиме.
//   i_TZ_KO11: IO | AT %IX1.0
//   m_Tros_KO11: Промежуточная катушка тросового выключателя КО-11 для фиксации защиты.
//   mh_Pusk_KO11: Маркер пуск КО-11 в ручном режиме.
mh_Pusk_KO11 R= NOT Pusk_HMI_KO11 OR i_TZ_KO11 OR m_Tros_KO11;

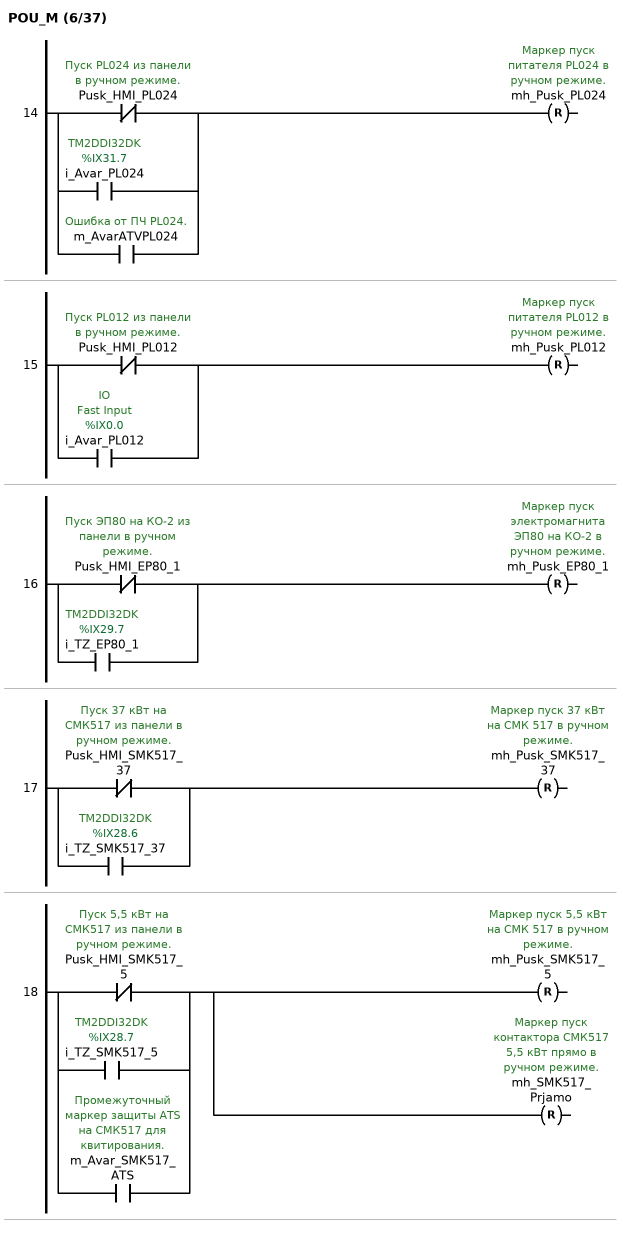
// NETWORK 14
//   Pusk_HMI_PL024: Пуск PL024 из панели в ручном режиме.
//   i_Avar_PL024: TM2DDI32DK | AT %IX31.7
//   m_AvarATVPL024: Ошибка от ПЧ PL024.
//   mh_Pusk_PL024: Маркер пуск питателя PL024 в ручном режиме.
mh_Pusk_PL024 R= NOT Pusk_HMI_PL024 OR i_Avar_PL024 OR m_AvarATVPL024;

// NETWORK 15
//   Pusk_HMI_PL012: Пуск PL012 из панели в ручном режиме.
//   i_Avar_PL012: IO Fast Input | AT %IX0.0
//   mh_Pusk_PL012: Маркер пуск питателя PL012 в ручном режиме.
mh_Pusk_PL012 R= NOT Pusk_HMI_PL012 OR i_Avar_PL012;

// NETWORK 16
//   Pusk_HMI_EP80_1: Пуск ЭП80 на КО-2 из панели в ручном режиме.
//   i_TZ_EP80_1: TM2DDI32DK | AT %IX29.7
//   mh_Pusk_EP80_1: Маркер пуск электромагнита ЭП80 на КО-2 в ручном режиме.
mh_Pusk_EP80_1 R= NOT Pusk_HMI_EP80_1 OR i_TZ_EP80_1;

// NETWORK 17
//   Pusk_HMI_SMK517_37: Пуск 37 кВт на СМК517 из панели в ручном режиме.
//   i_TZ_SMK517_37: TM2DDI32DK | AT %IX28.6
//   mh_Pusk_SMK517_37: Маркер пуск 37 кВт на СМК 517 в ручном режиме.
mh_Pusk_SMK517_37 R= NOT Pusk_HMI_SMK517_37 OR i_TZ_SMK517_37;

// NETWORK 18
//   Pusk_HMI_SMK517_5: Пуск 5,5 кВт на СМК517 из панели в ручном режиме.
//   i_TZ_SMK517_5: TM2DDI32DK | AT %IX28.7
//   m_Avar_SMK517_ATS: Промежуточный маркер защиты ATS на СМК517 для квитирования.
//   mh_Pusk_SMK517_5: Маркер пуск 5,5 кВт на СМК 517 в ручном режиме.
//   mh_SMK517_Prjamo: Маркер пуск контактора СМК517 5,5 кВт прямо в ручном режиме.
_w4 := NOT Pusk_HMI_SMK517_5 OR i_TZ_SMK517_5 OR m_Avar_SMK517_ATS;
mh_Pusk_SMK517_5 R= _w4;
mh_SMK517_Prjamo R= _w4;

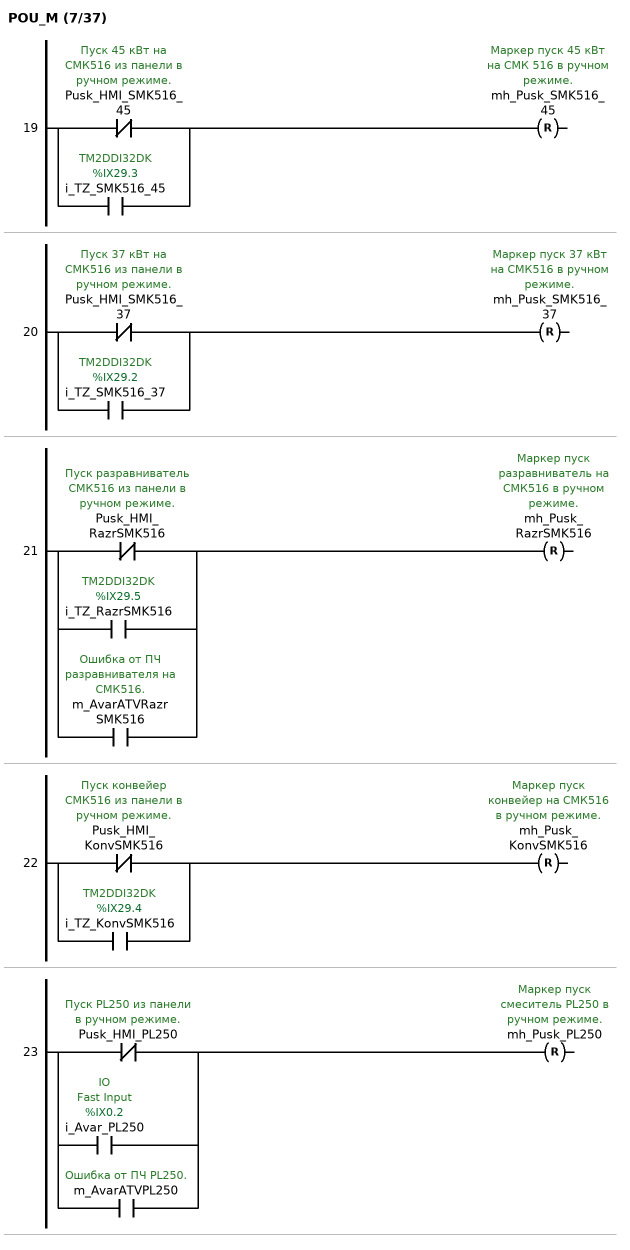
// NETWORK 19
//   Pusk_HMI_SMK516_45: Пуск 45 кВт на СМК516 из панели в ручном режиме.
//   i_TZ_SMK516_45: TM2DDI32DK | AT %IX29.3
//   mh_Pusk_SMK516_45: Маркер пуск 45 кВт на СМК 516 в ручном режиме.
mh_Pusk_SMK516_45 R= NOT Pusk_HMI_SMK516_45 OR i_TZ_SMK516_45;

// NETWORK 20
//   Pusk_HMI_SMK516_37: Пуск 37 кВт на СМК516 из панели в ручном режиме.
//   i_TZ_SMK516_37: TM2DDI32DK | AT %IX29.2
//   mh_Pusk_SMK516_37: Маркер пуск 37 кВт на СМК516 в ручном режиме.
mh_Pusk_SMK516_37 R= NOT Pusk_HMI_SMK516_37 OR i_TZ_SMK516_37;

// NETWORK 21
//   Pusk_HMI_RazrSMK516: Пуск разравниватель СМК516 из панели в ручном режиме.
//   i_TZ_RazrSMK516: TM2DDI32DK | AT %IX29.5
//   m_AvarATVRazrSMK516: Ошибка от ПЧ разравнивателя на СМК516.
//   mh_Pusk_RazrSMK516: Маркер пуск разравниватель на СМК516 в ручном режиме.
mh_Pusk_RazrSMK516 R= NOT Pusk_HMI_RazrSMK516 OR i_TZ_RazrSMK516 OR m_AvarATVRazrSMK516;

// NETWORK 22
//   Pusk_HMI_KonvSMK516: Пуск конвейер СМК516 из панели в ручном режиме.
//   i_TZ_KonvSMK516: TM2DDI32DK | AT %IX29.4
//   mh_Pusk_KonvSMK516: Маркер пуск конвейер на СМК516 в ручном режиме.
mh_Pusk_KonvSMK516 R= NOT Pusk_HMI_KonvSMK516 OR i_TZ_KonvSMK516;

// NETWORK 23
//   Pusk_HMI_PL250: Пуск PL250 из панели в ручном режиме.
//   i_Avar_PL250: IO Fast Input | AT %IX0.2
//   m_AvarATVPL250: Ошибка от ПЧ PL250.
//   mh_Pusk_PL250: Маркер пуск смеситель PL250 в ручном режиме.
mh_Pusk_PL250 R= NOT Pusk_HMI_PL250 OR i_Avar_PL250 OR m_AvarATVPL250;

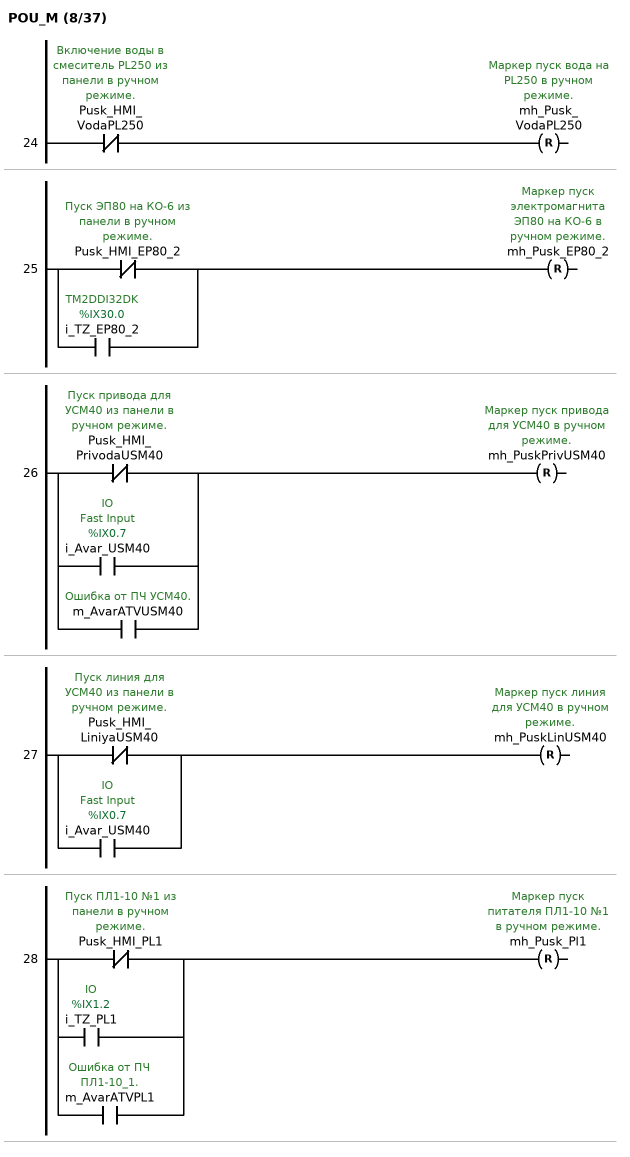
// NETWORK 24
//   Pusk_HMI_VodaPL250: Включение воды в смеситель PL250 из панели в ручном режиме.
//   mh_Pusk_VodaPL250: Маркер пуск вода на PL250 в ручном режиме.
mh_Pusk_VodaPL250 R= NOT Pusk_HMI_VodaPL250;

// NETWORK 25
//   Pusk_HMI_EP80_2: Пуск ЭП80 на КО-6 из панели в ручном режиме.
//   i_TZ_EP80_2: TM2DDI32DK | AT %IX30.0
//   mh_Pusk_EP80_2: Маркер пуск электромагнита ЭП80 на КО-6 в ручном режиме.
mh_Pusk_EP80_2 R= NOT Pusk_HMI_EP80_2 OR i_TZ_EP80_2;

// NETWORK 26
//   Pusk_HMI_PrivodaUSM40: Пуск привода для УСМ40 из панели в ручном режиме.
//   i_Avar_USM40: IO Fast Input | AT %IX0.7
//   m_AvarATVUSM40: Ошибка от ПЧ УСМ40.
//   mh_PuskPrivUSM40: Маркер пуск привода для УСМ40 в ручном режиме.
mh_PuskPrivUSM40 R= NOT Pusk_HMI_PrivodaUSM40 OR i_Avar_USM40 OR m_AvarATVUSM40;

// NETWORK 27
//   Pusk_HMI_LiniyaUSM40: Пуск линия для УСМ40 из панели в ручном режиме.
//   i_Avar_USM40: IO Fast Input | AT %IX0.7
//   mh_PuskLinUSM40: Маркер пуск линия для УСМ40 в ручном режиме.
mh_PuskLinUSM40 R= NOT Pusk_HMI_LiniyaUSM40 OR i_Avar_USM40;

// NETWORK 28
//   Pusk_HMI_PL1: Пуск ПЛ1-10 №1 из панели в ручном режиме.
//   i_TZ_PL1: IO | AT %IX1.2
//   m_AvarATVPL1: Ошибка от ПЧ ПЛ1-10_1.
//   mh_Pusk_Pl1: Маркер пуск питателя ПЛ1-10 №1 в ручном режиме.
mh_Pusk_Pl1 R= NOT Pusk_HMI_PL1 OR i_TZ_PL1 OR m_AvarATVPL1;

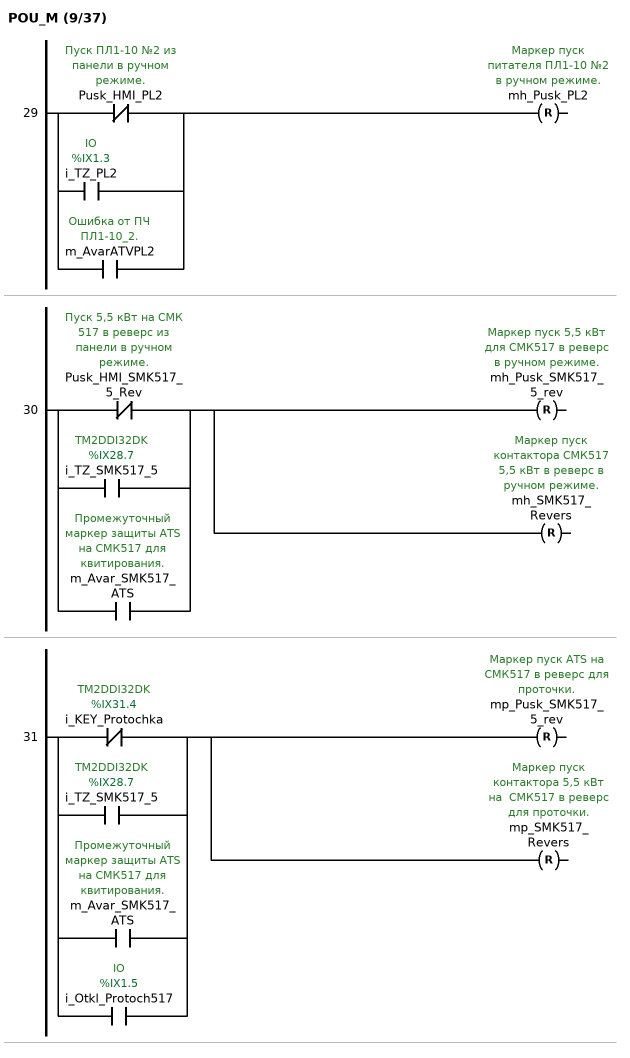
// NETWORK 29
//   Pusk_HMI_PL2: Пуск ПЛ1-10 №2 из панели в ручном режиме.
//   i_TZ_PL2: IO | AT %IX1.3
//   m_AvarATVPL2: Ошибка от ПЧ ПЛ1-10_2.
//   mh_Pusk_PL2: Маркер пуск питателя ПЛ1-10 №2 в ручном режиме.
mh_Pusk_PL2 R= NOT Pusk_HMI_PL2 OR i_TZ_PL2 OR m_AvarATVPL2;

// NETWORK 30
//   Pusk_HMI_SMK517_5_Rev: Пуск 5,5 кВт на СМК 517 в реверс из панели в ручном режиме.
//   i_TZ_SMK517_5: TM2DDI32DK | AT %IX28.7
//   m_Avar_SMK517_ATS: Промежуточный маркер защиты ATS на СМК517 для квитирования.
//   mh_Pusk_SMK517_5_rev: Маркер пуск 5,5 кВт для СМК517 в реверс в ручном режиме.
//   mh_SMK517_Revers: Маркер пуск контактора СМК517 5,5 кВт в реверс в ручном режиме.
_w5 := NOT Pusk_HMI_SMK517_5_Rev OR i_TZ_SMK517_5 OR m_Avar_SMK517_ATS;
mh_Pusk_SMK517_5_rev R= _w5;
mh_SMK517_Revers R= _w5;

// NETWORK 31
//   i_KEY_Protochka: TM2DDI32DK | AT %IX31.4
//   i_TZ_SMK517_5: TM2DDI32DK | AT %IX28.7
//   m_Avar_SMK517_ATS: Промежуточный маркер защиты ATS на СМК517 для квитирования.
//   i_Otkl_Protoch517: IO | AT %IX1.5
//   mp_Pusk_SMK517_5_rev: Маркер пуск ATS на СМК517 в реверс для проточки.
//   mp_SMK517_Revers: Маркер пуск контактора 5,5 кВт на СМК517 в реверс для проточки.
_w6 := NOT i_KEY_Protochka OR i_TZ_SMK517_5 OR m_Avar_SMK517_ATS OR i_Otkl_Protoch517;
mp_Pusk_SMK517_5_rev R= _w6;
mp_SMK517_Revers R= _w6;

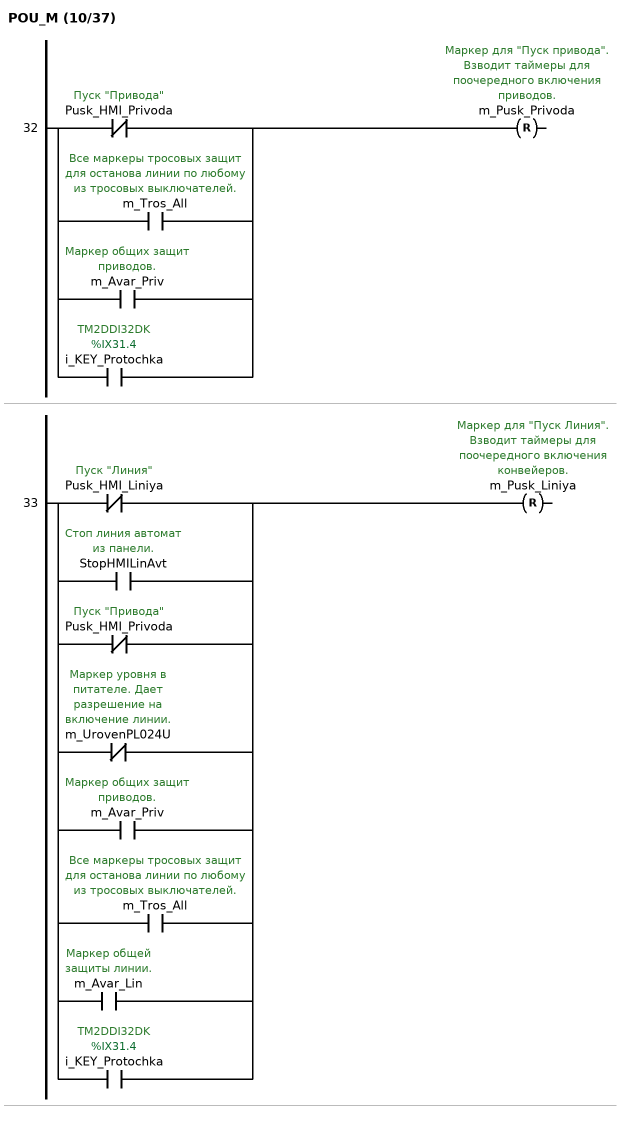
// NETWORK 32
//   Pusk_HMI_Privoda: Пуск "Привода"
//   m_Tros_All: Все маркеры тросовых защит для останова линии по любому из тросовых выключателей.
//   m_Avar_Priv: Маркер общих защит приводов.
//   i_KEY_Protochka: TM2DDI32DK | AT %IX31.4
//   m_Pusk_Privoda: Маркер для "Пуск привода". Взводит таймеры для поочередного включения приводов.
m_Pusk_Privoda R= NOT Pusk_HMI_Privoda OR m_Tros_All OR m_Avar_Priv OR i_KEY_Protochka;

// NETWORK 33
//   Pusk_HMI_Liniya: Пуск "Линия"
//   StopHMILinAvt: Стоп линия автомат из панели.
//   Pusk_HMI_Privoda: Пуск "Привода"
//   m_UrovenPL024U: Маркер уровня в питателе. Дает разрешение на включение линии.
//   m_Avar_Priv: Маркер общих защит приводов.
//   m_Tros_All: Все маркеры тросовых защит для останова линии по любому из тросовых выключателей.
//   m_Avar_Lin: Маркер общей защиты линии.
//   i_KEY_Protochka: TM2DDI32DK | AT %IX31.4
//   m_Pusk_Liniya: Маркер для "Пуск Линия". Взводит таймеры для поочередного включения конвейеров.
m_Pusk_Liniya R= NOT Pusk_HMI_Liniya OR StopHMILinAvt OR NOT Pusk_HMI_Privoda OR NOT m_UrovenPL024U OR m_Avar_Priv OR m_Tros_All OR m_Avar_Lin OR i_KEY_Protochka;

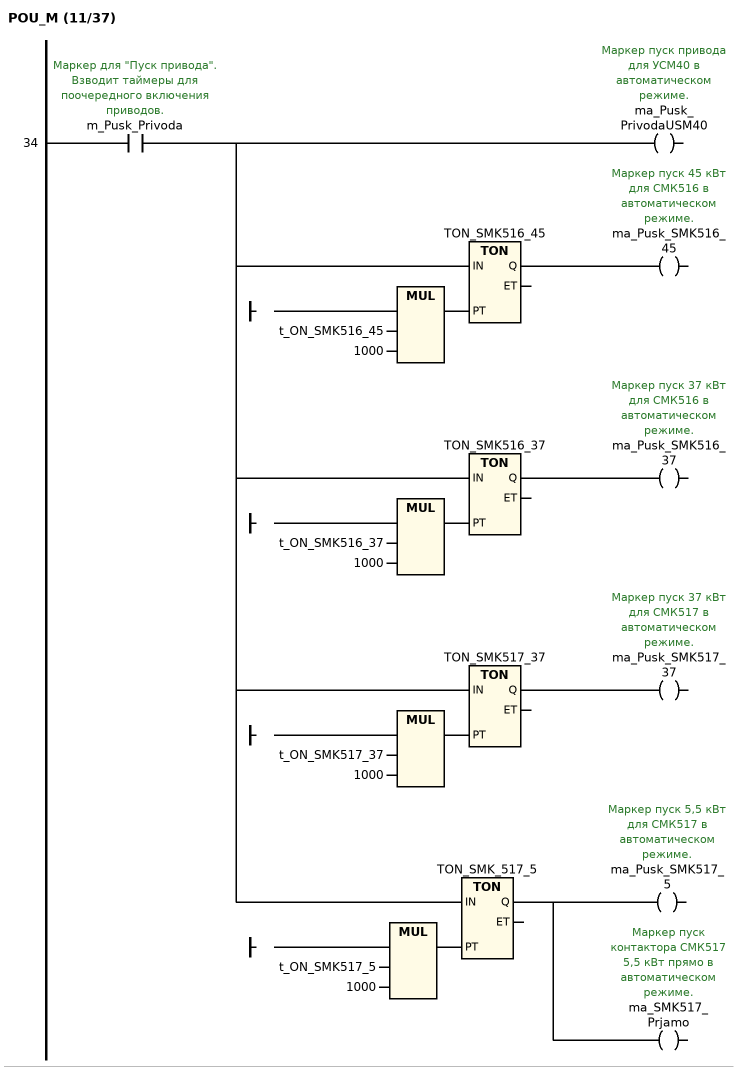
// NETWORK 34
//   m_Pusk_Privoda: Маркер для "Пуск привода". Взводит таймеры для поочередного включения приводов.
//   ma_Pusk_PrivodaUSM40: Маркер пуск привода для УСМ40 в автоматическом режиме.
//   TON_SMK516_45: Задержка перед пуском 45 кВт на СМК516.
//   t_ON_SMK516_45: Время задержки перед включением СМК516 45 кВт.
//   ma_Pusk_SMK516_45: Маркер пуск 45 кВт для СМК516 в автоматическом режиме.
//   TON_SMK516_37: Задержка перед пуском 37 кВт на СМК516.
//   t_ON_SMK516_37: Время задержки перед включением СМК516 37 кВт.
//   ma_Pusk_SMK516_37: Маркер пуск 37 кВт для СМК516 в автоматическом режиме.
//   TON_SMK517_37: Задержка перед пуском 37 кВт на СМК517.
//   t_ON_SMK517_37: Время задержки перед включением СМК517 37 кВт.
//   ma_Pusk_SMK517_37: Маркер пуск 37 кВт для СМК517 в автоматическом режиме.
//   TON_SMK_517_5: Задержка перед запуском 5 кВт на СМК517.
//   t_ON_SMK517_5: Время задержки перед включением СМК516 5,5 кВт.
//   ma_Pusk_SMK517_5: Маркер пуск 5,5 кВт для СМК517 в автоматическом режиме.
//   ma_SMK517_Prjamo: Маркер пуск контактора СМК517 5,5 кВт прямо в автоматическом режиме.
ma_Pusk_PrivodaUSM40 := m_Pusk_Privoda;
TON_SMK516_45(IN := m_Pusk_Privoda, PT := t_ON_SMK516_45 * 1000); // TON
ma_Pusk_SMK516_45 := TON_SMK516_45.Q;
TON_SMK516_37(IN := m_Pusk_Privoda, PT := t_ON_SMK516_37 * 1000); // TON
ma_Pusk_SMK516_37 := TON_SMK516_37.Q;
TON_SMK517_37(IN := m_Pusk_Privoda, PT := t_ON_SMK517_37 * 1000); // TON
ma_Pusk_SMK517_37 := TON_SMK517_37.Q;
TON_SMK_517_5(IN := m_Pusk_Privoda, PT := t_ON_SMK517_5 * 1000); // TON
ma_Pusk_SMK517_5 := TON_SMK_517_5.Q;
ma_SMK517_Prjamo := TON_SMK_517_5.Q;

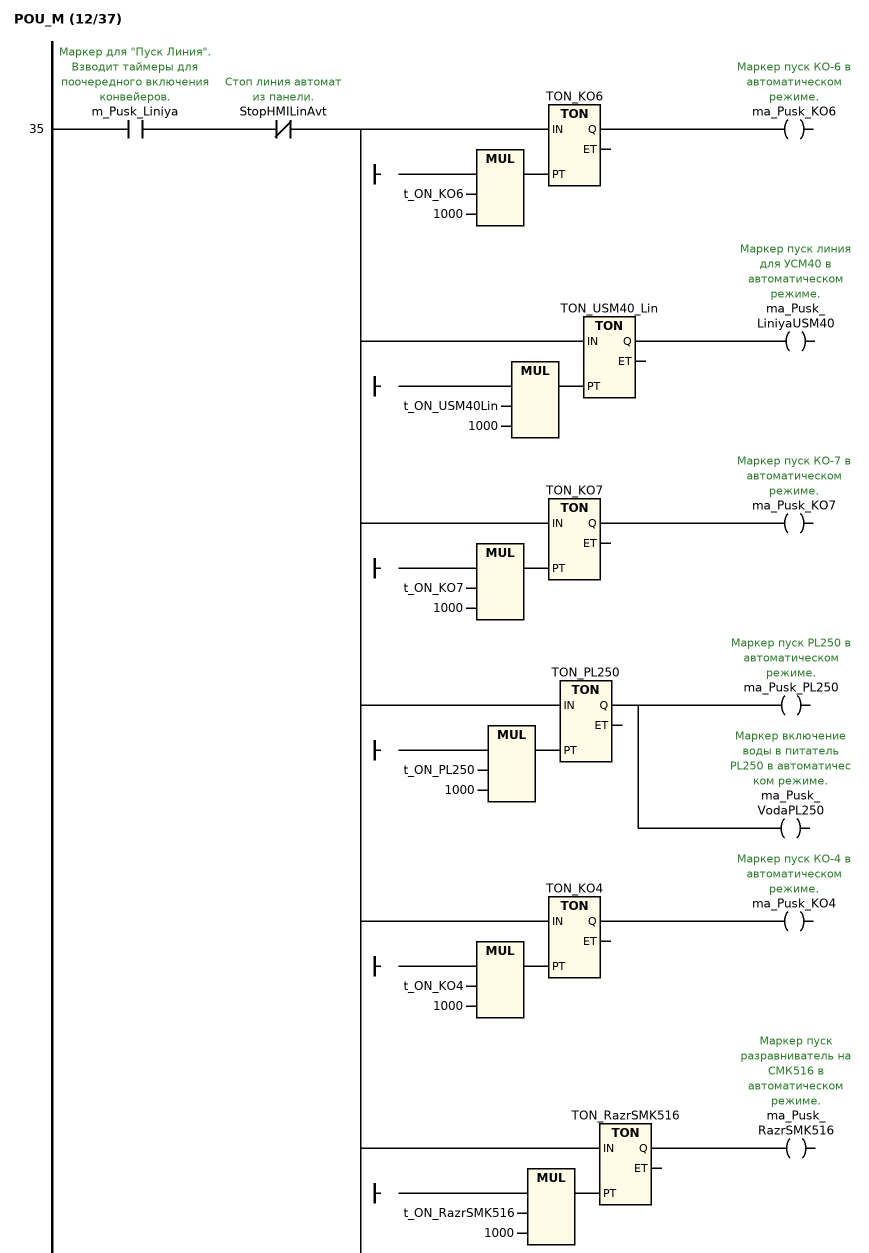
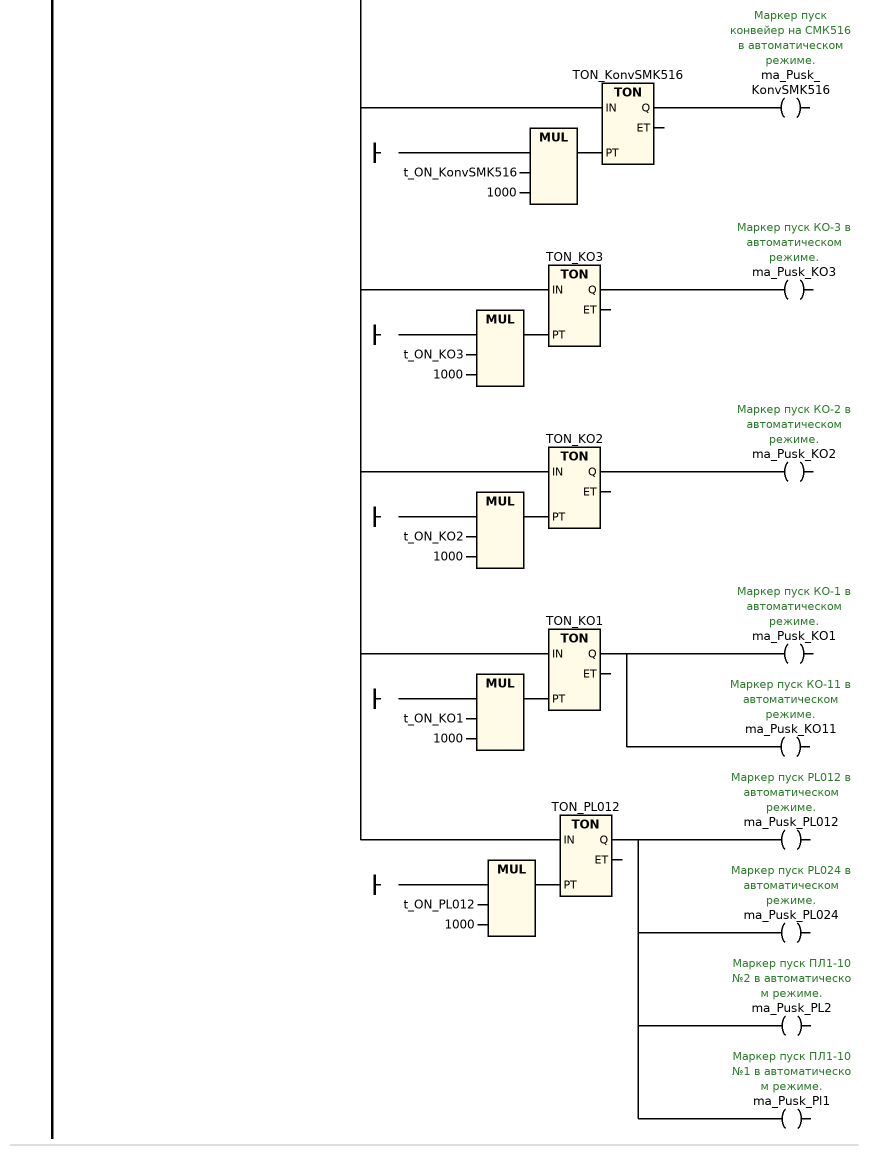
// NETWORK 35
//   m_Pusk_Liniya: Маркер для "Пуск Линия". Взводит таймеры для поочередного включения конвейеров.
//   StopHMILinAvt: Стоп линия автомат из панели.
//   TON_KO6: Задержка перед включением КО-6.
//   t_ON_KO6: Время задержки перед включением КО-6.
//   ma_Pusk_KO6: Маркер пуск КО-6 в автоматическом режиме.
//   TON_USM40_Lin: Задержка перед включение УСМ40 по "Пуск линия".
//   t_ON_USM40Lin: Время задержки перед включением линии на УСМ40.
//   ma_Pusk_LiniyaUSM40: Маркер пуск линия для УСМ40 в автоматическом режиме.
//   TON_KO7: Задержка перед включение КО-7.
//   t_ON_KO7: Время задержки перед включением КО-7.
//   ma_Pusk_KO7: Маркер пуск КО-7 в автоматическом режиме.
//   TON_PL250: Задержка перед включением PL250.
//   t_ON_PL250: Время задержки перед включением PL250.
//   ma_Pusk_PL250: Маркер пуск PL250 в автоматическом режиме.
//   ma_Pusk_VodaPL250: Маркер включение воды в питатель PL250 в автоматическом режиме.
//   TON_KO4: Задержка перед включением КО-4.
//   t_ON_KO4: Время задержки перед включением КО-4.
//   ma_Pusk_KO4: Маркер пуск КО-4 в автоматическом режиме.
//   TON_RazrSMK516: Задержка перед включением разравнивателя на СМК516 по "Пуск линия".
//   t_ON_RazrSMK516: Время задержки перед включением разравнивателя на СМК516.
//   ma_Pusk_RazrSMK516: Маркер пуск разравниватель на СМК516 в автоматическом режиме.
//   TON_KonvSMK516: Задержка перед включением конвейера на СМК516 по "Пуск линия".
//   t_ON_KonvSMK516: Время задержки перед включением конвейера на СМК516.
//   ma_Pusk_KonvSMK516: Маркер пуск конвейер на СМК516 в автоматическом режиме.
//   TON_KO3: Задержка перед включением КО-3.
//   t_ON_KO3: Время задержки перед включением КО-3.
//   ma_Pusk_KO3: Маркер пуск КО-3 в автоматическом режиме.
//   TON_KO2: Задержка перед включением КО-2.
//   t_ON_KO2: Время задержки перед включением КО-2.
//   ma_Pusk_KO2: Маркер пуск КО-2 в автоматическом режиме.
//   TON_KO1: Задержка перед включением КО-1.
//   t_ON_KO1: Время задержки перед включением КО-1 и КО-11.
//   ma_Pusk_KO1: Маркер пуск КО-1 в автоматическом режиме.
//   ma_Pusk_KO11: Маркер пуск КО-11 в автоматическом режиме.
//   TON_PL012: Задержка перед включением PL012.
//   t_ON_PL012: Время задержки перед включением питателей в приемном (PL012, PL024) отделении и на добавках (ПЛ1-10).
//   ma_Pusk_PL012: Маркер пуск PL012 в автоматическом режиме.
//   ma_Pusk_PL024: Маркер пуск PL024 в автоматическом режиме.
//   ma_Pusk_PL2: Маркер пуск ПЛ1-10 №2 в автоматическом режиме.
//   ma_Pusk_Pl1: Маркер пуск ПЛ1-10 №1 в автоматическом режиме.
_w7 := m_Pusk_Liniya AND NOT StopHMILinAvt;
TON_KO6(IN := _w7, PT := t_ON_KO6 * 1000); // TON
ma_Pusk_KO6 := TON_KO6.Q;
TON_USM40_Lin(IN := _w7, PT := t_ON_USM40Lin * 1000); // TON
ma_Pusk_LiniyaUSM40 := TON_USM40_Lin.Q;
TON_KO7(IN := _w7, PT := t_ON_KO7 * 1000); // TON
ma_Pusk_KO7 := TON_KO7.Q;
TON_PL250(IN := _w7, PT := t_ON_PL250 * 1000); // TON
ma_Pusk_PL250 := TON_PL250.Q;
ma_Pusk_VodaPL250 := TON_PL250.Q;
TON_KO4(IN := _w7, PT := t_ON_KO4 * 1000); // TON
ma_Pusk_KO4 := TON_KO4.Q;
TON_RazrSMK516(IN := _w7, PT := t_ON_RazrSMK516 * 1000); // TON
ma_Pusk_RazrSMK516 := TON_RazrSMK516.Q;
TON_KonvSMK516(IN := _w7, PT := t_ON_KonvSMK516 * 1000); // TON
ma_Pusk_KonvSMK516 := TON_KonvSMK516.Q;
TON_KO3(IN := _w7, PT := t_ON_KO3 * 1000); // TON
ma_Pusk_KO3 := TON_KO3.Q;
TON_KO2(IN := _w7, PT := t_ON_KO2 * 1000); // TON
ma_Pusk_KO2 := TON_KO2.Q;
TON_KO1(IN := _w7, PT := t_ON_KO1 * 1000); // TON
ma_Pusk_KO1 := TON_KO1.Q;
ma_Pusk_KO11 := TON_KO1.Q;
TON_PL012(IN := _w7, PT := t_ON_PL012 * 1000); // TON
ma_Pusk_PL012 := TON_PL012.Q;
ma_Pusk_PL024 := TON_PL012.Q;
ma_Pusk_PL2 := TON_PL012.Q;
ma_Pusk_Pl1 := TON_PL012.Q;

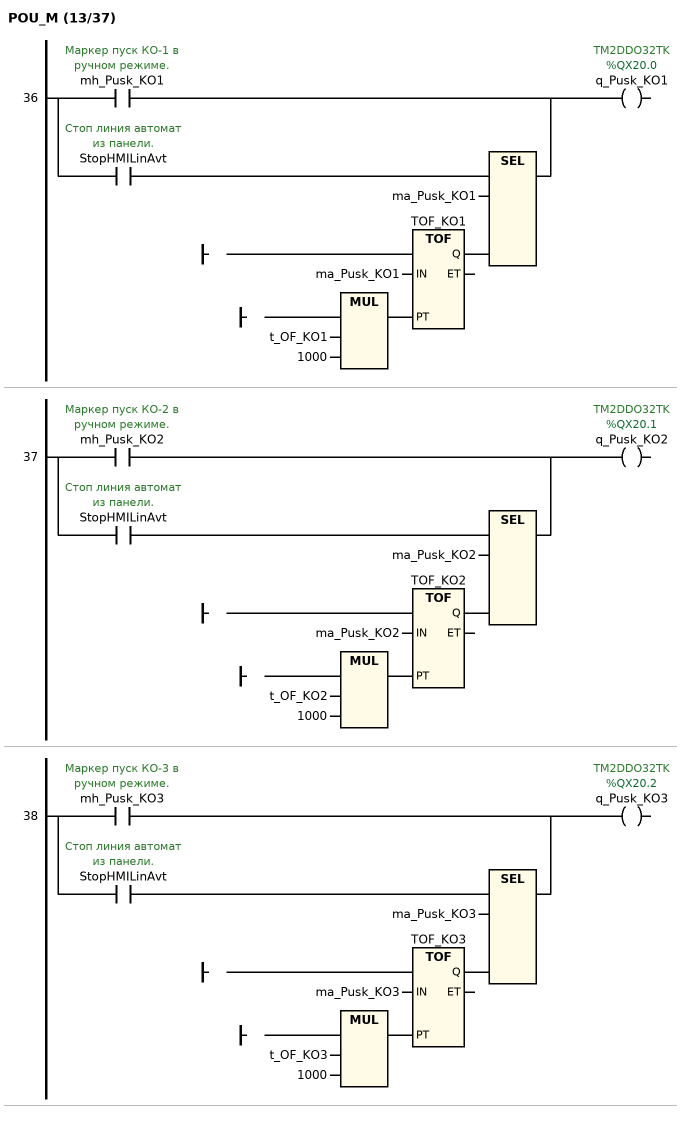
// NETWORK 36
//   mh_Pusk_KO1: Маркер пуск КО-1 в ручном режиме.
//   StopHMILinAvt: Стоп линия автомат из панели.
//   ma_Pusk_KO1: Маркер пуск КО-1 в автоматическом режиме.
//   TOF_KO1: Задержка перед выключением КО-1 при "Стоп линия автомат".
//   t_OF_KO1: Время задержки перед выключением КО-1 при Стоп Линия Автомат.
//   q_Pusk_KO1: TM2DDO32TK | AT %QX20.0
TOF_KO1(IN := ma_Pusk_KO1, PT := t_OF_KO1 * 1000); // TOF
q_Pusk_KO1 := mh_Pusk_KO1 OR SEL(StopHMILinAvt, ma_Pusk_KO1, TOF_KO1.Q);

// NETWORK 37
//   mh_Pusk_KO2: Маркер пуск КО-2 в ручном режиме.
//   StopHMILinAvt: Стоп линия автомат из панели.
//   ma_Pusk_KO2: Маркер пуск КО-2 в автоматическом режиме.
//   TOF_KO2: Задержка перед выключением КО-2 при "Стоп линия автомат".
//   t_OF_KO2: Время задержки перед выключением КО-2 при Стоп Линия Автомат.
//   q_Pusk_KO2: TM2DDO32TK | AT %QX20.1
TOF_KO2(IN := ma_Pusk_KO2, PT := t_OF_KO2 * 1000); // TOF
q_Pusk_KO2 := mh_Pusk_KO2 OR SEL(StopHMILinAvt, ma_Pusk_KO2, TOF_KO2.Q);

// NETWORK 38
//   mh_Pusk_KO3: Маркер пуск КО-3 в ручном режиме.
//   StopHMILinAvt: Стоп линия автомат из панели.
//   ma_Pusk_KO3: Маркер пуск КО-3 в автоматическом режиме.
//   TOF_KO3: Задержка перед выключением КО-3 при "Стоп линия автомат".
//   t_OF_KO3: Время задержки перед выключением КО-3 при Стоп Линия Автомат.
//   q_Pusk_KO3: TM2DDO32TK | AT %QX20.2
TOF_KO3(IN := ma_Pusk_KO3, PT := t_OF_KO3 * 1000); // TOF
q_Pusk_KO3 := mh_Pusk_KO3 OR SEL(StopHMILinAvt, ma_Pusk_KO3, TOF_KO3.Q);

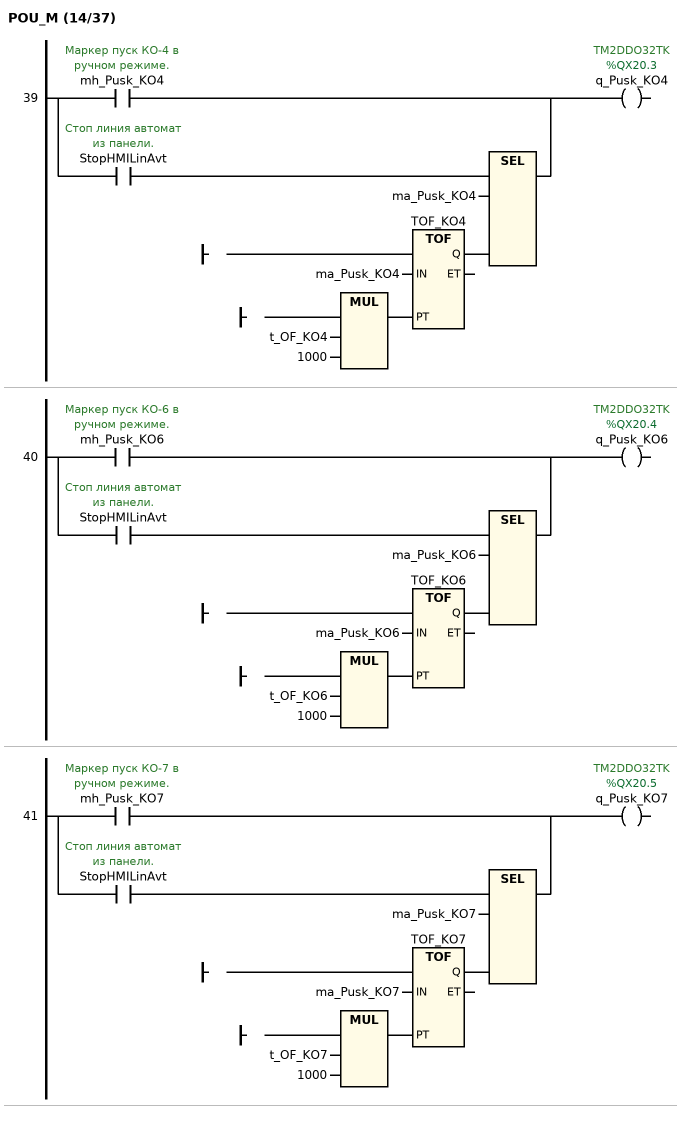
// NETWORK 39
//   mh_Pusk_KO4: Маркер пуск КО-4 в ручном режиме.
//   StopHMILinAvt: Стоп линия автомат из панели.
//   ma_Pusk_KO4: Маркер пуск КО-4 в автоматическом режиме.
//   TOF_KO4: Задержка перед выключением КО-4 при "Стоп линия автомат".
//   t_OF_KO4: Время задержки перед выключением КО-4 при Стоп Линия Автомат.
//   q_Pusk_KO4: TM2DDO32TK | AT %QX20.3
TOF_KO4(IN := ma_Pusk_KO4, PT := t_OF_KO4 * 1000); // TOF
q_Pusk_KO4 := mh_Pusk_KO4 OR SEL(StopHMILinAvt, ma_Pusk_KO4, TOF_KO4.Q);

// NETWORK 40
//   mh_Pusk_KO6: Маркер пуск КО-6 в ручном режиме.
//   StopHMILinAvt: Стоп линия автомат из панели.
//   ma_Pusk_KO6: Маркер пуск КО-6 в автоматическом режиме.
//   TOF_KO6: Задержка перед выключением КО-6 при "Стоп линия автомат".
//   t_OF_KO6: Время задержки перед выключением КО-6 при Стоп Линия Автомат.
//   q_Pusk_KO6: TM2DDO32TK | AT %QX20.4
TOF_KO6(IN := ma_Pusk_KO6, PT := t_OF_KO6 * 1000); // TOF
q_Pusk_KO6 := mh_Pusk_KO6 OR SEL(StopHMILinAvt, ma_Pusk_KO6, TOF_KO6.Q);

// NETWORK 41
//   mh_Pusk_KO7: Маркер пуск КО-7 в ручном режиме.
//   StopHMILinAvt: Стоп линия автомат из панели.
//   ma_Pusk_KO7: Маркер пуск КО-7 в автоматическом режиме.
//   TOF_KO7: Задержка перед выключением КО-7 при "Стоп линия автомат".
//   t_OF_KO7: Время задержки перед выключением КО-7 при Стоп Линия Автомат.
//   q_Pusk_KO7: TM2DDO32TK | AT %QX20.5
TOF_KO7(IN := ma_Pusk_KO7, PT := t_OF_KO7 * 1000); // TOF
q_Pusk_KO7 := mh_Pusk_KO7 OR SEL(StopHMILinAvt, ma_Pusk_KO7, TOF_KO7.Q);

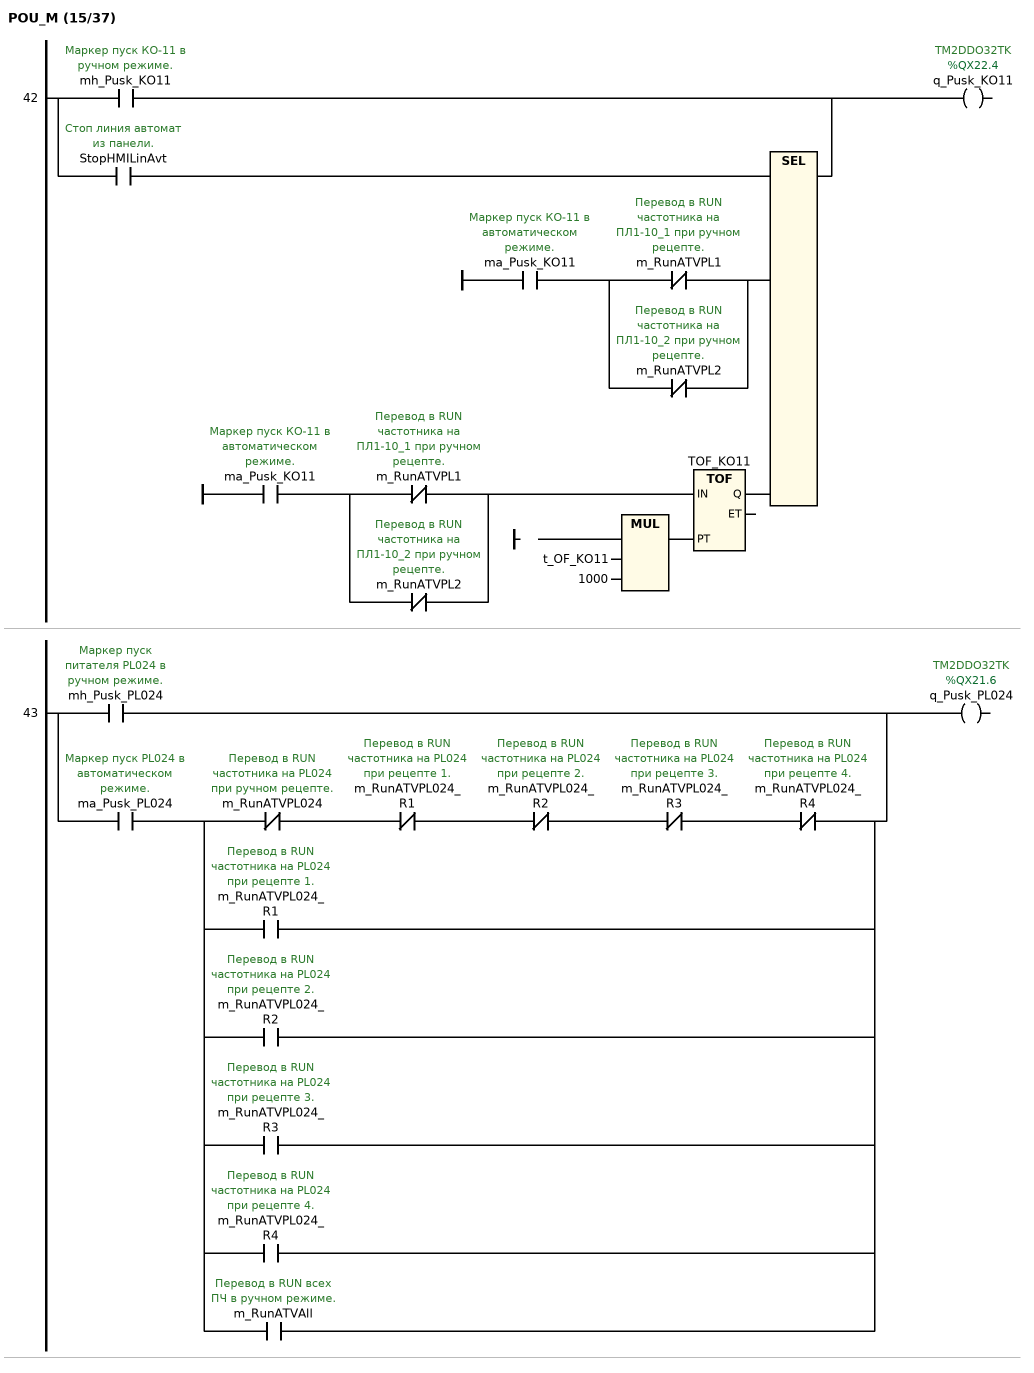
// NETWORK 42
//   mh_Pusk_KO11: Маркер пуск КО-11 в ручном режиме.
//   StopHMILinAvt: Стоп линия автомат из панели.
//   ma_Pusk_KO11: Маркер пуск КО-11 в автоматическом режиме.
//   m_RunATVPL1: Перевод в RUN частотника на ПЛ1-10_1 при ручном рецепте.
//   m_RunATVPL2: Перевод в RUN частотника на ПЛ1-10_2 при ручном рецепте.
//   TOF_KO11: Задержка перед выключением КО-11 при "Стоп линия автомат".
//   t_OF_KO11: Время задержки перед выключением КО-11 при Стоп Линия Автомат.
//   q_Pusk_KO11: TM2DDO32TK | AT %QX22.4
TOF_KO11(IN := ma_Pusk_KO11 AND (NOT m_RunATVPL1 OR NOT m_RunATVPL2), PT := t_OF_KO11 * 1000); // TOF
q_Pusk_KO11 := mh_Pusk_KO11 OR SEL(StopHMILinAvt, ma_Pusk_KO11 AND (NOT m_RunATVPL1 OR NOT m_RunATVPL2), TOF_KO11.Q);

// NETWORK 43
//   mh_Pusk_PL024: Маркер пуск питателя PL024 в ручном режиме.
//   ma_Pusk_PL024: Маркер пуск PL024 в автоматическом режиме.
//   m_RunATVPL024: Перевод в RUN частотника на PL024 при ручном рецепте.
//   m_RunATVPL024_R1: Перевод в RUN частотника на PL024 при рецепте 1.
//   m_RunATVPL024_R2: Перевод в RUN частотника на PL024 при рецепте 2.
//   m_RunATVPL024_R3: Перевод в RUN частотника на PL024 при рецепте 3.
//   m_RunATVPL024_R4: Перевод в RUN частотника на PL024 при рецепте 4.
//   m_RunATVAll: Перевод в RUN всех ПЧ в ручном режиме.
//   q_Pusk_PL024: TM2DDO32TK | AT %QX21.6
q_Pusk_PL024 := mh_Pusk_PL024 OR ma_Pusk_PL024 AND (NOT m_RunATVPL024 AND NOT m_RunATVPL024_R1 AND NOT m_RunATVPL024_R2 AND NOT m_RunATVPL024_R3 AND NOT m_RunATVPL024_R4 OR m_RunATVPL024_R1 OR m_RunATVPL024_R2 OR m_RunATVPL024_R3 OR m_RunATVPL024_R4 OR m_RunATVAll);

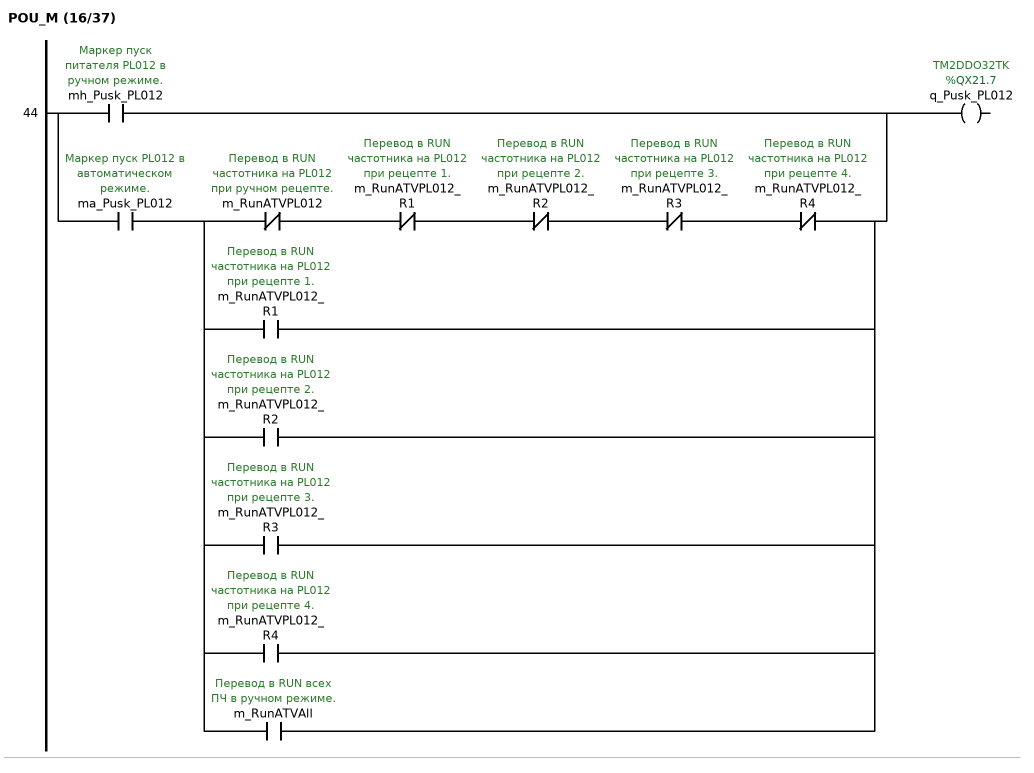
// NETWORK 44
//   mh_Pusk_PL012: Маркер пуск питателя PL012 в ручном режиме.
//   ma_Pusk_PL012: Маркер пуск PL012 в автоматическом режиме.
//   m_RunATVPL012: Перевод в RUN частотника на PL012 при ручном рецепте.
//   m_RunATVPL012_R1: Перевод в RUN частотника на PL012 при рецепте 1.
//   m_RunATVPL012_R2: Перевод в RUN частотника на PL012 при рецепте 2.
//   m_RunATVPL012_R3: Перевод в RUN частотника на PL012 при рецепте 3.
//   m_RunATVPL012_R4: Перевод в RUN частотника на PL012 при рецепте 4.
//   m_RunATVAll: Перевод в RUN всех ПЧ в ручном режиме.
//   q_Pusk_PL012: TM2DDO32TK | AT %QX21.7
q_Pusk_PL012 := mh_Pusk_PL012 OR ma_Pusk_PL012 AND (NOT m_RunATVPL012 AND NOT m_RunATVPL012_R1 AND NOT m_RunATVPL012_R2 AND NOT m_RunATVPL012_R3 AND NOT m_RunATVPL012_R4 OR m_RunATVPL012_R1 OR m_RunATVPL012_R2 OR m_RunATVPL012_R3 OR m_RunATVPL012_R4 OR m_RunATVAll);

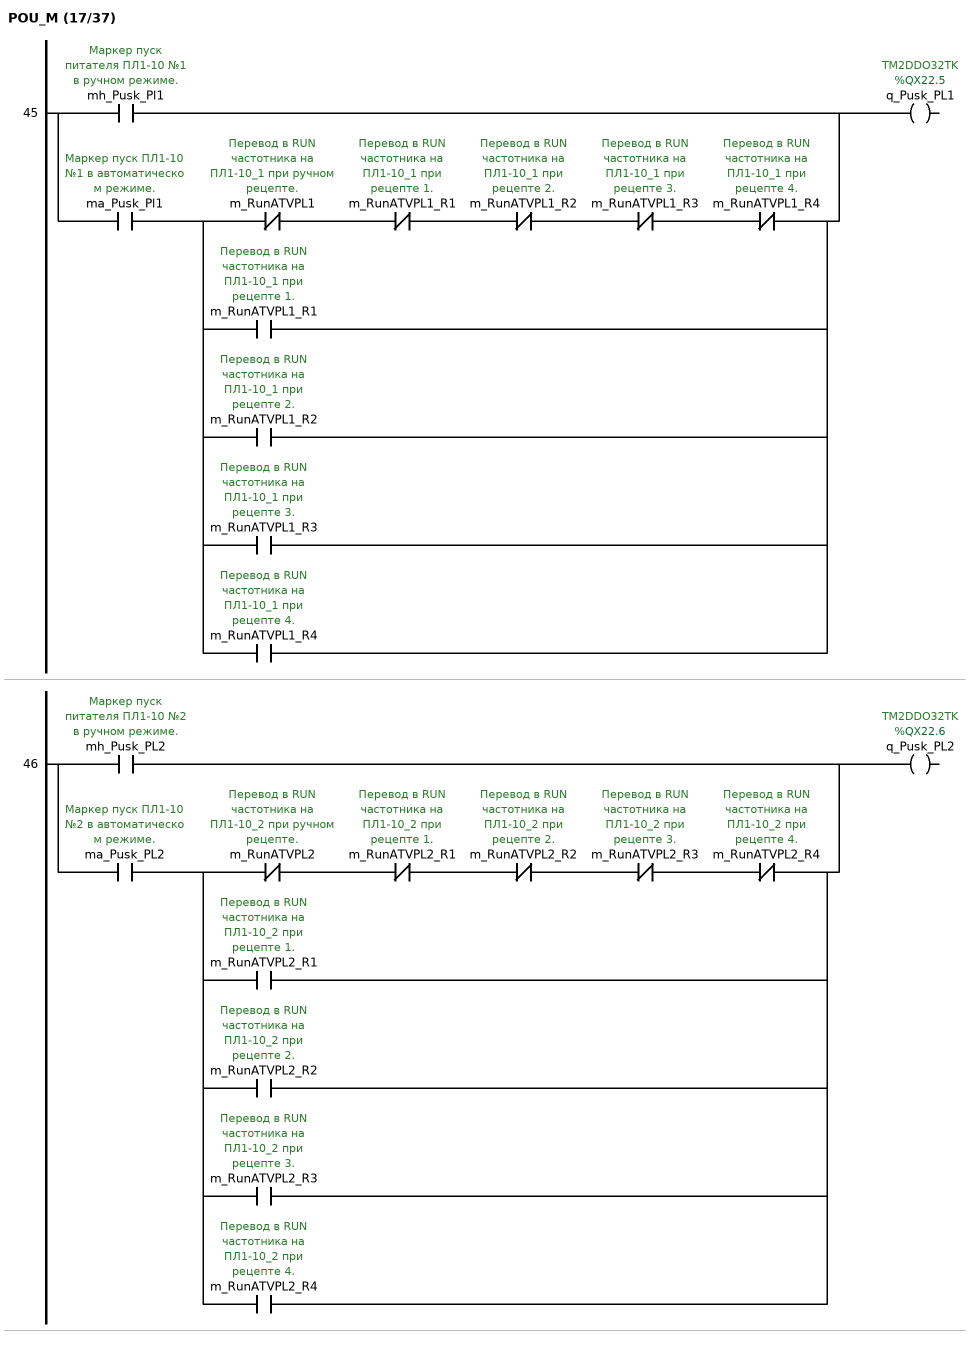
// NETWORK 45
//   mh_Pusk_Pl1: Маркер пуск питателя ПЛ1-10 №1 в ручном режиме.
//   ma_Pusk_Pl1: Маркер пуск ПЛ1-10 №1 в автоматическом режиме.
//   m_RunATVPL1: Перевод в RUN частотника на ПЛ1-10_1 при ручном рецепте.
//   m_RunATVPL1_R1: Перевод в RUN частотника на ПЛ1-10_1 при рецепте 1.
//   m_RunATVPL1_R2: Перевод в RUN частотника на ПЛ1-10_1 при рецепте 2.
//   m_RunATVPL1_R3: Перевод в RUN частотника на ПЛ1-10_1 при рецепте 3.
//   m_RunATVPL1_R4: Перевод в RUN частотника на ПЛ1-10_1 при рецепте 4.
//   q_Pusk_PL1: TM2DDO32TK | AT %QX22.5
q_Pusk_PL1 := mh_Pusk_Pl1 OR ma_Pusk_Pl1 AND (NOT m_RunATVPL1 AND NOT m_RunATVPL1_R1 AND NOT m_RunATVPL1_R2 AND NOT m_RunATVPL1_R3 AND NOT m_RunATVPL1_R4 OR m_RunATVPL1_R1 OR m_RunATVPL1_R2 OR m_RunATVPL1_R3 OR m_RunATVPL1_R4);

// NETWORK 46
//   mh_Pusk_PL2: Маркер пуск питателя ПЛ1-10 №2 в ручном режиме.
//   ma_Pusk_PL2: Маркер пуск ПЛ1-10 №2 в автоматическом режиме.
//   m_RunATVPL2: Перевод в RUN частотника на ПЛ1-10_2 при ручном рецепте.
//   m_RunATVPL2_R1: Перевод в RUN частотника на ПЛ1-10_2 при рецепте 1.
//   m_RunATVPL2_R2: Перевод в RUN частотника на ПЛ1-10_2 при рецепте 2.
//   m_RunATVPL2_R3: Перевод в RUN частотника на ПЛ1-10_2 при рецепте 3.
//   m_RunATVPL2_R4: Перевод в RUN частотника на ПЛ1-10_2 при рецепте 4.
//   q_Pusk_PL2: TM2DDO32TK | AT %QX22.6
q_Pusk_PL2 := mh_Pusk_PL2 OR ma_Pusk_PL2 AND (NOT m_RunATVPL2 AND NOT m_RunATVPL2_R1 AND NOT m_RunATVPL2_R2 AND NOT m_RunATVPL2_R3 AND NOT m_RunATVPL2_R4 OR m_RunATVPL2_R1 OR m_RunATVPL2_R2 OR m_RunATVPL2_R3 OR m_RunATVPL2_R4);

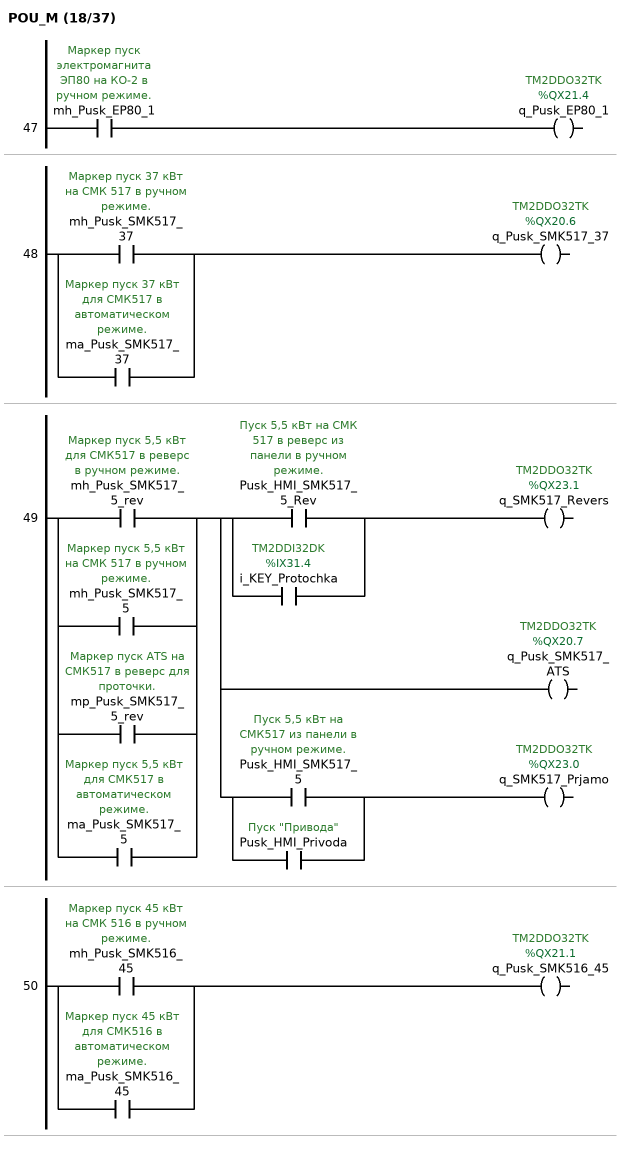
// NETWORK 47
//   mh_Pusk_EP80_1: Маркер пуск электромагнита ЭП80 на КО-2 в ручном режиме.
//   q_Pusk_EP80_1: TM2DDO32TK | AT %QX21.4
q_Pusk_EP80_1 := mh_Pusk_EP80_1;

// NETWORK 48
//   mh_Pusk_SMK517_37: Маркер пуск 37 кВт на СМК 517 в ручном режиме.
//   ma_Pusk_SMK517_37: Маркер пуск 37 кВт для СМК517 в автоматическом режиме.
//   q_Pusk_SMK517_37: TM2DDO32TK | AT %QX20.6
q_Pusk_SMK517_37 := mh_Pusk_SMK517_37 OR ma_Pusk_SMK517_37;

// NETWORK 49
//   mh_Pusk_SMK517_5_rev: Маркер пуск 5,5 кВт для СМК517 в реверс в ручном режиме.
//   mh_Pusk_SMK517_5: Маркер пуск 5,5 кВт на СМК 517 в ручном режиме.
//   mp_Pusk_SMK517_5_rev: Маркер пуск ATS на СМК517 в реверс для проточки.
//   ma_Pusk_SMK517_5: Маркер пуск 5,5 кВт для СМК517 в автоматическом режиме.
//   Pusk_HMI_SMK517_5_Rev: Пуск 5,5 кВт на СМК 517 в реверс из панели в ручном режиме.
//   i_KEY_Protochka: TM2DDI32DK | AT %IX31.4
//   q_SMK517_Revers: TM2DDO32TK | AT %QX23.1
//   q_Pusk_SMK517_ATS: TM2DDO32TK | AT %QX20.7
//   Pusk_HMI_SMK517_5: Пуск 5,5 кВт на СМК517 из панели в ручном режиме.
//   Pusk_HMI_Privoda: Пуск "Привода"
//   q_SMK517_Prjamo: TM2DDO32TK | AT %QX23.0
_w8 := mh_Pusk_SMK517_5_rev OR mh_Pusk_SMK517_5 OR mp_Pusk_SMK517_5_rev OR ma_Pusk_SMK517_5;
q_SMK517_Revers := _w8 AND (Pusk_HMI_SMK517_5_Rev OR i_KEY_Protochka);
q_Pusk_SMK517_ATS := _w8;
q_SMK517_Prjamo := _w8 AND (Pusk_HMI_SMK517_5 OR Pusk_HMI_Privoda);

// NETWORK 50
//   mh_Pusk_SMK516_45: Маркер пуск 45 кВт на СМК 516 в ручном режиме.
//   ma_Pusk_SMK516_45: Маркер пуск 45 кВт для СМК516 в автоматическом режиме.
//   q_Pusk_SMK516_45: TM2DDO32TK | AT %QX21.1
q_Pusk_SMK516_45 := mh_Pusk_SMK516_45 OR ma_Pusk_SMK516_45;

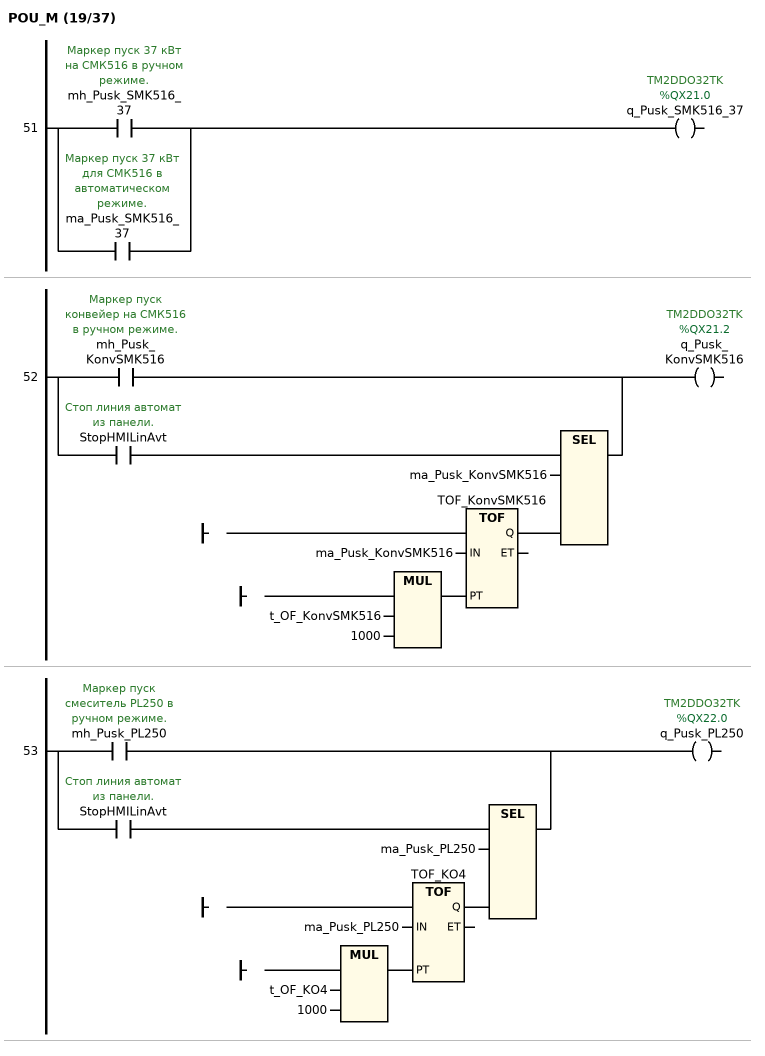
// NETWORK 51
//   mh_Pusk_SMK516_37: Маркер пуск 37 кВт на СМК516 в ручном режиме.
//   ma_Pusk_SMK516_37: Маркер пуск 37 кВт для СМК516 в автоматическом режиме.
//   q_Pusk_SMK516_37: TM2DDO32TK | AT %QX21.0
q_Pusk_SMK516_37 := mh_Pusk_SMK516_37 OR ma_Pusk_SMK516_37;

// NETWORK 52
//   mh_Pusk_KonvSMK516: Маркер пуск конвейер на СМК516 в ручном режиме.
//   StopHMILinAvt: Стоп линия автомат из панели.
//   ma_Pusk_KonvSMK516: Маркер пуск конвейер на СМК516 в автоматическом режиме.
//   TOF_KonvSMK516: Задержка перед выключением конвейера на СМК516 при "Стоп линия автомат".
//   t_OF_KonvSMK516: Время задержки перед выключением конвейера на СМК516 при Стоп Линия Автомат.
//   q_Pusk_KonvSMK516: TM2DDO32TK | AT %QX21.2
TOF_KonvSMK516(IN := ma_Pusk_KonvSMK516, PT := t_OF_KonvSMK516 * 1000); // TOF
q_Pusk_KonvSMK516 := mh_Pusk_KonvSMK516 OR SEL(StopHMILinAvt, ma_Pusk_KonvSMK516, TOF_KonvSMK516.Q);

// NETWORK 53
//   mh_Pusk_PL250: Маркер пуск смеситель PL250 в ручном режиме.
//   StopHMILinAvt: Стоп линия автомат из панели.
//   ma_Pusk_PL250: Маркер пуск PL250 в автоматическом режиме.
//   TOF_KO4: Задержка перед выключением КО-4 при "Стоп линия автомат".
//   t_OF_KO4: Время задержки перед выключением КО-4 при Стоп Линия Автомат.
//   q_Pusk_PL250: TM2DDO32TK | AT %QX22.0
TOF_KO4(IN := ma_Pusk_PL250, PT := t_OF_KO4 * 1000); // TOF
q_Pusk_PL250 := mh_Pusk_PL250 OR SEL(StopHMILinAvt, ma_Pusk_PL250, TOF_KO4.Q);

